// TIA Portal V20 export
FUNCTION_BLOCK "Sequence_1_JRUnloading"   // FB32865, LAD
TITLE = Sequence
// Sequence template programmend in ladder logic
// stored: IsIECCheckEnabled true, MemoryReserve 100, Namespace Unit1.Em13, SetENOAutomatically true
   VAR_INPUT
      unitStatus { ExternalAccessible := 'False'; ExternalVisible := 'False'; ExternalWritable := 'False'} : "LAF_typeUnitStatus";   // Current unit status o be used in this EM
   END_VAR
   VAR
      instSequenceLADControl { ExternalAccessible := 'False'; ExternalVisible := 'False'; ExternalWritable := 'False'} : "LAF_ControlLadSequence";
      instSequenceLADStatus { ExternalAccessible := 'False'; ExternalVisible := 'False'; ExternalWritable := 'False'} : "LAF_StatusLadSequence";
      statTonTime { ExternalAccessible := 'False'; ExternalVisible := 'False'; ExternalWritable := 'False'} : Array[0..9999] of TON_TIME;
      NoDataCheck { S7_SetPoint := 'True'} : "LER_typePartData";
      statPulse { ExternalWritable := 'False'} : Array[0..9] of Bool;
   END_VAR
   VAR_TEMP
      tempCustomerAction : Bool;   // Placeholder for possible actions
      tempDo_nothing_and_wait_for_init : Bool;   // Placeholder for doing nothing
      tempSafeStateCondition : Bool;   // Temp Condition for the equipment module to be in a safe state
   END_VAR
   VAR CONSTANT
      STEP_IDLE : DInt := 1;
      JOB_1_STEP_01 : DInt := 101;
      JOB_1_STEP_10 : DInt := 110;
      JOB_1_STEP_20 : DInt := 120;
      JOB_1_STEP_30 : DInt := 130;
      JOB_1_STEP_40 : DInt := 140;
      JOB_1_STEP_50 : DInt := 150;
      JOB_1_STEP_60 : DInt := 160;
      JOB_1_STEP_70 : DInt := 170;
      JOB_1_STEP_80 : DInt := 180;
      JOB_1_STEP_90 : DInt := 190;
      JOB_2_STEP_01 : DInt := 201;
      JOB_2_STEP_10 : DInt := 210;
      JOB_2_STEP_20 : DInt := 220;
      JOB_2_STEP_30 : DInt := 230;
      JOB_2_STEP_40 : DInt := 240;
      JOB_2_STEP_50 : DInt := 250;
      JOB_2_STEP_51 : DInt := 251;
      JOB_2_STEP_60 : DInt := 260;
      JOB_2_STEP_70 : DInt := 270;
      JOB_2_STEP_80 : DInt := 280;
      JOB_2_STEP_90 : DInt := 290;
      JOB_3_STEP_01 : DInt := 301;
      JOB_3_STEP_10 : DInt := 310;
      JOB_3_STEP_20 : DInt := 320;
      JOB_3_STEP_30 : DInt := 330;
      JOB_3_STEP_31 : DInt := 331;
      JOB_3_STEP_32 : DInt := 332;
      JOB_3_STEP_33 : DInt := 333;
      JOB_3_STEP_34 : DInt := 334;
      JOB_3_STEP_35 : DInt := 335;
      JOB_3_STEP_36 : DInt := 336;
      JOB_3_STEP_37 : DInt := 337;
      JOB_3_STEP_38 : DInt := 338;
      JOB_3_STEP_39 : DInt := 339;
      JOB_3_STEP_40 : DInt := 340;
      JOB_3_STEP_41 : DInt := 341;
      JOB_3_STEP_50 : DInt := 350;
      JOB_3_STEP_60 : DInt := 360;
      JOB_3_STEP_70 : DInt := 370;
      JOB_3_STEP_80 : DInt := 380;
      JOB_3_STEP_90 : DInt := 390;
      JOB_4_STEP_01 : DInt := 401;
      JOB_4_STEP_10 : DInt := 410;
      JOB_4_STEP_11 : DInt := 411;
      JOB_4_STEP_20 : DInt := 420;
      JOB_4_STEP_30 : DInt := 430;
      JOB_4_STEP_31 : DInt := 431;
      JOB_4_STEP_40 : DInt := 440;
      JOB_4_STEP_50 : DInt := 450;
      JOB_4_STEP_51 : DInt := 451;
      JOB_4_STEP_60 : DInt := 460;
      JOB_4_STEP_70 : DInt := 470;
      JOB_4_STEP_71 : DInt := 471;
      JOB_4_STEP_80 : DInt := 480;
      JOB_4_STEP_90 : DInt := 490;
      STEP_IMMEDIATE_STOP : DInt := 9001;   // Step executed when an immediate stop command is triggered for the sequence (i.e. when unit is in state aborting)
      TO_DO_INSERT_ACTIONS_HERE : Bool := TRUE;   // Template : Add actions
      TO_DO_INSERT_CONDITION_FOR_TRANSITION_HERE : Bool := TRUE;   // Template : Add conditions
   END_VAR
   VAR_TEMP   // added for the SCL form of the ladder/FBD networks
      _w1 : Bool;
      _w2 : Bool;
      _w3 : Bool;
      _w4 : Bool;
      _w5 : Bool;
   END_VAR
BEGIN

REGION Network 1: BLOCK INFO HEADER
   // (company) / (C) Copyright (year)
   // ---------------------------------------------------------------------------------
   // Title:                             (Title of this block)
   // Comment/Function: (that is implemented in the block)
   // Library/Family:           (that the source is dedicated to)
   // Author:                        (department / person in charge / contact)
   // Target System:          (test system with FW version)
   // Engineering:              TIA Portal (SW version)
   // Restrictions:               (OB types, etc.)
   // Requirements:           (hardware, technological package, etc.)
   // ---------------------------------------------------------------------------------
   // Change log table:
   // Version          | Date             | Signature      | Expert in charge  | Changes applied ------------------------|----------------------|-------------------------|--------------------------------|-----------------------
   // 001.000.000 | yyyy-mm-dd | 0x00000000 | (name of expert) | First released version
END_REGION

REGION Network 2: DESCRIPTION
   // This is a template block provided by the Automation Framework. It can be used to create an own project.
   // The Block Info Header is prepared to put in your own data.
   // Description of the block could be added here and the docu created by Code2Docu.
END_REGION

REGION Network 3: ********************* CONTROL *************************
END_REGION

REGION Network 4: Sequence Control ("Enter your Sequins number here")
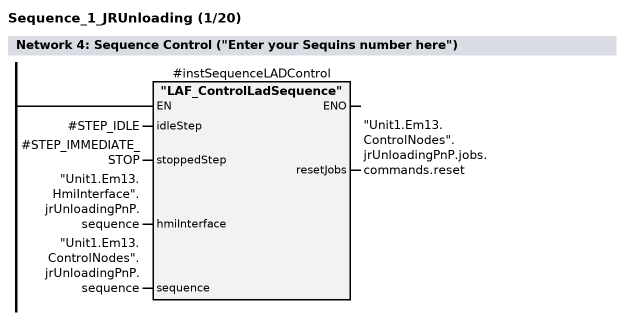
   RUNG wire#powerrail
      #instSequenceLADControl(idleStep := #STEP_IDLE, stoppedStep := #STEP_IMMEDIATE_STOP, hmiInterface := "Unit1.Em13.HmiInterface".jrUnloadingPnP.sequence, sequence := "Unit1.Em13.ControlNodes".jrUnloadingPnP.sequence, resetJobs => "Unit1.Em13.ControlNodes".jrUnloadingPnP.jobs.commands.reset)
   END_RUNG
   // the same network as SCL:
   #instSequenceLADControl(idleStep := #STEP_IDLE,   // "LAF_ControlLadSequence"
                           stoppedStep := #STEP_IMMEDIATE_STOP,
                           hmiInterface := "Unit1.Em13.HmiInterface".jrUnloadingPnP.sequence,
                           sequence := "Unit1.Em13.ControlNodes".jrUnloadingPnP.sequence,
                           resetJobs => "Unit1.Em13.ControlNodes".jrUnloadingPnP.jobs.commands.reset);
END_REGION

REGION Network 5: Step IDLE
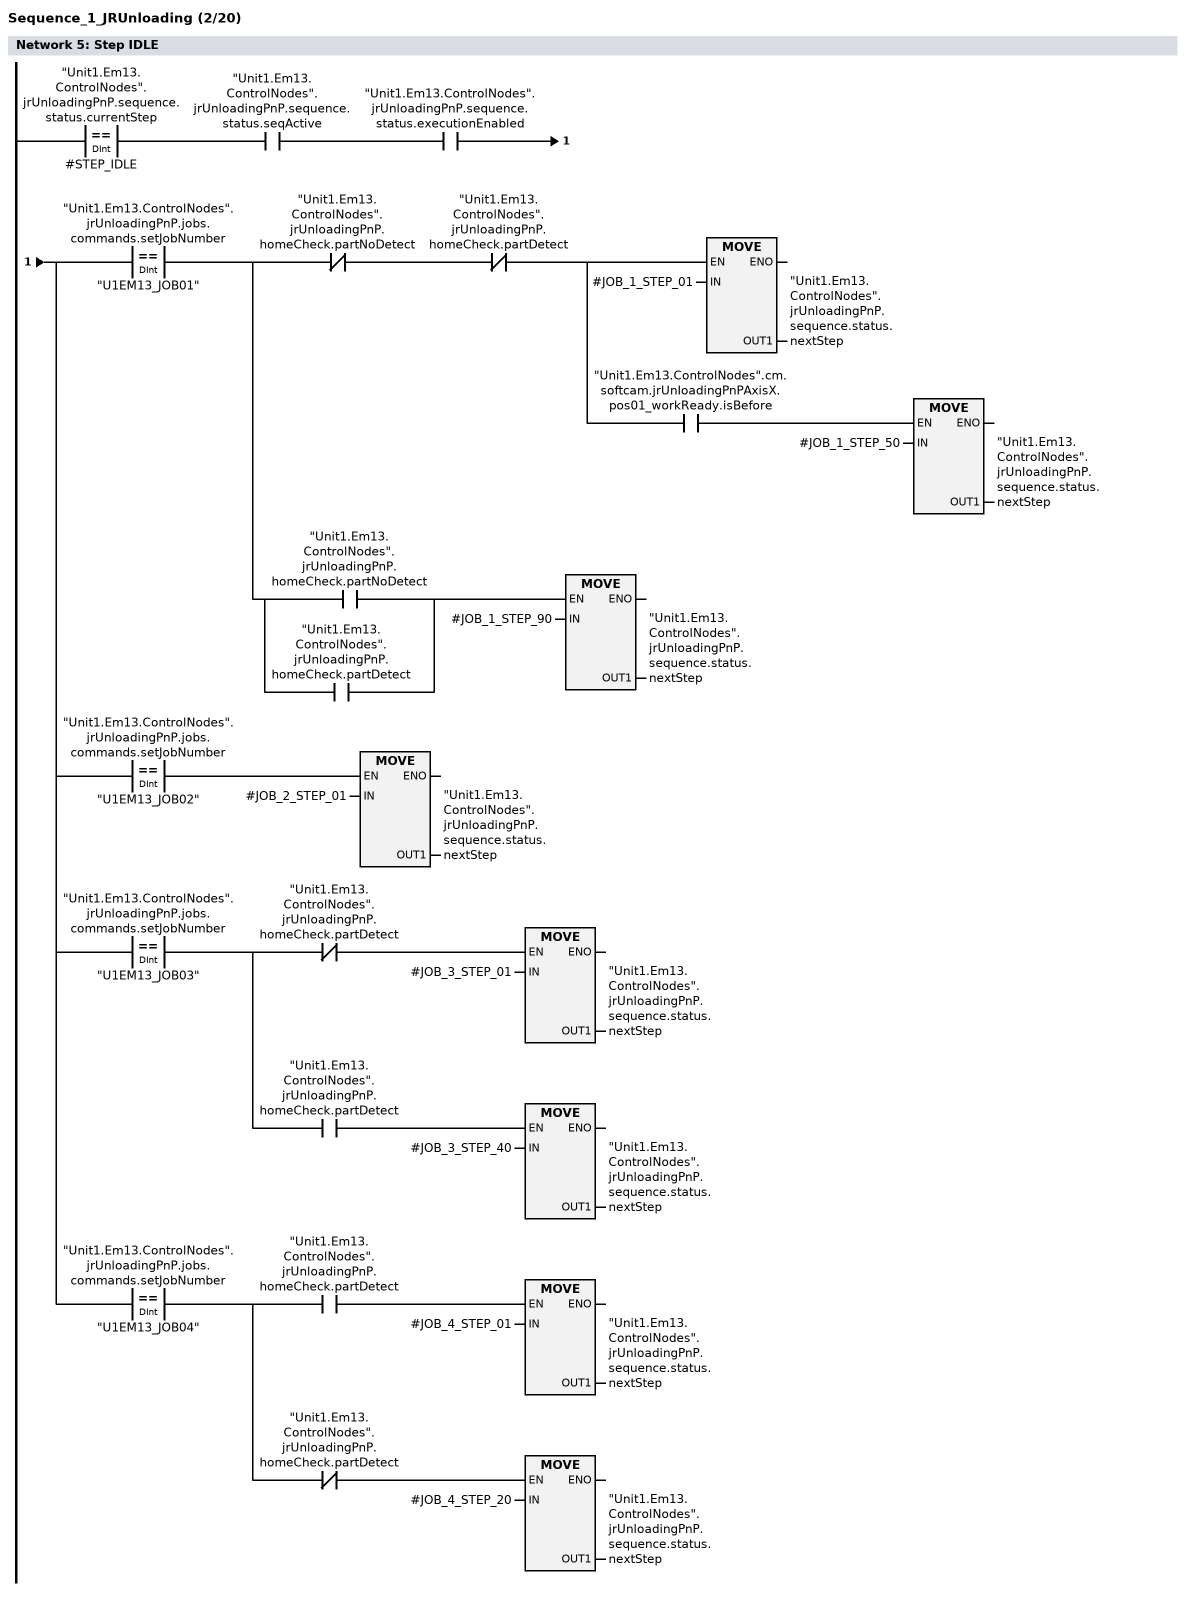
   RUNG wire#powerrail
      { S7_Templates := "SrcType := DInt" } EQ_Contact(in1 := "Unit1.Em13.ControlNodes".jrUnloadingPnP.sequence.status.currentStep, in2 := #STEP_IDLE)
      Contact( "Unit1.Em13.ControlNodes".jrUnloadingPnP.sequence.status.seqActive )
      Contact( "Unit1.Em13.ControlNodes".jrUnloadingPnP.sequence.status.executionEnabled )
      wire#w1
      { S7_Templates := "SrcType := DInt" } EQ_Contact(in1 := "Unit1.Em13.ControlNodes".jrUnloadingPnP.jobs.commands.setJobNumber, in2 := "U1EM13_JOB01")
      wire#w2
      I_Contact( "Unit1.Em13.ControlNodes".jrUnloadingPnP.homeCheck.partNoDetect )
      I_Contact( "Unit1.Em13.ControlNodes".jrUnloadingPnP.homeCheck.partDetect )
      wire#w3
      Move(in := #JOB_1_STEP_01, out1 => "Unit1.Em13.ControlNodes".jrUnloadingPnP.sequence.status.nextStep)
   END_RUNG
   RUNG wire#w3
      Contact( "Unit1.Em13.ControlNodes".cm.softcam.jrUnIoadingPnPAxisX.pos01_workReady.isBefore )
      Move(in := #JOB_1_STEP_50, out1 => "Unit1.Em13.ControlNodes".jrUnloadingPnP.sequence.status.nextStep)
   END_RUNG
   RUNG wire#w2
      Contact( "Unit1.Em13.ControlNodes".jrUnloadingPnP.homeCheck.partNoDetect )
      wire#w4
      Move(in := #JOB_1_STEP_90, out1 => "Unit1.Em13.ControlNodes".jrUnloadingPnP.sequence.status.nextStep)
   END_RUNG
   RUNG wire#w2
      Contact( "Unit1.Em13.ControlNodes".jrUnloadingPnP.homeCheck.partDetect )
   END_RUNG wire#w4
   RUNG wire#w1
      { S7_Templates := "SrcType := DInt" } EQ_Contact(in1 := "Unit1.Em13.ControlNodes".jrUnloadingPnP.jobs.commands.setJobNumber, in2 := "U1EM13_JOB02")
      Move(in := #JOB_2_STEP_01, out1 => "Unit1.Em13.ControlNodes".jrUnloadingPnP.sequence.status.nextStep)
   END_RUNG
   RUNG wire#w1
      { S7_Templates := "SrcType := DInt" } EQ_Contact(in1 := "Unit1.Em13.ControlNodes".jrUnloadingPnP.jobs.commands.setJobNumber, in2 := "U1EM13_JOB03")
      wire#w5
      I_Contact( "Unit1.Em13.ControlNodes".jrUnloadingPnP.homeCheck.partDetect )
      Move(in := #JOB_3_STEP_01, out1 => "Unit1.Em13.ControlNodes".jrUnloadingPnP.sequence.status.nextStep)
   END_RUNG
   RUNG wire#w5
      Contact( "Unit1.Em13.ControlNodes".jrUnloadingPnP.homeCheck.partDetect )
      Move(in := #JOB_3_STEP_40, out1 => "Unit1.Em13.ControlNodes".jrUnloadingPnP.sequence.status.nextStep)
   END_RUNG
   RUNG wire#w1
      { S7_Templates := "SrcType := DInt" } EQ_Contact(in1 := "Unit1.Em13.ControlNodes".jrUnloadingPnP.jobs.commands.setJobNumber, in2 := "U1EM13_JOB04")
      wire#w6
      Contact( "Unit1.Em13.ControlNodes".jrUnloadingPnP.homeCheck.partDetect )
      Move(in := #JOB_4_STEP_01, out1 => "Unit1.Em13.ControlNodes".jrUnloadingPnP.sequence.status.nextStep)
   END_RUNG
   RUNG wire#w6
      I_Contact( "Unit1.Em13.ControlNodes".jrUnloadingPnP.homeCheck.partDetect )
      Move(in := #JOB_4_STEP_20, out1 => "Unit1.Em13.ControlNodes".jrUnloadingPnP.sequence.status.nextStep)
   END_RUNG
   // the same network as SCL:
   #_w1 := ("Unit1.Em13.ControlNodes".jrUnloadingPnP.sequence.status.currentStep = #STEP_IDLE) AND "Unit1.Em13.ControlNodes".jrUnloadingPnP.sequence.status.seqActive AND "Unit1.Em13.ControlNodes".jrUnloadingPnP.sequence.status.executionEnabled;
   #_w2 := #_w1 AND ("Unit1.Em13.ControlNodes".jrUnloadingPnP.jobs.commands.setJobNumber = "U1EM13_JOB01");
   #_w3 := #_w2 AND NOT "Unit1.Em13.ControlNodes".jrUnloadingPnP.homeCheck.partNoDetect AND NOT "Unit1.Em13.ControlNodes".jrUnloadingPnP.homeCheck.partDetect;
   IF #_w3 THEN "Unit1.Em13.ControlNodes".jrUnloadingPnP.sequence.status.nextStep := #JOB_1_STEP_01; END_IF;
   IF #_w3 AND "Unit1.Em13.ControlNodes".cm.softcam.jrUnIoadingPnPAxisX.pos01_workReady.isBefore THEN
       "Unit1.Em13.ControlNodes".jrUnloadingPnP.sequence.status.nextStep := #JOB_1_STEP_50;
   END_IF;
   IF #_w2 AND ("Unit1.Em13.ControlNodes".jrUnloadingPnP.homeCheck.partNoDetect OR "Unit1.Em13.ControlNodes".jrUnloadingPnP.homeCheck.partDetect) THEN
       "Unit1.Em13.ControlNodes".jrUnloadingPnP.sequence.status.nextStep := #JOB_1_STEP_90;
   END_IF;
   IF #_w1 AND ("Unit1.Em13.ControlNodes".jrUnloadingPnP.jobs.commands.setJobNumber = "U1EM13_JOB02") THEN
       "Unit1.Em13.ControlNodes".jrUnloadingPnP.sequence.status.nextStep := #JOB_2_STEP_01;
   END_IF;
   #_w4 := #_w1 AND ("Unit1.Em13.ControlNodes".jrUnloadingPnP.jobs.commands.setJobNumber = "U1EM13_JOB03");
   IF #_w4 AND NOT "Unit1.Em13.ControlNodes".jrUnloadingPnP.homeCheck.partDetect THEN
       "Unit1.Em13.ControlNodes".jrUnloadingPnP.sequence.status.nextStep := #JOB_3_STEP_01;
   END_IF;
   IF #_w4 AND "Unit1.Em13.ControlNodes".jrUnloadingPnP.homeCheck.partDetect THEN
       "Unit1.Em13.ControlNodes".jrUnloadingPnP.sequence.status.nextStep := #JOB_3_STEP_40;
   END_IF;
   #_w5 := #_w1 AND ("Unit1.Em13.ControlNodes".jrUnloadingPnP.jobs.commands.setJobNumber = "U1EM13_JOB04");
   IF #_w5 AND "Unit1.Em13.ControlNodes".jrUnloadingPnP.homeCheck.partDetect THEN
       "Unit1.Em13.ControlNodes".jrUnloadingPnP.sequence.status.nextStep := #JOB_4_STEP_01;
   END_IF;
   IF #_w5 AND NOT "Unit1.Em13.ControlNodes".jrUnloadingPnP.homeCheck.partDetect THEN
       "Unit1.Em13.ControlNodes".jrUnloadingPnP.sequence.status.nextStep := #JOB_4_STEP_20;
   END_IF;
END_REGION

REGION Network 6: *************** JOB[1] EM HOMING ************************
END_REGION

REGION Network 7: Step[101] : JOB[1] Condition
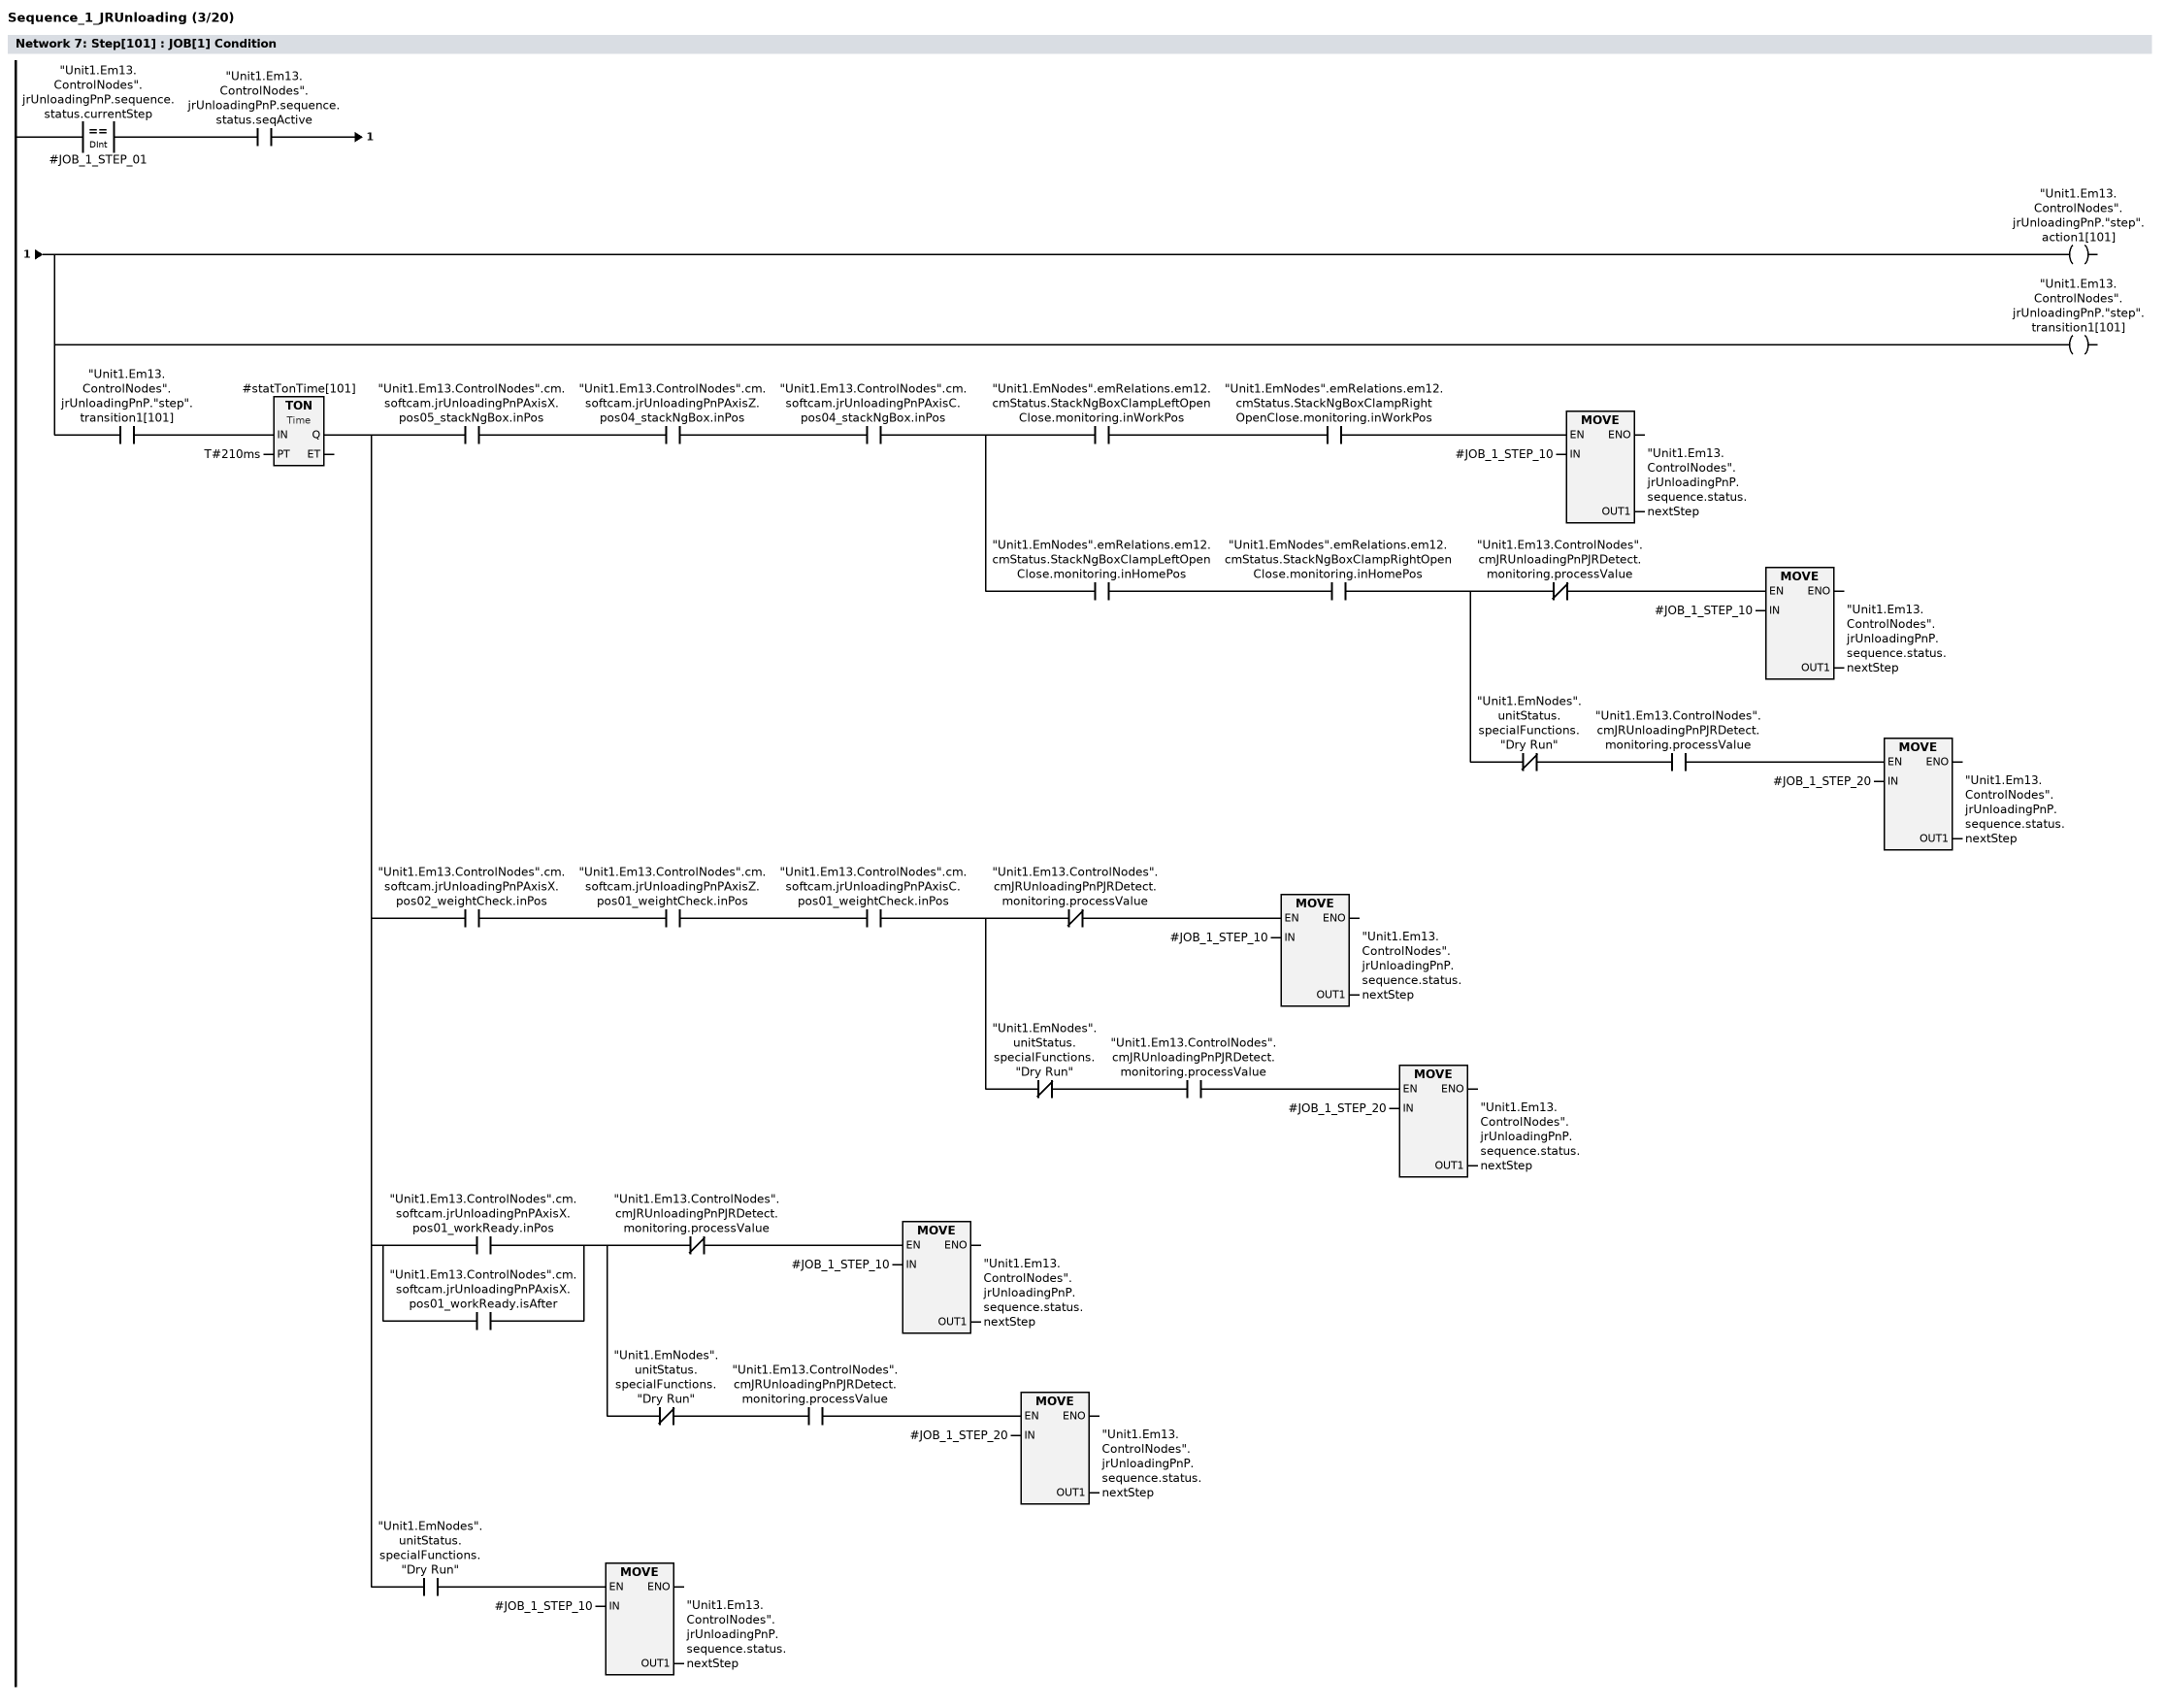
   RUNG wire#powerrail
      { S7_Templates := "SrcType := DInt" } EQ_Contact(in1 := "Unit1.Em13.ControlNodes".jrUnloadingPnP.sequence.status.currentStep, in2 := #JOB_1_STEP_01)
      Contact( "Unit1.Em13.ControlNodes".jrUnloadingPnP.sequence.status.seqActive )
      wire#w1
      Coil( "Unit1.Em13.ControlNodes".jrUnloadingPnP."step".action1[101] )
   END_RUNG
   RUNG wire#w1
      Coil( "Unit1.Em13.ControlNodes".jrUnloadingPnP."step".transition1[101] )
   END_RUNG
   RUNG wire#w1
      Contact( "Unit1.Em13.ControlNodes".jrUnloadingPnP."step".transition1[101] )
      { S7_Templates := "time_type := Time" } #statTonTime[101].TON(pt := T#210ms, et =>)
      wire#w2
      Contact( "Unit1.Em13.ControlNodes".cm.softcam.jrUnIoadingPnPAxisX.pos05_stackNgBox.inPos )
      Contact( "Unit1.Em13.ControlNodes".cm.softcam.jrUnIoadingPnPAxisZ.pos04_stackNgBox.inPos )
      Contact( "Unit1.Em13.ControlNodes".cm.softcam.jrUnIoadingPnPAxisC.pos04_stackNgBox.inPos )
      wire#w3
      Contact( "Unit1.EmNodes".emRelations.em12.cmStatus.StackNgBoxClampLeftOpenClose.monitoring.inWorkPos )
      Contact( "Unit1.EmNodes".emRelations.em12.cmStatus.StackNgBoxClampRightOpenClose.monitoring.inWorkPos )
      Move(in := #JOB_1_STEP_10, out1 => "Unit1.Em13.ControlNodes".jrUnloadingPnP.sequence.status.nextStep)
   END_RUNG
   RUNG wire#w3
      Contact( "Unit1.EmNodes".emRelations.em12.cmStatus.StackNgBoxClampLeftOpenClose.monitoring.inHomePos )
      Contact( "Unit1.EmNodes".emRelations.em12.cmStatus.StackNgBoxClampRightOpenClose.monitoring.inHomePos )
      wire#w4
      I_Contact( "Unit1.Em13.ControlNodes".cmJRUnloadingPnPJRDetect.monitoring.processValue )
      Move(in := #JOB_1_STEP_10, out1 => "Unit1.Em13.ControlNodes".jrUnloadingPnP.sequence.status.nextStep)
   END_RUNG
   RUNG wire#w4
      I_Contact( "Unit1.EmNodes".unitStatus.specialFunctions."Dry Run" )
      Contact( "Unit1.Em13.ControlNodes".cmJRUnloadingPnPJRDetect.monitoring.processValue )
      Move(in := #JOB_1_STEP_20, out1 => "Unit1.Em13.ControlNodes".jrUnloadingPnP.sequence.status.nextStep)
   END_RUNG
   RUNG wire#w2
      Contact( "Unit1.Em13.ControlNodes".cm.softcam.jrUnIoadingPnPAxisX.pos02_weightCheck.inPos )
      Contact( "Unit1.Em13.ControlNodes".cm.softcam.jrUnIoadingPnPAxisZ.pos01_weightCheck.inPos )
      Contact( "Unit1.Em13.ControlNodes".cm.softcam.jrUnIoadingPnPAxisC.pos01_weightCheck.inPos )
      wire#w5
      I_Contact( "Unit1.Em13.ControlNodes".cmJRUnloadingPnPJRDetect.monitoring.processValue )
      Move(in := #JOB_1_STEP_10, out1 => "Unit1.Em13.ControlNodes".jrUnloadingPnP.sequence.status.nextStep)
   END_RUNG
   RUNG wire#w5
      I_Contact( "Unit1.EmNodes".unitStatus.specialFunctions."Dry Run" )
      Contact( "Unit1.Em13.ControlNodes".cmJRUnloadingPnPJRDetect.monitoring.processValue )
      Move(in := #JOB_1_STEP_20, out1 => "Unit1.Em13.ControlNodes".jrUnloadingPnP.sequence.status.nextStep)
   END_RUNG
   RUNG wire#w2
      Contact( "Unit1.Em13.ControlNodes".cm.softcam.jrUnIoadingPnPAxisX.pos01_workReady.inPos )
      wire#w6
      I_Contact( "Unit1.Em13.ControlNodes".cmJRUnloadingPnPJRDetect.monitoring.processValue )
      Move(in := #JOB_1_STEP_10, out1 => "Unit1.Em13.ControlNodes".jrUnloadingPnP.sequence.status.nextStep)
   END_RUNG
   RUNG wire#w2
      Contact( "Unit1.Em13.ControlNodes".cm.softcam.jrUnIoadingPnPAxisX.pos01_workReady.isAfter )
   END_RUNG wire#w6
   RUNG wire#w6
      I_Contact( "Unit1.EmNodes".unitStatus.specialFunctions."Dry Run" )
      Contact( "Unit1.Em13.ControlNodes".cmJRUnloadingPnPJRDetect.monitoring.processValue )
      Move(in := #JOB_1_STEP_20, out1 => "Unit1.Em13.ControlNodes".jrUnloadingPnP.sequence.status.nextStep)
   END_RUNG
   RUNG wire#w2
      Contact( "Unit1.EmNodes".unitStatus.specialFunctions."Dry Run" )
      Move(in := #JOB_1_STEP_10, out1 => "Unit1.Em13.ControlNodes".jrUnloadingPnP.sequence.status.nextStep)
   END_RUNG
   // the same network as SCL:
   "Unit1.Em13.ControlNodes".jrUnloadingPnP."step".action1[101] := ("Unit1.Em13.ControlNodes".jrUnloadingPnP.sequence.status.currentStep = #JOB_1_STEP_01) AND "Unit1.Em13.ControlNodes".jrUnloadingPnP.sequence.status.seqActive;
   "Unit1.Em13.ControlNodes".jrUnloadingPnP."step".transition1[101] := ("Unit1.Em13.ControlNodes".jrUnloadingPnP.sequence.status.currentStep = #JOB_1_STEP_01) AND "Unit1.Em13.ControlNodes".jrUnloadingPnP.sequence.status.seqActive;
   #statTonTime[101].TON(IN := ("Unit1.Em13.ControlNodes".jrUnloadingPnP.sequence.status.currentStep = #JOB_1_STEP_01) AND "Unit1.Em13.ControlNodes".jrUnloadingPnP.sequence.status.seqActive AND "Unit1.Em13.ControlNodes".jrUnloadingPnP."step".transition1[101],
                         PT := T#210ms);
   #_w1 := #statTonTime[101].Q AND "Unit1.Em13.ControlNodes".cm.softcam.jrUnIoadingPnPAxisX.pos05_stackNgBox.inPos AND "Unit1.Em13.ControlNodes".cm.softcam.jrUnIoadingPnPAxisZ.pos04_stackNgBox.inPos AND "Unit1.Em13.ControlNodes".cm.softcam.jrUnIoadingPnPAxisC.pos04_stackNgBox.inPos;
   IF #_w1 AND "Unit1.EmNodes".emRelations.em12.cmStatus.StackNgBoxClampLeftOpenClose.monitoring.inWorkPos AND "Unit1.EmNodes".emRelations.em12.cmStatus.StackNgBoxClampRightOpenClose.monitoring.inWorkPos THEN
       "Unit1.Em13.ControlNodes".jrUnloadingPnP.sequence.status.nextStep := #JOB_1_STEP_10;
   END_IF;
   #_w2 := #_w1 AND "Unit1.EmNodes".emRelations.em12.cmStatus.StackNgBoxClampLeftOpenClose.monitoring.inHomePos AND "Unit1.EmNodes".emRelations.em12.cmStatus.StackNgBoxClampRightOpenClose.monitoring.inHomePos;
   IF #_w2 AND NOT "Unit1.Em13.ControlNodes".cmJRUnloadingPnPJRDetect.monitoring.processValue THEN
       "Unit1.Em13.ControlNodes".jrUnloadingPnP.sequence.status.nextStep := #JOB_1_STEP_10;
   END_IF;
   IF #_w2 AND NOT "Unit1.EmNodes".unitStatus.specialFunctions."Dry Run" AND "Unit1.Em13.ControlNodes".cmJRUnloadingPnPJRDetect.monitoring.processValue THEN
       "Unit1.Em13.ControlNodes".jrUnloadingPnP.sequence.status.nextStep := #JOB_1_STEP_20;
   END_IF;
   #_w3 := #statTonTime[101].Q AND "Unit1.Em13.ControlNodes".cm.softcam.jrUnIoadingPnPAxisX.pos02_weightCheck.inPos AND "Unit1.Em13.ControlNodes".cm.softcam.jrUnIoadingPnPAxisZ.pos01_weightCheck.inPos AND "Unit1.Em13.ControlNodes".cm.softcam.jrUnIoadingPnPAxisC.pos01_weightCheck.inPos;
   IF #_w3 AND NOT "Unit1.Em13.ControlNodes".cmJRUnloadingPnPJRDetect.monitoring.processValue THEN
       "Unit1.Em13.ControlNodes".jrUnloadingPnP.sequence.status.nextStep := #JOB_1_STEP_10;
   END_IF;
   IF #_w3 AND NOT "Unit1.EmNodes".unitStatus.specialFunctions."Dry Run" AND "Unit1.Em13.ControlNodes".cmJRUnloadingPnPJRDetect.monitoring.processValue THEN
       "Unit1.Em13.ControlNodes".jrUnloadingPnP.sequence.status.nextStep := #JOB_1_STEP_20;
   END_IF;
   #_w4 := #statTonTime[101].Q AND ("Unit1.Em13.ControlNodes".cm.softcam.jrUnIoadingPnPAxisX.pos01_workReady.inPos OR "Unit1.Em13.ControlNodes".cm.softcam.jrUnIoadingPnPAxisX.pos01_workReady.isAfter);
   IF #_w4 AND NOT "Unit1.Em13.ControlNodes".cmJRUnloadingPnPJRDetect.monitoring.processValue THEN
       "Unit1.Em13.ControlNodes".jrUnloadingPnP.sequence.status.nextStep := #JOB_1_STEP_10;
   END_IF;
   IF #_w4 AND NOT "Unit1.EmNodes".unitStatus.specialFunctions."Dry Run" AND "Unit1.Em13.ControlNodes".cmJRUnloadingPnPJRDetect.monitoring.processValue THEN
       "Unit1.Em13.ControlNodes".jrUnloadingPnP.sequence.status.nextStep := #JOB_1_STEP_20;
   END_IF;
   IF #statTonTime[101].Q AND "Unit1.EmNodes".unitStatus.specialFunctions."Dry Run" THEN
       "Unit1.Em13.ControlNodes".jrUnloadingPnP.sequence.status.nextStep := #JOB_1_STEP_10;
   END_IF;
END_REGION

REGION Network 8: Step[110] : Clamp Open
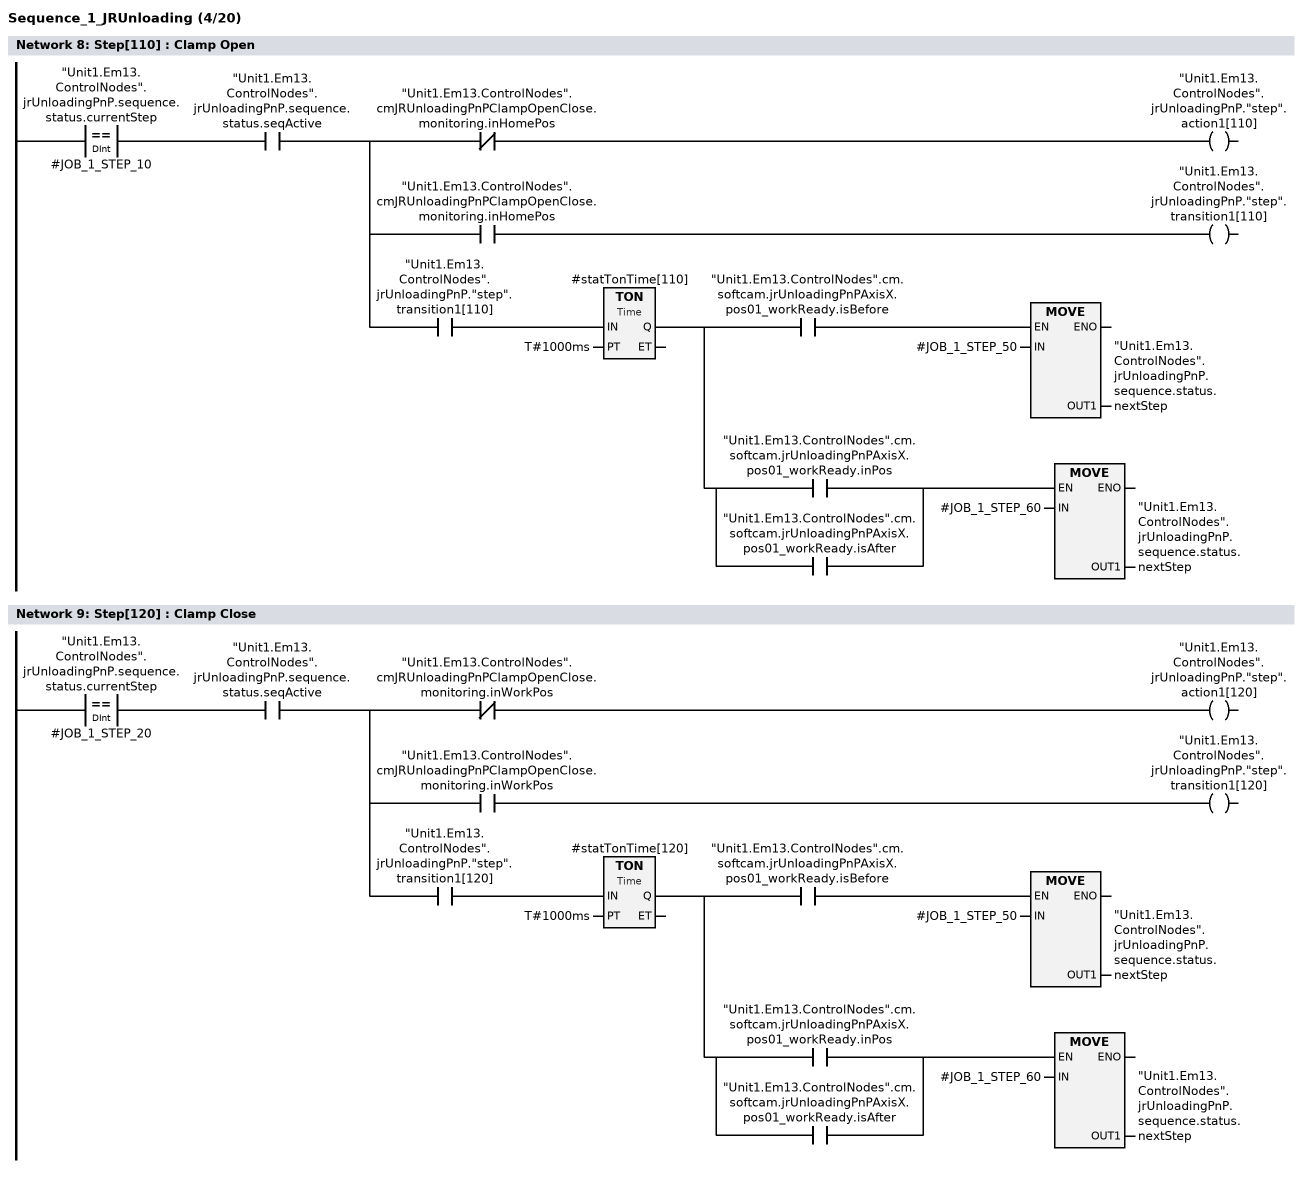
   RUNG wire#powerrail
      { S7_Templates := "SrcType := DInt" } EQ_Contact(in1 := "Unit1.Em13.ControlNodes".jrUnloadingPnP.sequence.status.currentStep, in2 := #JOB_1_STEP_10)
      Contact( "Unit1.Em13.ControlNodes".jrUnloadingPnP.sequence.status.seqActive )
      wire#w1
      I_Contact( "Unit1.Em13.ControlNodes".cmJRUnloadingPnPClampOpenClose.monitoring.inHomePos )
      Coil( "Unit1.Em13.ControlNodes".jrUnloadingPnP."step".action1[110] )
   END_RUNG
   RUNG wire#w1
      Contact( "Unit1.Em13.ControlNodes".cmJRUnloadingPnPClampOpenClose.monitoring.inHomePos )
      Coil( "Unit1.Em13.ControlNodes".jrUnloadingPnP."step".transition1[110] )
   END_RUNG
   RUNG wire#w1
      Contact( "Unit1.Em13.ControlNodes".jrUnloadingPnP."step".transition1[110] )
      { S7_Templates := "time_type := Time" } #statTonTime[110].TON(pt := T#1000ms, et =>)
      wire#w2
      Contact( "Unit1.Em13.ControlNodes".cm.softcam.jrUnIoadingPnPAxisX.pos01_workReady.isBefore )
      Move(in := #JOB_1_STEP_50, out1 => "Unit1.Em13.ControlNodes".jrUnloadingPnP.sequence.status.nextStep)
   END_RUNG
   RUNG wire#w2
      Contact( "Unit1.Em13.ControlNodes".cm.softcam.jrUnIoadingPnPAxisX.pos01_workReady.inPos )
      wire#w3
      Move(in := #JOB_1_STEP_60, out1 => "Unit1.Em13.ControlNodes".jrUnloadingPnP.sequence.status.nextStep)
   END_RUNG
   RUNG wire#w2
      Contact( "Unit1.Em13.ControlNodes".cm.softcam.jrUnIoadingPnPAxisX.pos01_workReady.isAfter )
   END_RUNG wire#w3
   // the same network as SCL:
   #_w1 := ("Unit1.Em13.ControlNodes".jrUnloadingPnP.sequence.status.currentStep = #JOB_1_STEP_10) AND "Unit1.Em13.ControlNodes".jrUnloadingPnP.sequence.status.seqActive;
   "Unit1.Em13.ControlNodes".jrUnloadingPnP."step".action1[110] := #_w1 AND NOT "Unit1.Em13.ControlNodes".cmJRUnloadingPnPClampOpenClose.monitoring.inHomePos;
   "Unit1.Em13.ControlNodes".jrUnloadingPnP."step".transition1[110] := #_w1 AND "Unit1.Em13.ControlNodes".cmJRUnloadingPnPClampOpenClose.monitoring.inHomePos;
   #statTonTime[110].TON(IN := #_w1 AND "Unit1.Em13.ControlNodes".jrUnloadingPnP."step".transition1[110],
                         PT := T#1000ms);
   IF #statTonTime[110].Q AND "Unit1.Em13.ControlNodes".cm.softcam.jrUnIoadingPnPAxisX.pos01_workReady.isBefore THEN
       "Unit1.Em13.ControlNodes".jrUnloadingPnP.sequence.status.nextStep := #JOB_1_STEP_50;
   END_IF;
   IF #statTonTime[110].Q AND ("Unit1.Em13.ControlNodes".cm.softcam.jrUnIoadingPnPAxisX.pos01_workReady.inPos OR "Unit1.Em13.ControlNodes".cm.softcam.jrUnIoadingPnPAxisX.pos01_workReady.isAfter) THEN
       "Unit1.Em13.ControlNodes".jrUnloadingPnP.sequence.status.nextStep := #JOB_1_STEP_60;
   END_IF;
END_REGION

REGION Network 9: Step[120] : Clamp Close
   RUNG wire#powerrail
      { S7_Templates := "SrcType := DInt" } EQ_Contact(in1 := "Unit1.Em13.ControlNodes".jrUnloadingPnP.sequence.status.currentStep, in2 := #JOB_1_STEP_20)
      Contact( "Unit1.Em13.ControlNodes".jrUnloadingPnP.sequence.status.seqActive )
      wire#w1
      I_Contact( "Unit1.Em13.ControlNodes".cmJRUnloadingPnPClampOpenClose.monitoring.inWorkPos )
      Coil( "Unit1.Em13.ControlNodes".jrUnloadingPnP."step".action1[120] )
   END_RUNG
   RUNG wire#w1
      Contact( "Unit1.Em13.ControlNodes".cmJRUnloadingPnPClampOpenClose.monitoring.inWorkPos )
      Coil( "Unit1.Em13.ControlNodes".jrUnloadingPnP."step".transition1[120] )
   END_RUNG
   RUNG wire#w1
      Contact( "Unit1.Em13.ControlNodes".jrUnloadingPnP."step".transition1[120] )
      { S7_Templates := "time_type := Time" } #statTonTime[120].TON(pt := T#1000ms, et =>)
      wire#w2
      Contact( "Unit1.Em13.ControlNodes".cm.softcam.jrUnIoadingPnPAxisX.pos01_workReady.isBefore )
      Move(in := #JOB_1_STEP_50, out1 => "Unit1.Em13.ControlNodes".jrUnloadingPnP.sequence.status.nextStep)
   END_RUNG
   RUNG wire#w2
      Contact( "Unit1.Em13.ControlNodes".cm.softcam.jrUnIoadingPnPAxisX.pos01_workReady.inPos )
      wire#w3
      Move(in := #JOB_1_STEP_60, out1 => "Unit1.Em13.ControlNodes".jrUnloadingPnP.sequence.status.nextStep)
   END_RUNG
   RUNG wire#w2
      Contact( "Unit1.Em13.ControlNodes".cm.softcam.jrUnIoadingPnPAxisX.pos01_workReady.isAfter )
   END_RUNG wire#w3
   // the same network as SCL:
   #_w1 := ("Unit1.Em13.ControlNodes".jrUnloadingPnP.sequence.status.currentStep = #JOB_1_STEP_20) AND "Unit1.Em13.ControlNodes".jrUnloadingPnP.sequence.status.seqActive;
   "Unit1.Em13.ControlNodes".jrUnloadingPnP."step".action1[120] := #_w1 AND NOT "Unit1.Em13.ControlNodes".cmJRUnloadingPnPClampOpenClose.monitoring.inWorkPos;
   "Unit1.Em13.ControlNodes".jrUnloadingPnP."step".transition1[120] := #_w1 AND "Unit1.Em13.ControlNodes".cmJRUnloadingPnPClampOpenClose.monitoring.inWorkPos;
   #statTonTime[120].TON(IN := #_w1 AND "Unit1.Em13.ControlNodes".jrUnloadingPnP."step".transition1[120],
                         PT := T#1000ms);
   IF #statTonTime[120].Q AND "Unit1.Em13.ControlNodes".cm.softcam.jrUnIoadingPnPAxisX.pos01_workReady.isBefore THEN
       "Unit1.Em13.ControlNodes".jrUnloadingPnP.sequence.status.nextStep := #JOB_1_STEP_50;
   END_IF;
   IF #statTonTime[120].Q AND ("Unit1.Em13.ControlNodes".cm.softcam.jrUnIoadingPnPAxisX.pos01_workReady.inPos OR "Unit1.Em13.ControlNodes".cm.softcam.jrUnIoadingPnPAxisX.pos01_workReady.isAfter) THEN
       "Unit1.Em13.ControlNodes".jrUnloadingPnP.sequence.status.nextStep := #JOB_1_STEP_60;
   END_IF;
END_REGION

REGION Network 10: Step[150] : JR Unload P&P X-axis Work Ready Position
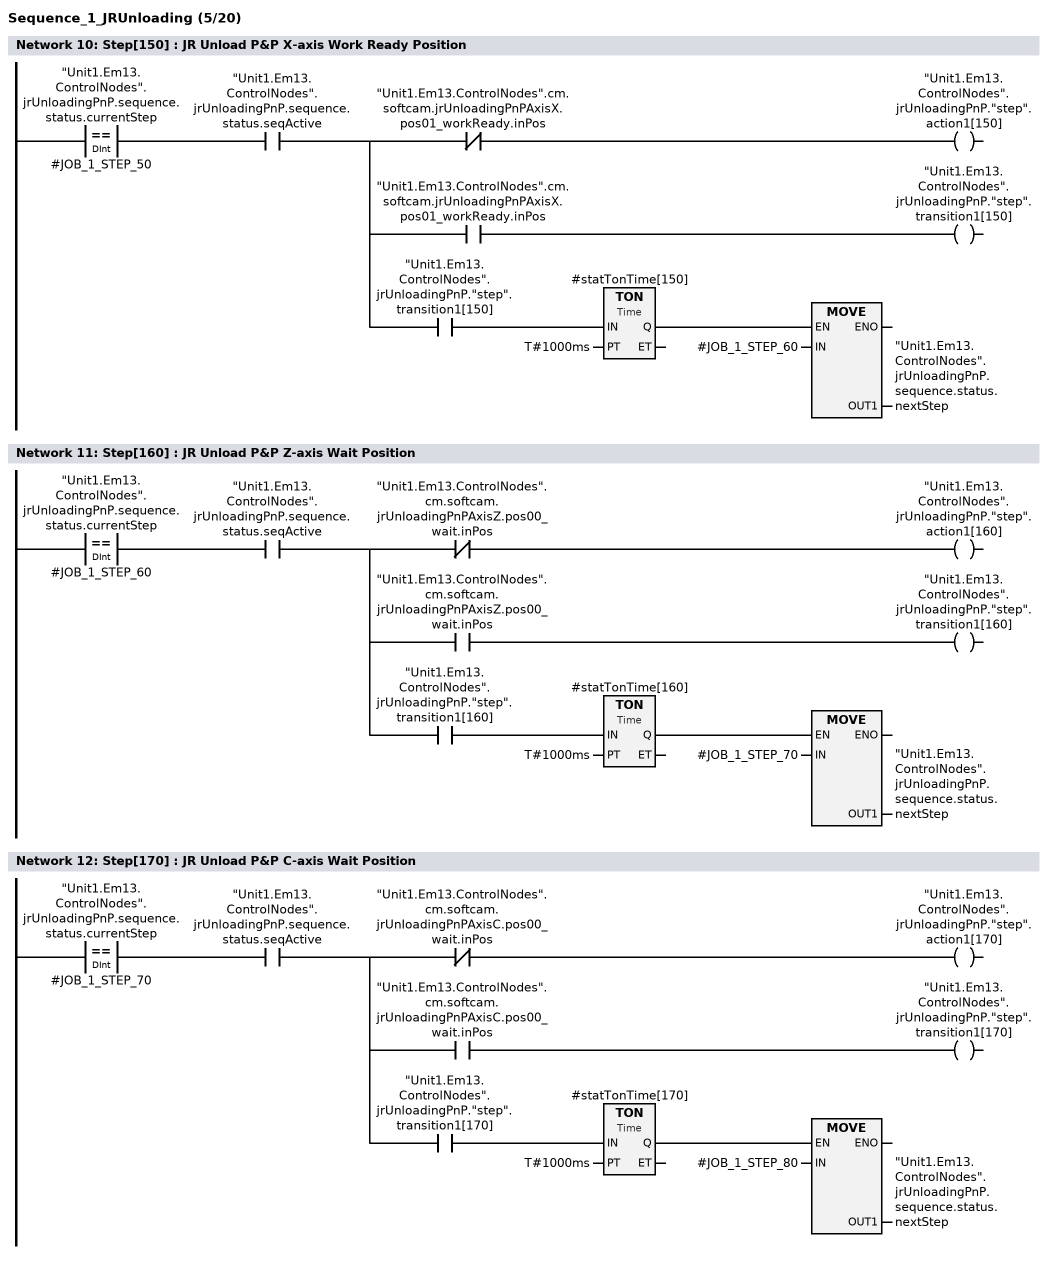
   RUNG wire#powerrail
      { S7_Templates := "SrcType := DInt" } EQ_Contact(in1 := "Unit1.Em13.ControlNodes".jrUnloadingPnP.sequence.status.currentStep, in2 := #JOB_1_STEP_50)
      Contact( "Unit1.Em13.ControlNodes".jrUnloadingPnP.sequence.status.seqActive )
      wire#w1
      I_Contact( "Unit1.Em13.ControlNodes".cm.softcam.jrUnIoadingPnPAxisX.pos01_workReady.inPos )
      Coil( "Unit1.Em13.ControlNodes".jrUnloadingPnP."step".action1[150] )
   END_RUNG
   RUNG wire#w1
      Contact( "Unit1.Em13.ControlNodes".cm.softcam.jrUnIoadingPnPAxisX.pos01_workReady.inPos )
      Coil( "Unit1.Em13.ControlNodes".jrUnloadingPnP."step".transition1[150] )
   END_RUNG
   RUNG wire#w1
      Contact( "Unit1.Em13.ControlNodes".jrUnloadingPnP."step".transition1[150] )
      { S7_Templates := "time_type := Time" } #statTonTime[150].TON(pt := T#1000ms, et =>)
      Move(in := #JOB_1_STEP_60, out1 => "Unit1.Em13.ControlNodes".jrUnloadingPnP.sequence.status.nextStep)
   END_RUNG
   // the same network as SCL:
   #_w1 := ("Unit1.Em13.ControlNodes".jrUnloadingPnP.sequence.status.currentStep = #JOB_1_STEP_50) AND "Unit1.Em13.ControlNodes".jrUnloadingPnP.sequence.status.seqActive;
   "Unit1.Em13.ControlNodes".jrUnloadingPnP."step".action1[150] := #_w1 AND NOT "Unit1.Em13.ControlNodes".cm.softcam.jrUnIoadingPnPAxisX.pos01_workReady.inPos;
   "Unit1.Em13.ControlNodes".jrUnloadingPnP."step".transition1[150] := #_w1 AND "Unit1.Em13.ControlNodes".cm.softcam.jrUnIoadingPnPAxisX.pos01_workReady.inPos;
   #statTonTime[150].TON(IN := #_w1 AND "Unit1.Em13.ControlNodes".jrUnloadingPnP."step".transition1[150],
                         PT := T#1000ms);
   IF #statTonTime[150].Q THEN
       "Unit1.Em13.ControlNodes".jrUnloadingPnP.sequence.status.nextStep := #JOB_1_STEP_60;
   END_IF;
END_REGION

REGION Network 11: Step[160] : JR Unload P&P Z-axis Wait Position
   RUNG wire#powerrail
      { S7_Templates := "SrcType := DInt" } EQ_Contact(in1 := "Unit1.Em13.ControlNodes".jrUnloadingPnP.sequence.status.currentStep, in2 := #JOB_1_STEP_60)
      Contact( "Unit1.Em13.ControlNodes".jrUnloadingPnP.sequence.status.seqActive )
      wire#w1
      I_Contact( "Unit1.Em13.ControlNodes".cm.softcam.jrUnIoadingPnPAxisZ.pos00_wait.inPos )
      Coil( "Unit1.Em13.ControlNodes".jrUnloadingPnP."step".action1[160] )
   END_RUNG
   RUNG wire#w1
      Contact( "Unit1.Em13.ControlNodes".cm.softcam.jrUnIoadingPnPAxisZ.pos00_wait.inPos )
      Coil( "Unit1.Em13.ControlNodes".jrUnloadingPnP."step".transition1[160] )
   END_RUNG
   RUNG wire#w1
      Contact( "Unit1.Em13.ControlNodes".jrUnloadingPnP."step".transition1[160] )
      { S7_Templates := "time_type := Time" } #statTonTime[160].TON(pt := T#1000ms, et =>)
      Move(in := #JOB_1_STEP_70, out1 => "Unit1.Em13.ControlNodes".jrUnloadingPnP.sequence.status.nextStep)
   END_RUNG
   // the same network as SCL:
   #_w1 := ("Unit1.Em13.ControlNodes".jrUnloadingPnP.sequence.status.currentStep = #JOB_1_STEP_60) AND "Unit1.Em13.ControlNodes".jrUnloadingPnP.sequence.status.seqActive;
   "Unit1.Em13.ControlNodes".jrUnloadingPnP."step".action1[160] := #_w1 AND NOT "Unit1.Em13.ControlNodes".cm.softcam.jrUnIoadingPnPAxisZ.pos00_wait.inPos;
   "Unit1.Em13.ControlNodes".jrUnloadingPnP."step".transition1[160] := #_w1 AND "Unit1.Em13.ControlNodes".cm.softcam.jrUnIoadingPnPAxisZ.pos00_wait.inPos;
   #statTonTime[160].TON(IN := #_w1 AND "Unit1.Em13.ControlNodes".jrUnloadingPnP."step".transition1[160],
                         PT := T#1000ms);
   IF #statTonTime[160].Q THEN
       "Unit1.Em13.ControlNodes".jrUnloadingPnP.sequence.status.nextStep := #JOB_1_STEP_70;
   END_IF;
END_REGION

REGION Network 12: Step[170] : JR Unload P&P C-axis Wait Position
   RUNG wire#powerrail
      { S7_Templates := "SrcType := DInt" } EQ_Contact(in1 := "Unit1.Em13.ControlNodes".jrUnloadingPnP.sequence.status.currentStep, in2 := #JOB_1_STEP_70)
      Contact( "Unit1.Em13.ControlNodes".jrUnloadingPnP.sequence.status.seqActive )
      wire#w1
      I_Contact( "Unit1.Em13.ControlNodes".cm.softcam.jrUnIoadingPnPAxisC.pos00_wait.inPos )
      Coil( "Unit1.Em13.ControlNodes".jrUnloadingPnP."step".action1[170] )
   END_RUNG
   RUNG wire#w1
      Contact( "Unit1.Em13.ControlNodes".cm.softcam.jrUnIoadingPnPAxisC.pos00_wait.inPos )
      Coil( "Unit1.Em13.ControlNodes".jrUnloadingPnP."step".transition1[170] )
   END_RUNG
   RUNG wire#w1
      Contact( "Unit1.Em13.ControlNodes".jrUnloadingPnP."step".transition1[170] )
      { S7_Templates := "time_type := Time" } #statTonTime[170].TON(pt := T#1000ms, et =>)
      Move(in := #JOB_1_STEP_80, out1 => "Unit1.Em13.ControlNodes".jrUnloadingPnP.sequence.status.nextStep)
   END_RUNG
   // the same network as SCL:
   #_w1 := ("Unit1.Em13.ControlNodes".jrUnloadingPnP.sequence.status.currentStep = #JOB_1_STEP_70) AND "Unit1.Em13.ControlNodes".jrUnloadingPnP.sequence.status.seqActive;
   "Unit1.Em13.ControlNodes".jrUnloadingPnP."step".action1[170] := #_w1 AND NOT "Unit1.Em13.ControlNodes".cm.softcam.jrUnIoadingPnPAxisC.pos00_wait.inPos;
   "Unit1.Em13.ControlNodes".jrUnloadingPnP."step".transition1[170] := #_w1 AND "Unit1.Em13.ControlNodes".cm.softcam.jrUnIoadingPnPAxisC.pos00_wait.inPos;
   #statTonTime[170].TON(IN := #_w1 AND "Unit1.Em13.ControlNodes".jrUnloadingPnP."step".transition1[170],
                         PT := T#1000ms);
   IF #statTonTime[170].Q THEN
       "Unit1.Em13.ControlNodes".jrUnloadingPnP.sequence.status.nextStep := #JOB_1_STEP_80;
   END_IF;
END_REGION

REGION Network 13: Step[180] : JR Unload P&P X-axis Wait Position
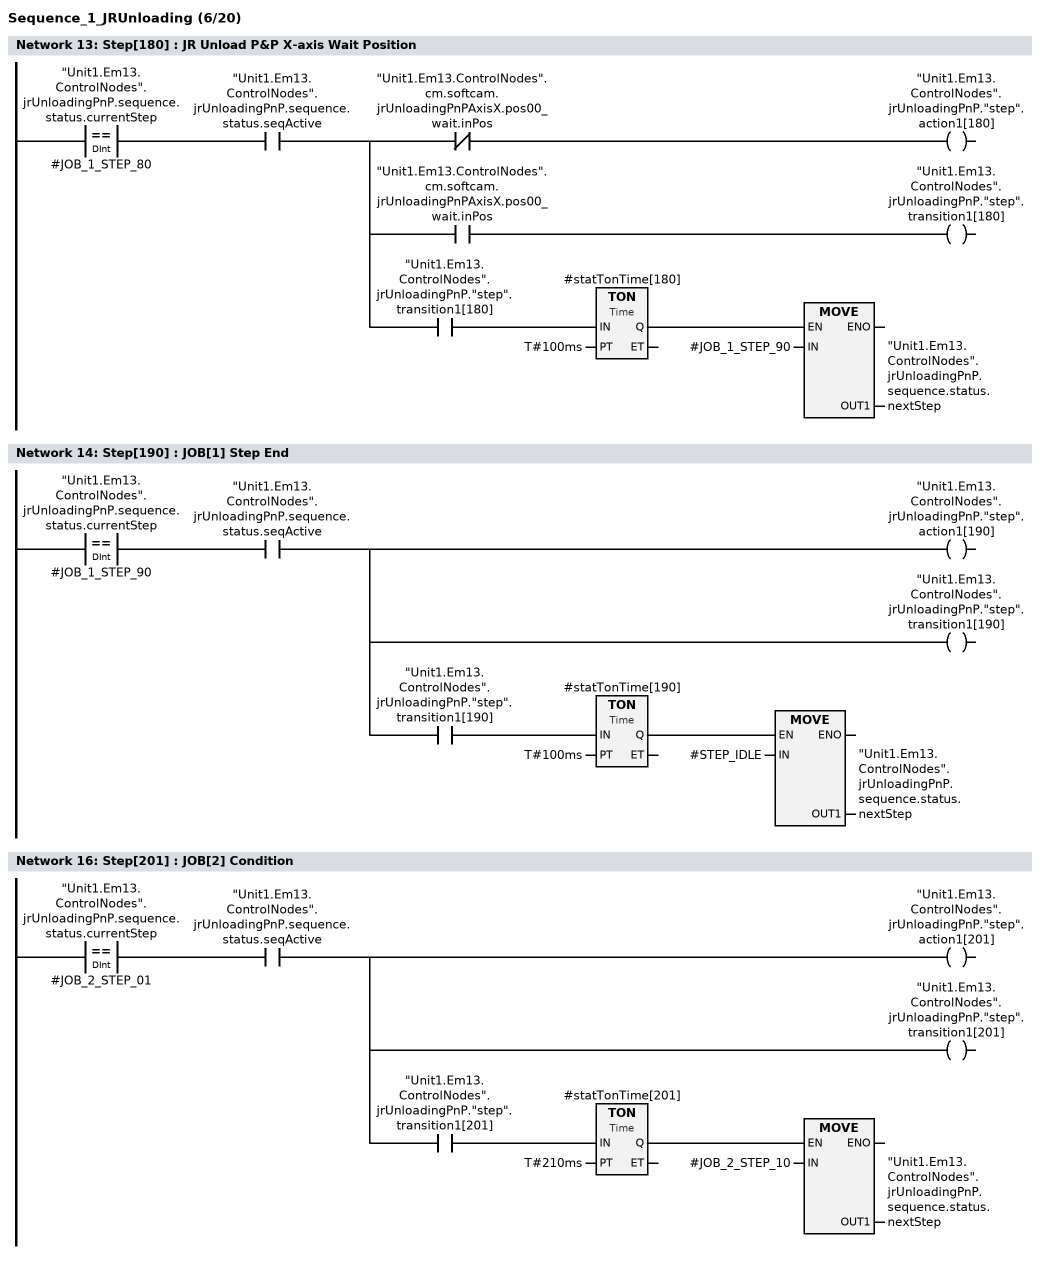
   RUNG wire#powerrail
      { S7_Templates := "SrcType := DInt" } EQ_Contact(in1 := "Unit1.Em13.ControlNodes".jrUnloadingPnP.sequence.status.currentStep, in2 := #JOB_1_STEP_80)
      Contact( "Unit1.Em13.ControlNodes".jrUnloadingPnP.sequence.status.seqActive )
      wire#w1
      I_Contact( "Unit1.Em13.ControlNodes".cm.softcam.jrUnIoadingPnPAxisX.pos00_wait.inPos )
      Coil( "Unit1.Em13.ControlNodes".jrUnloadingPnP."step".action1[180] )
   END_RUNG
   RUNG wire#w1
      Contact( "Unit1.Em13.ControlNodes".cm.softcam.jrUnIoadingPnPAxisX.pos00_wait.inPos )
      Coil( "Unit1.Em13.ControlNodes".jrUnloadingPnP."step".transition1[180] )
   END_RUNG
   RUNG wire#w1
      Contact( "Unit1.Em13.ControlNodes".jrUnloadingPnP."step".transition1[180] )
      { S7_Templates := "time_type := Time" } #statTonTime[180].TON(pt := T#100ms, et =>)
      Move(in := #JOB_1_STEP_90, out1 => "Unit1.Em13.ControlNodes".jrUnloadingPnP.sequence.status.nextStep)
   END_RUNG
   // the same network as SCL:
   #_w1 := ("Unit1.Em13.ControlNodes".jrUnloadingPnP.sequence.status.currentStep = #JOB_1_STEP_80) AND "Unit1.Em13.ControlNodes".jrUnloadingPnP.sequence.status.seqActive;
   "Unit1.Em13.ControlNodes".jrUnloadingPnP."step".action1[180] := #_w1 AND NOT "Unit1.Em13.ControlNodes".cm.softcam.jrUnIoadingPnPAxisX.pos00_wait.inPos;
   "Unit1.Em13.ControlNodes".jrUnloadingPnP."step".transition1[180] := #_w1 AND "Unit1.Em13.ControlNodes".cm.softcam.jrUnIoadingPnPAxisX.pos00_wait.inPos;
   #statTonTime[180].TON(IN := #_w1 AND "Unit1.Em13.ControlNodes".jrUnloadingPnP."step".transition1[180],
                         PT := T#100ms);
   IF #statTonTime[180].Q THEN
       "Unit1.Em13.ControlNodes".jrUnloadingPnP.sequence.status.nextStep := #JOB_1_STEP_90;
   END_IF;
END_REGION

REGION Network 14: Step[190] : JOB[1] Step End
   RUNG wire#powerrail
      { S7_Templates := "SrcType := DInt" } EQ_Contact(in1 := "Unit1.Em13.ControlNodes".jrUnloadingPnP.sequence.status.currentStep, in2 := #JOB_1_STEP_90)
      Contact( "Unit1.Em13.ControlNodes".jrUnloadingPnP.sequence.status.seqActive )
      wire#w1
      Coil( "Unit1.Em13.ControlNodes".jrUnloadingPnP."step".action1[190] )
   END_RUNG
   RUNG wire#w1
      Coil( "Unit1.Em13.ControlNodes".jrUnloadingPnP."step".transition1[190] )
   END_RUNG
   RUNG wire#w1
      Contact( "Unit1.Em13.ControlNodes".jrUnloadingPnP."step".transition1[190] )
      { S7_Templates := "time_type := Time" } #statTonTime[190].TON(pt := T#100ms, et =>)
      Move(in := #STEP_IDLE, out1 => "Unit1.Em13.ControlNodes".jrUnloadingPnP.sequence.status.nextStep)
   END_RUNG
   // the same network as SCL:
   "Unit1.Em13.ControlNodes".jrUnloadingPnP."step".action1[190] := ("Unit1.Em13.ControlNodes".jrUnloadingPnP.sequence.status.currentStep = #JOB_1_STEP_90) AND "Unit1.Em13.ControlNodes".jrUnloadingPnP.sequence.status.seqActive;
   "Unit1.Em13.ControlNodes".jrUnloadingPnP."step".transition1[190] := ("Unit1.Em13.ControlNodes".jrUnloadingPnP.sequence.status.currentStep = #JOB_1_STEP_90) AND "Unit1.Em13.ControlNodes".jrUnloadingPnP.sequence.status.seqActive;
   #statTonTime[190].TON(IN := ("Unit1.Em13.ControlNodes".jrUnloadingPnP.sequence.status.currentStep = #JOB_1_STEP_90) AND "Unit1.Em13.ControlNodes".jrUnloadingPnP.sequence.status.seqActive AND "Unit1.Em13.ControlNodes".jrUnloadingPnP."step".transition1[190],
                         PT := T#100ms);
   IF #statTonTime[190].Q THEN
       "Unit1.Em13.ControlNodes".jrUnloadingPnP.sequence.status.nextStep := #STEP_IDLE;
   END_IF;
END_REGION

REGION Network 15: *************** JOB[2] JR GET=AUTO **********************
END_REGION

REGION Network 16: Step[201] : JOB[2] Condition
   RUNG wire#powerrail
      { S7_Templates := "SrcType := DInt" } EQ_Contact(in1 := "Unit1.Em13.ControlNodes".jrUnloadingPnP.sequence.status.currentStep, in2 := #JOB_2_STEP_01)
      Contact( "Unit1.Em13.ControlNodes".jrUnloadingPnP.sequence.status.seqActive )
      wire#w1
      Coil( "Unit1.Em13.ControlNodes".jrUnloadingPnP."step".action1[201] )
   END_RUNG
   RUNG wire#w1
      Coil( "Unit1.Em13.ControlNodes".jrUnloadingPnP."step".transition1[201] )
   END_RUNG
   RUNG wire#w1
      Contact( "Unit1.Em13.ControlNodes".jrUnloadingPnP."step".transition1[201] )
      { S7_Templates := "time_type := Time" } #statTonTime[201].TON(pt := T#210ms, et =>)
      Move(in := #JOB_2_STEP_10, out1 => "Unit1.Em13.ControlNodes".jrUnloadingPnP.sequence.status.nextStep)
   END_RUNG
   // the same network as SCL:
   "Unit1.Em13.ControlNodes".jrUnloadingPnP."step".action1[201] := ("Unit1.Em13.ControlNodes".jrUnloadingPnP.sequence.status.currentStep = #JOB_2_STEP_01) AND "Unit1.Em13.ControlNodes".jrUnloadingPnP.sequence.status.seqActive;
   "Unit1.Em13.ControlNodes".jrUnloadingPnP."step".transition1[201] := ("Unit1.Em13.ControlNodes".jrUnloadingPnP.sequence.status.currentStep = #JOB_2_STEP_01) AND "Unit1.Em13.ControlNodes".jrUnloadingPnP.sequence.status.seqActive;
   #statTonTime[201].TON(IN := ("Unit1.Em13.ControlNodes".jrUnloadingPnP.sequence.status.currentStep = #JOB_2_STEP_01) AND "Unit1.Em13.ControlNodes".jrUnloadingPnP.sequence.status.seqActive AND "Unit1.Em13.ControlNodes".jrUnloadingPnP."step".transition1[201],
                         PT := T#210ms);
   IF #statTonTime[201].Q THEN
       "Unit1.Em13.ControlNodes".jrUnloadingPnP.sequence.status.nextStep := #JOB_2_STEP_10;
   END_IF;
END_REGION

REGION Network 17: Step[210] : JR Unload P&P X-axis Work Ready Position
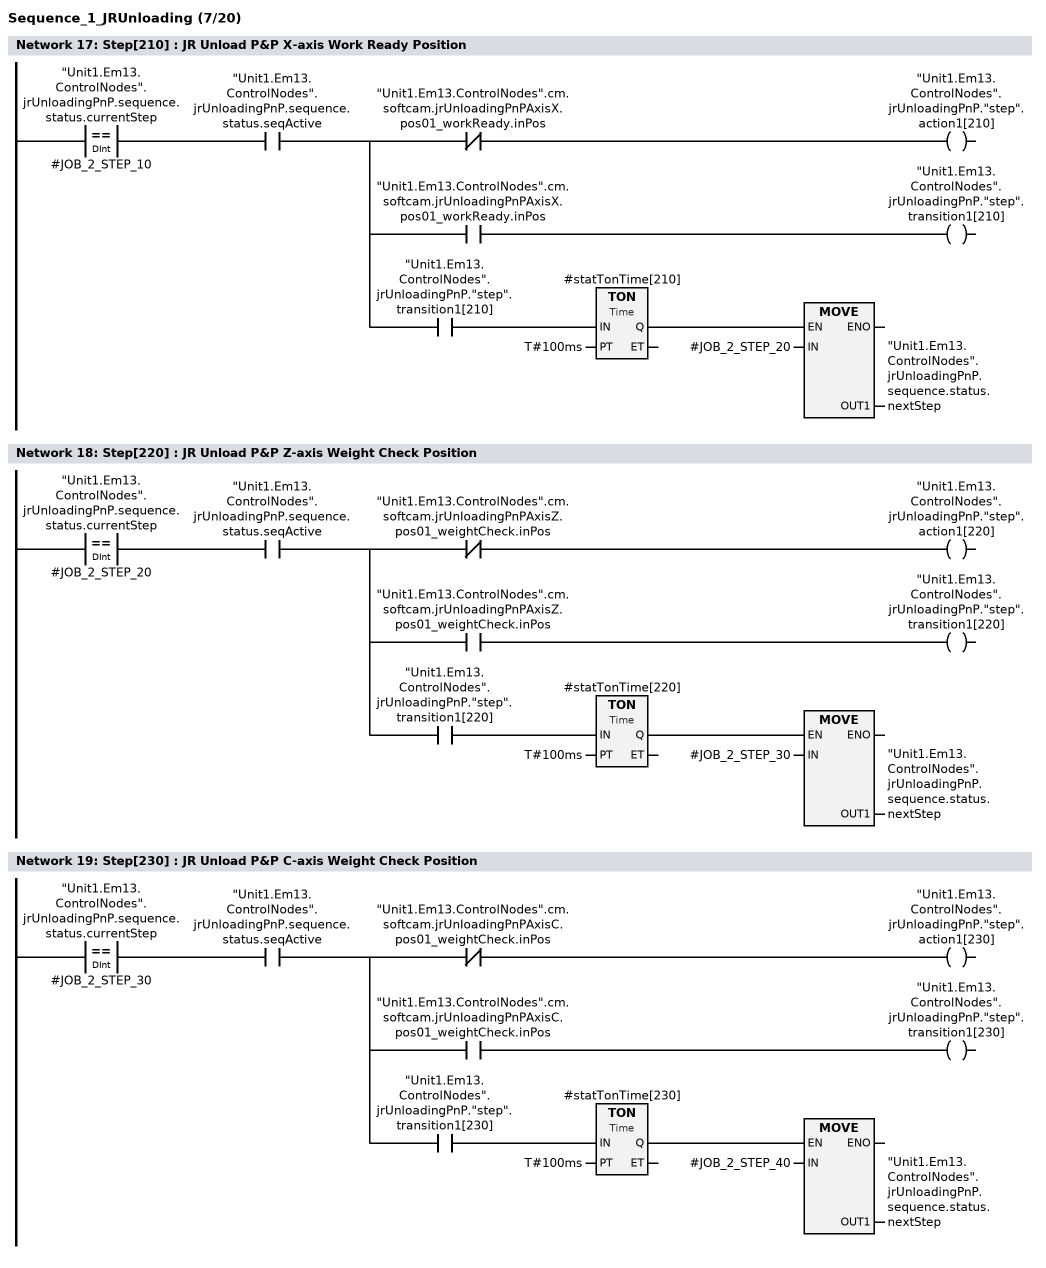
   RUNG wire#powerrail
      { S7_Templates := "SrcType := DInt" } EQ_Contact(in1 := "Unit1.Em13.ControlNodes".jrUnloadingPnP.sequence.status.currentStep, in2 := #JOB_2_STEP_10)
      Contact( "Unit1.Em13.ControlNodes".jrUnloadingPnP.sequence.status.seqActive )
      wire#w1
      I_Contact( "Unit1.Em13.ControlNodes".cm.softcam.jrUnIoadingPnPAxisX.pos01_workReady.inPos )
      Coil( "Unit1.Em13.ControlNodes".jrUnloadingPnP."step".action1[210] )
   END_RUNG
   RUNG wire#w1
      Contact( "Unit1.Em13.ControlNodes".cm.softcam.jrUnIoadingPnPAxisX.pos01_workReady.inPos )
      Coil( "Unit1.Em13.ControlNodes".jrUnloadingPnP."step".transition1[210] )
   END_RUNG
   RUNG wire#w1
      Contact( "Unit1.Em13.ControlNodes".jrUnloadingPnP."step".transition1[210] )
      { S7_Templates := "time_type := Time" } #statTonTime[210].TON(pt := T#100ms, et =>)
      Move(in := #JOB_2_STEP_20, out1 => "Unit1.Em13.ControlNodes".jrUnloadingPnP.sequence.status.nextStep)
   END_RUNG
   // the same network as SCL:
   #_w1 := ("Unit1.Em13.ControlNodes".jrUnloadingPnP.sequence.status.currentStep = #JOB_2_STEP_10) AND "Unit1.Em13.ControlNodes".jrUnloadingPnP.sequence.status.seqActive;
   "Unit1.Em13.ControlNodes".jrUnloadingPnP."step".action1[210] := #_w1 AND NOT "Unit1.Em13.ControlNodes".cm.softcam.jrUnIoadingPnPAxisX.pos01_workReady.inPos;
   "Unit1.Em13.ControlNodes".jrUnloadingPnP."step".transition1[210] := #_w1 AND "Unit1.Em13.ControlNodes".cm.softcam.jrUnIoadingPnPAxisX.pos01_workReady.inPos;
   #statTonTime[210].TON(IN := #_w1 AND "Unit1.Em13.ControlNodes".jrUnloadingPnP."step".transition1[210],
                         PT := T#100ms);
   IF #statTonTime[210].Q THEN
       "Unit1.Em13.ControlNodes".jrUnloadingPnP.sequence.status.nextStep := #JOB_2_STEP_20;
   END_IF;
END_REGION

REGION Network 18: Step[220] : JR Unload P&P Z-axis Weight Check Position
   RUNG wire#powerrail
      { S7_Templates := "SrcType := DInt" } EQ_Contact(in1 := "Unit1.Em13.ControlNodes".jrUnloadingPnP.sequence.status.currentStep, in2 := #JOB_2_STEP_20)
      Contact( "Unit1.Em13.ControlNodes".jrUnloadingPnP.sequence.status.seqActive )
      wire#w1
      I_Contact( "Unit1.Em13.ControlNodes".cm.softcam.jrUnIoadingPnPAxisZ.pos01_weightCheck.inPos )
      Coil( "Unit1.Em13.ControlNodes".jrUnloadingPnP."step".action1[220] )
   END_RUNG
   RUNG wire#w1
      Contact( "Unit1.Em13.ControlNodes".cm.softcam.jrUnIoadingPnPAxisZ.pos01_weightCheck.inPos )
      Coil( "Unit1.Em13.ControlNodes".jrUnloadingPnP."step".transition1[220] )
   END_RUNG
   RUNG wire#w1
      Contact( "Unit1.Em13.ControlNodes".jrUnloadingPnP."step".transition1[220] )
      { S7_Templates := "time_type := Time" } #statTonTime[220].TON(pt := T#100ms, et =>)
      Move(in := #JOB_2_STEP_30, out1 => "Unit1.Em13.ControlNodes".jrUnloadingPnP.sequence.status.nextStep)
   END_RUNG
   // the same network as SCL:
   #_w1 := ("Unit1.Em13.ControlNodes".jrUnloadingPnP.sequence.status.currentStep = #JOB_2_STEP_20) AND "Unit1.Em13.ControlNodes".jrUnloadingPnP.sequence.status.seqActive;
   "Unit1.Em13.ControlNodes".jrUnloadingPnP."step".action1[220] := #_w1 AND NOT "Unit1.Em13.ControlNodes".cm.softcam.jrUnIoadingPnPAxisZ.pos01_weightCheck.inPos;
   "Unit1.Em13.ControlNodes".jrUnloadingPnP."step".transition1[220] := #_w1 AND "Unit1.Em13.ControlNodes".cm.softcam.jrUnIoadingPnPAxisZ.pos01_weightCheck.inPos;
   #statTonTime[220].TON(IN := #_w1 AND "Unit1.Em13.ControlNodes".jrUnloadingPnP."step".transition1[220],
                         PT := T#100ms);
   IF #statTonTime[220].Q THEN
       "Unit1.Em13.ControlNodes".jrUnloadingPnP.sequence.status.nextStep := #JOB_2_STEP_30;
   END_IF;
END_REGION

REGION Network 19: Step[230] : JR Unload P&P C-axis Weight Check Position
   RUNG wire#powerrail
      { S7_Templates := "SrcType := DInt" } EQ_Contact(in1 := "Unit1.Em13.ControlNodes".jrUnloadingPnP.sequence.status.currentStep, in2 := #JOB_2_STEP_30)
      Contact( "Unit1.Em13.ControlNodes".jrUnloadingPnP.sequence.status.seqActive )
      wire#w1
      I_Contact( "Unit1.Em13.ControlNodes".cm.softcam.jrUnIoadingPnPAxisC.pos01_weightCheck.inPos )
      Coil( "Unit1.Em13.ControlNodes".jrUnloadingPnP."step".action1[230] )
   END_RUNG
   RUNG wire#w1
      Contact( "Unit1.Em13.ControlNodes".cm.softcam.jrUnIoadingPnPAxisC.pos01_weightCheck.inPos )
      Coil( "Unit1.Em13.ControlNodes".jrUnloadingPnP."step".transition1[230] )
   END_RUNG
   RUNG wire#w1
      Contact( "Unit1.Em13.ControlNodes".jrUnloadingPnP."step".transition1[230] )
      { S7_Templates := "time_type := Time" } #statTonTime[230].TON(pt := T#100ms, et =>)
      Move(in := #JOB_2_STEP_40, out1 => "Unit1.Em13.ControlNodes".jrUnloadingPnP.sequence.status.nextStep)
   END_RUNG
   // the same network as SCL:
   #_w1 := ("Unit1.Em13.ControlNodes".jrUnloadingPnP.sequence.status.currentStep = #JOB_2_STEP_30) AND "Unit1.Em13.ControlNodes".jrUnloadingPnP.sequence.status.seqActive;
   "Unit1.Em13.ControlNodes".jrUnloadingPnP."step".action1[230] := #_w1 AND NOT "Unit1.Em13.ControlNodes".cm.softcam.jrUnIoadingPnPAxisC.pos01_weightCheck.inPos;
   "Unit1.Em13.ControlNodes".jrUnloadingPnP."step".transition1[230] := #_w1 AND "Unit1.Em13.ControlNodes".cm.softcam.jrUnIoadingPnPAxisC.pos01_weightCheck.inPos;
   #statTonTime[230].TON(IN := #_w1 AND "Unit1.Em13.ControlNodes".jrUnloadingPnP."step".transition1[230],
                         PT := T#100ms);
   IF #statTonTime[230].Q THEN
       "Unit1.Em13.ControlNodes".jrUnloadingPnP.sequence.status.nextStep := #JOB_2_STEP_40;
   END_IF;
END_REGION

REGION Network 20: Step[240] : JR Unload P&P X-axis Weight Check Position
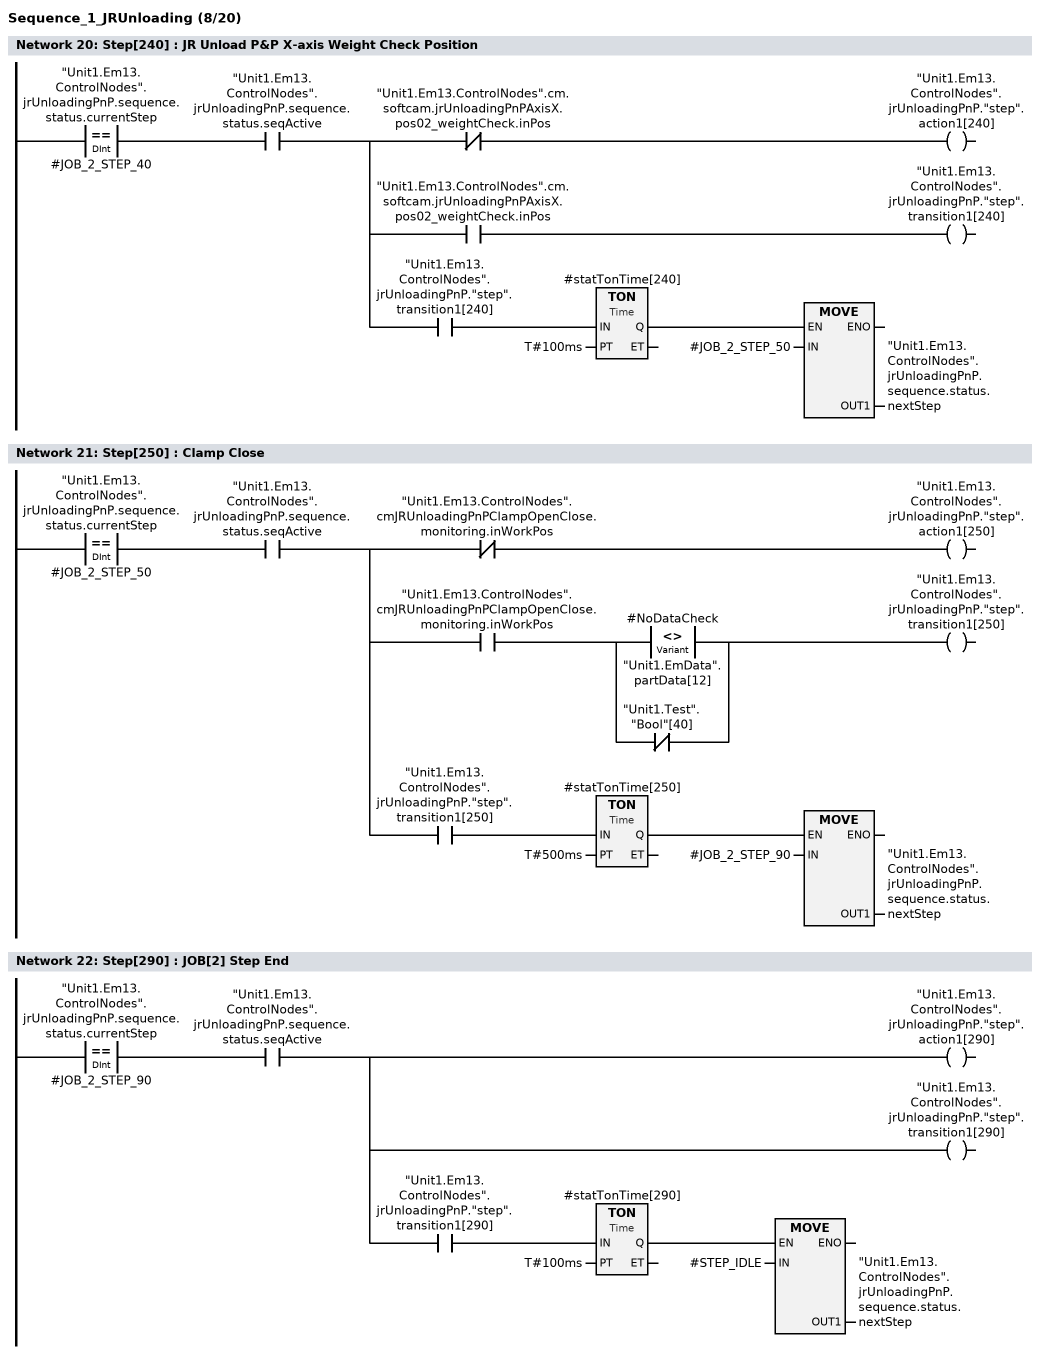
   RUNG wire#powerrail
      { S7_Templates := "SrcType := DInt" } EQ_Contact(in1 := "Unit1.Em13.ControlNodes".jrUnloadingPnP.sequence.status.currentStep, in2 := #JOB_2_STEP_40)
      Contact( "Unit1.Em13.ControlNodes".jrUnloadingPnP.sequence.status.seqActive )
      wire#w1
      I_Contact( "Unit1.Em13.ControlNodes".cm.softcam.jrUnIoadingPnPAxisX.pos02_weightCheck.inPos )
      Coil( "Unit1.Em13.ControlNodes".jrUnloadingPnP."step".action1[240] )
   END_RUNG
   RUNG wire#w1
      Contact( "Unit1.Em13.ControlNodes".cm.softcam.jrUnIoadingPnPAxisX.pos02_weightCheck.inPos )
      Coil( "Unit1.Em13.ControlNodes".jrUnloadingPnP."step".transition1[240] )
   END_RUNG
   RUNG wire#w1
      Contact( "Unit1.Em13.ControlNodes".jrUnloadingPnP."step".transition1[240] )
      { S7_Templates := "time_type := Time" } #statTonTime[240].TON(pt := T#100ms, et =>)
      Move(in := #JOB_2_STEP_50, out1 => "Unit1.Em13.ControlNodes".jrUnloadingPnP.sequence.status.nextStep)
   END_RUNG
   // the same network as SCL:
   #_w1 := ("Unit1.Em13.ControlNodes".jrUnloadingPnP.sequence.status.currentStep = #JOB_2_STEP_40) AND "Unit1.Em13.ControlNodes".jrUnloadingPnP.sequence.status.seqActive;
   "Unit1.Em13.ControlNodes".jrUnloadingPnP."step".action1[240] := #_w1 AND NOT "Unit1.Em13.ControlNodes".cm.softcam.jrUnIoadingPnPAxisX.pos02_weightCheck.inPos;
   "Unit1.Em13.ControlNodes".jrUnloadingPnP."step".transition1[240] := #_w1 AND "Unit1.Em13.ControlNodes".cm.softcam.jrUnIoadingPnPAxisX.pos02_weightCheck.inPos;
   #statTonTime[240].TON(IN := #_w1 AND "Unit1.Em13.ControlNodes".jrUnloadingPnP."step".transition1[240],
                         PT := T#100ms);
   IF #statTonTime[240].Q THEN
       "Unit1.Em13.ControlNodes".jrUnloadingPnP.sequence.status.nextStep := #JOB_2_STEP_50;
   END_IF;
END_REGION

REGION Network 21: Step[250] : Clamp Close
   RUNG wire#powerrail
      { S7_Templates := "SrcType := DInt" } EQ_Contact(in1 := "Unit1.Em13.ControlNodes".jrUnloadingPnP.sequence.status.currentStep, in2 := #JOB_2_STEP_50)
      Contact( "Unit1.Em13.ControlNodes".jrUnloadingPnP.sequence.status.seqActive )
      wire#w1
      I_Contact( "Unit1.Em13.ControlNodes".cmJRUnloadingPnPClampOpenClose.monitoring.inWorkPos )
      Coil( "Unit1.Em13.ControlNodes".jrUnloadingPnP."step".action1[250] )
   END_RUNG
   RUNG wire#w1
      Contact( "Unit1.Em13.ControlNodes".cmJRUnloadingPnPClampOpenClose.monitoring.inWorkPos )
      wire#w2
      { S7_Templates := "SrcType := Variant" } NE_Contact(in1 := #NoDataCheck, in2 := "Unit1.EmData".partData[12])
      wire#w3
      Coil( "Unit1.Em13.ControlNodes".jrUnloadingPnP."step".transition1[250] )
   END_RUNG
   RUNG wire#w2
      I_Contact( "Unit1.Test"."Bool"[40] )
   END_RUNG wire#w3
   RUNG wire#w1
      Contact( "Unit1.Em13.ControlNodes".jrUnloadingPnP."step".transition1[250] )
      { S7_Templates := "time_type := Time" } #statTonTime[250].TON(pt := T#500ms, et =>)
      Move(in := #JOB_2_STEP_90, out1 => "Unit1.Em13.ControlNodes".jrUnloadingPnP.sequence.status.nextStep)
   END_RUNG
   // the same network as SCL:
   #_w1 := ("Unit1.Em13.ControlNodes".jrUnloadingPnP.sequence.status.currentStep = #JOB_2_STEP_50) AND "Unit1.Em13.ControlNodes".jrUnloadingPnP.sequence.status.seqActive;
   "Unit1.Em13.ControlNodes".jrUnloadingPnP."step".action1[250] := #_w1 AND NOT "Unit1.Em13.ControlNodes".cmJRUnloadingPnPClampOpenClose.monitoring.inWorkPos;
   "Unit1.Em13.ControlNodes".jrUnloadingPnP."step".transition1[250] := #_w1 AND "Unit1.Em13.ControlNodes".cmJRUnloadingPnPClampOpenClose.monitoring.inWorkPos AND ((#NoDataCheck <> "Unit1.EmData".partData[12]) OR NOT "Unit1.Test"."Bool"[40]);
   #statTonTime[250].TON(IN := #_w1 AND "Unit1.Em13.ControlNodes".jrUnloadingPnP."step".transition1[250],
                         PT := T#500ms);
   IF #statTonTime[250].Q THEN
       "Unit1.Em13.ControlNodes".jrUnloadingPnP.sequence.status.nextStep := #JOB_2_STEP_90;
   END_IF;
END_REGION

REGION Network 22: Step[290] : JOB[2] Step End
   RUNG wire#powerrail
      { S7_Templates := "SrcType := DInt" } EQ_Contact(in1 := "Unit1.Em13.ControlNodes".jrUnloadingPnP.sequence.status.currentStep, in2 := #JOB_2_STEP_90)
      Contact( "Unit1.Em13.ControlNodes".jrUnloadingPnP.sequence.status.seqActive )
      wire#w1
      Coil( "Unit1.Em13.ControlNodes".jrUnloadingPnP."step".action1[290] )
   END_RUNG
   RUNG wire#w1
      Coil( "Unit1.Em13.ControlNodes".jrUnloadingPnP."step".transition1[290] )
   END_RUNG
   RUNG wire#w1
      Contact( "Unit1.Em13.ControlNodes".jrUnloadingPnP."step".transition1[290] )
      { S7_Templates := "time_type := Time" } #statTonTime[290].TON(pt := T#100ms, et =>)
      Move(in := #STEP_IDLE, out1 => "Unit1.Em13.ControlNodes".jrUnloadingPnP.sequence.status.nextStep)
   END_RUNG
   // the same network as SCL:
   "Unit1.Em13.ControlNodes".jrUnloadingPnP."step".action1[290] := ("Unit1.Em13.ControlNodes".jrUnloadingPnP.sequence.status.currentStep = #JOB_2_STEP_90) AND "Unit1.Em13.ControlNodes".jrUnloadingPnP.sequence.status.seqActive;
   "Unit1.Em13.ControlNodes".jrUnloadingPnP."step".transition1[290] := ("Unit1.Em13.ControlNodes".jrUnloadingPnP.sequence.status.currentStep = #JOB_2_STEP_90) AND "Unit1.Em13.ControlNodes".jrUnloadingPnP.sequence.status.seqActive;
   #statTonTime[290].TON(IN := ("Unit1.Em13.ControlNodes".jrUnloadingPnP.sequence.status.currentStep = #JOB_2_STEP_90) AND "Unit1.Em13.ControlNodes".jrUnloadingPnP.sequence.status.seqActive AND "Unit1.Em13.ControlNodes".jrUnloadingPnP."step".transition1[290],
                         PT := T#100ms);
   IF #statTonTime[290].Q THEN
       "Unit1.Em13.ControlNodes".jrUnloadingPnP.sequence.status.nextStep := #STEP_IDLE;
   END_IF;
END_REGION

REGION Network 23: ************* JOB[3] CONVEYOR A JR PUT=AUTO ***************
END_REGION

REGION Network 24: Step[301] : JOB[3] Condition
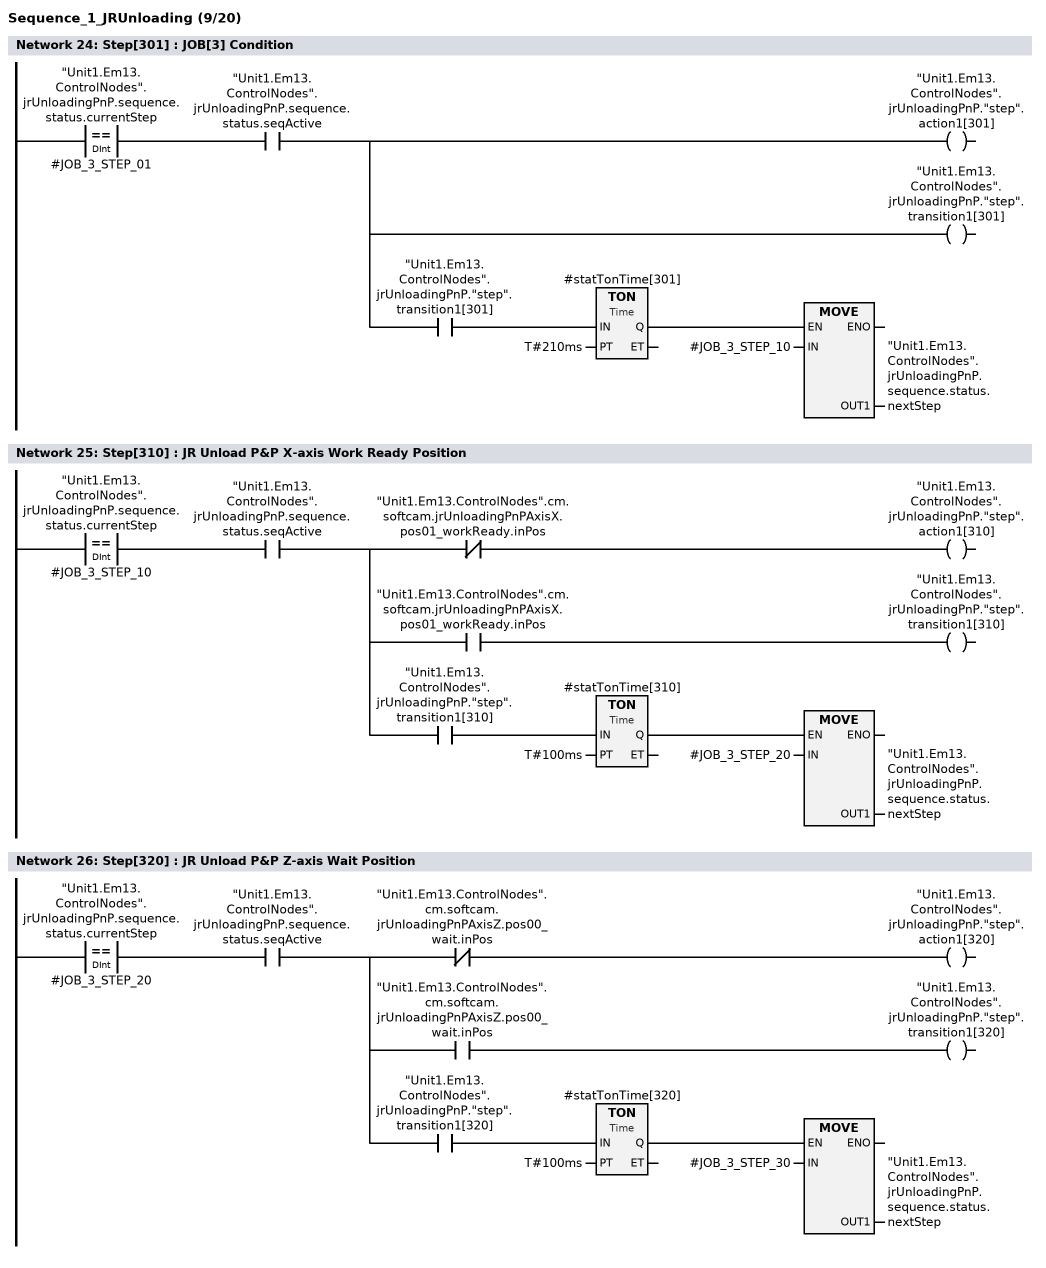
   RUNG wire#powerrail
      { S7_Templates := "SrcType := DInt" } EQ_Contact(in1 := "Unit1.Em13.ControlNodes".jrUnloadingPnP.sequence.status.currentStep, in2 := #JOB_3_STEP_01)
      Contact( "Unit1.Em13.ControlNodes".jrUnloadingPnP.sequence.status.seqActive )
      wire#w1
      Coil( "Unit1.Em13.ControlNodes".jrUnloadingPnP."step".action1[301] )
   END_RUNG
   RUNG wire#w1
      Coil( "Unit1.Em13.ControlNodes".jrUnloadingPnP."step".transition1[301] )
   END_RUNG
   RUNG wire#w1
      Contact( "Unit1.Em13.ControlNodes".jrUnloadingPnP."step".transition1[301] )
      { S7_Templates := "time_type := Time" } #statTonTime[301].TON(pt := T#210ms, et =>)
      Move(in := #JOB_3_STEP_10, out1 => "Unit1.Em13.ControlNodes".jrUnloadingPnP.sequence.status.nextStep)
   END_RUNG
   // the same network as SCL:
   "Unit1.Em13.ControlNodes".jrUnloadingPnP."step".action1[301] := ("Unit1.Em13.ControlNodes".jrUnloadingPnP.sequence.status.currentStep = #JOB_3_STEP_01) AND "Unit1.Em13.ControlNodes".jrUnloadingPnP.sequence.status.seqActive;
   "Unit1.Em13.ControlNodes".jrUnloadingPnP."step".transition1[301] := ("Unit1.Em13.ControlNodes".jrUnloadingPnP.sequence.status.currentStep = #JOB_3_STEP_01) AND "Unit1.Em13.ControlNodes".jrUnloadingPnP.sequence.status.seqActive;
   #statTonTime[301].TON(IN := ("Unit1.Em13.ControlNodes".jrUnloadingPnP.sequence.status.currentStep = #JOB_3_STEP_01) AND "Unit1.Em13.ControlNodes".jrUnloadingPnP.sequence.status.seqActive AND "Unit1.Em13.ControlNodes".jrUnloadingPnP."step".transition1[301],
                         PT := T#210ms);
   IF #statTonTime[301].Q THEN
       "Unit1.Em13.ControlNodes".jrUnloadingPnP.sequence.status.nextStep := #JOB_3_STEP_10;
   END_IF;
END_REGION

REGION Network 25: Step[310] : JR Unload P&P X-axis Work Ready Position
   RUNG wire#powerrail
      { S7_Templates := "SrcType := DInt" } EQ_Contact(in1 := "Unit1.Em13.ControlNodes".jrUnloadingPnP.sequence.status.currentStep, in2 := #JOB_3_STEP_10)
      Contact( "Unit1.Em13.ControlNodes".jrUnloadingPnP.sequence.status.seqActive )
      wire#w1
      I_Contact( "Unit1.Em13.ControlNodes".cm.softcam.jrUnIoadingPnPAxisX.pos01_workReady.inPos )
      Coil( "Unit1.Em13.ControlNodes".jrUnloadingPnP."step".action1[310] )
   END_RUNG
   RUNG wire#w1
      Contact( "Unit1.Em13.ControlNodes".cm.softcam.jrUnIoadingPnPAxisX.pos01_workReady.inPos )
      Coil( "Unit1.Em13.ControlNodes".jrUnloadingPnP."step".transition1[310] )
   END_RUNG
   RUNG wire#w1
      Contact( "Unit1.Em13.ControlNodes".jrUnloadingPnP."step".transition1[310] )
      { S7_Templates := "time_type := Time" } #statTonTime[310].TON(pt := T#100ms, et =>)
      Move(in := #JOB_3_STEP_20, out1 => "Unit1.Em13.ControlNodes".jrUnloadingPnP.sequence.status.nextStep)
   END_RUNG
   // the same network as SCL:
   #_w1 := ("Unit1.Em13.ControlNodes".jrUnloadingPnP.sequence.status.currentStep = #JOB_3_STEP_10) AND "Unit1.Em13.ControlNodes".jrUnloadingPnP.sequence.status.seqActive;
   "Unit1.Em13.ControlNodes".jrUnloadingPnP."step".action1[310] := #_w1 AND NOT "Unit1.Em13.ControlNodes".cm.softcam.jrUnIoadingPnPAxisX.pos01_workReady.inPos;
   "Unit1.Em13.ControlNodes".jrUnloadingPnP."step".transition1[310] := #_w1 AND "Unit1.Em13.ControlNodes".cm.softcam.jrUnIoadingPnPAxisX.pos01_workReady.inPos;
   #statTonTime[310].TON(IN := #_w1 AND "Unit1.Em13.ControlNodes".jrUnloadingPnP."step".transition1[310],
                         PT := T#100ms);
   IF #statTonTime[310].Q THEN
       "Unit1.Em13.ControlNodes".jrUnloadingPnP.sequence.status.nextStep := #JOB_3_STEP_20;
   END_IF;
END_REGION

REGION Network 26: Step[320] : JR Unload P&P Z-axis Wait Position
   RUNG wire#powerrail
      { S7_Templates := "SrcType := DInt" } EQ_Contact(in1 := "Unit1.Em13.ControlNodes".jrUnloadingPnP.sequence.status.currentStep, in2 := #JOB_3_STEP_20)
      Contact( "Unit1.Em13.ControlNodes".jrUnloadingPnP.sequence.status.seqActive )
      wire#w1
      I_Contact( "Unit1.Em13.ControlNodes".cm.softcam.jrUnIoadingPnPAxisZ.pos00_wait.inPos )
      Coil( "Unit1.Em13.ControlNodes".jrUnloadingPnP."step".action1[320] )
   END_RUNG
   RUNG wire#w1
      Contact( "Unit1.Em13.ControlNodes".cm.softcam.jrUnIoadingPnPAxisZ.pos00_wait.inPos )
      Coil( "Unit1.Em13.ControlNodes".jrUnloadingPnP."step".transition1[320] )
   END_RUNG
   RUNG wire#w1
      Contact( "Unit1.Em13.ControlNodes".jrUnloadingPnP."step".transition1[320] )
      { S7_Templates := "time_type := Time" } #statTonTime[320].TON(pt := T#100ms, et =>)
      Move(in := #JOB_3_STEP_30, out1 => "Unit1.Em13.ControlNodes".jrUnloadingPnP.sequence.status.nextStep)
   END_RUNG
   // the same network as SCL:
   #_w1 := ("Unit1.Em13.ControlNodes".jrUnloadingPnP.sequence.status.currentStep = #JOB_3_STEP_20) AND "Unit1.Em13.ControlNodes".jrUnloadingPnP.sequence.status.seqActive;
   "Unit1.Em13.ControlNodes".jrUnloadingPnP."step".action1[320] := #_w1 AND NOT "Unit1.Em13.ControlNodes".cm.softcam.jrUnIoadingPnPAxisZ.pos00_wait.inPos;
   "Unit1.Em13.ControlNodes".jrUnloadingPnP."step".transition1[320] := #_w1 AND "Unit1.Em13.ControlNodes".cm.softcam.jrUnIoadingPnPAxisZ.pos00_wait.inPos;
   #statTonTime[320].TON(IN := #_w1 AND "Unit1.Em13.ControlNodes".jrUnloadingPnP."step".transition1[320],
                         PT := T#100ms);
   IF #statTonTime[320].Q THEN
       "Unit1.Em13.ControlNodes".jrUnloadingPnP.sequence.status.nextStep := #JOB_3_STEP_30;
   END_IF;
END_REGION

REGION Network 27: Step[330] : JR Unload P&P X-axis Wait Position
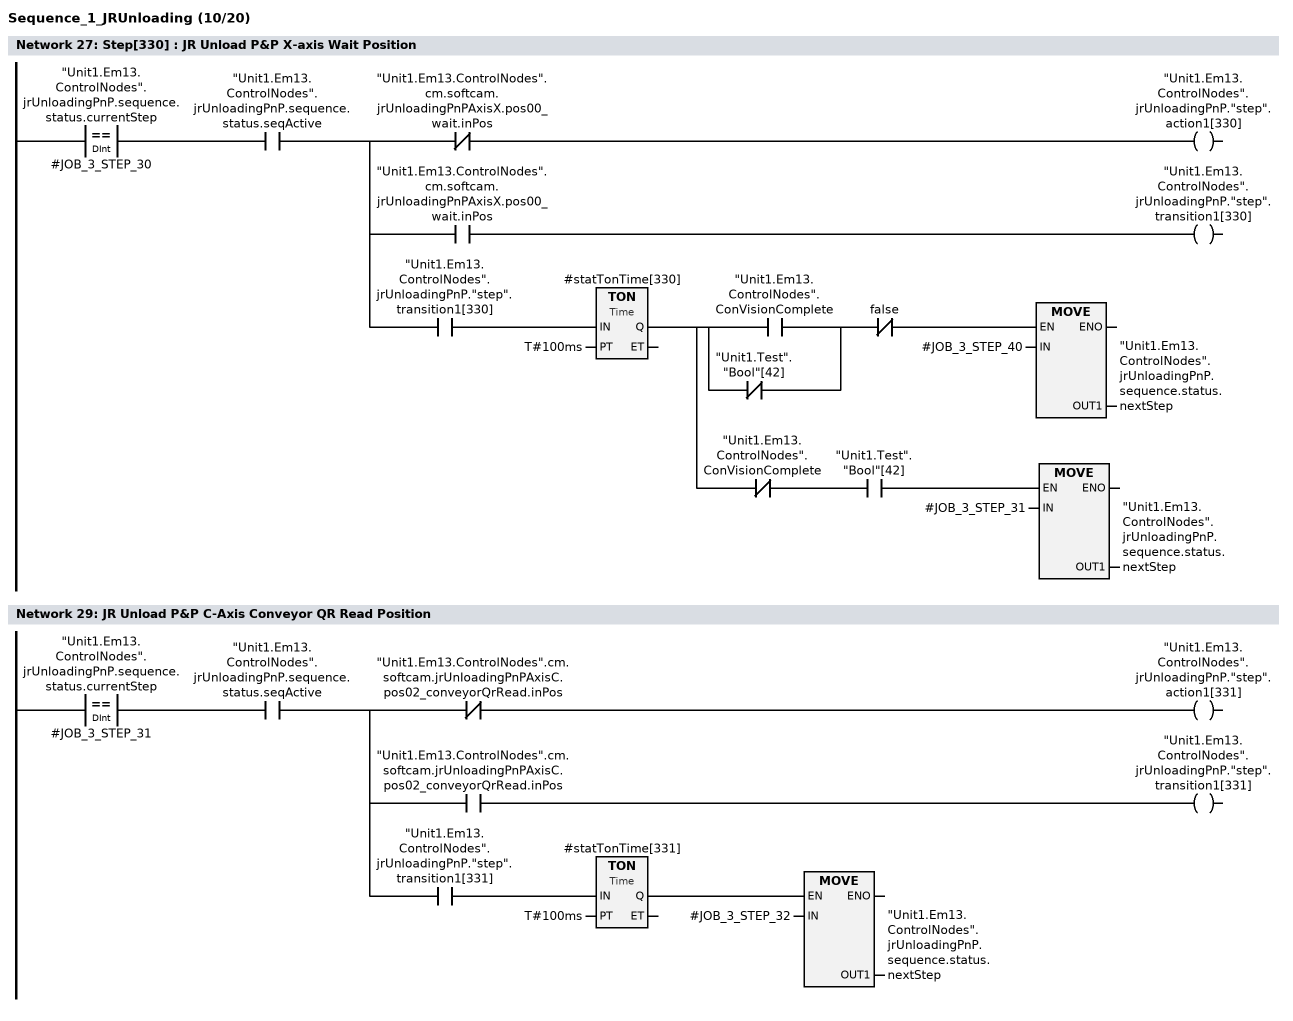
   RUNG wire#powerrail
      { S7_Templates := "SrcType := DInt" } EQ_Contact(in1 := "Unit1.Em13.ControlNodes".jrUnloadingPnP.sequence.status.currentStep, in2 := #JOB_3_STEP_30)
      Contact( "Unit1.Em13.ControlNodes".jrUnloadingPnP.sequence.status.seqActive )
      wire#w1
      I_Contact( "Unit1.Em13.ControlNodes".cm.softcam.jrUnIoadingPnPAxisX.pos00_wait.inPos )
      Coil( "Unit1.Em13.ControlNodes".jrUnloadingPnP."step".action1[330] )
   END_RUNG
   RUNG wire#w1
      Contact( "Unit1.Em13.ControlNodes".cm.softcam.jrUnIoadingPnPAxisX.pos00_wait.inPos )
      Coil( "Unit1.Em13.ControlNodes".jrUnloadingPnP."step".transition1[330] )
   END_RUNG
   RUNG wire#w1
      Contact( "Unit1.Em13.ControlNodes".jrUnloadingPnP."step".transition1[330] )
      { S7_Templates := "time_type := Time" } #statTonTime[330].TON(pt := T#100ms, et =>)
      wire#w2
      Contact( "Unit1.Em13.ControlNodes".ConVisionComplete )
      wire#w3
      I_Contact( false )
      Move(in := #JOB_3_STEP_40, out1 => "Unit1.Em13.ControlNodes".jrUnloadingPnP.sequence.status.nextStep)
   END_RUNG
   RUNG wire#w2
      I_Contact( "Unit1.Test"."Bool"[42] )
   END_RUNG wire#w3
   RUNG wire#w2
      I_Contact( "Unit1.Em13.ControlNodes".ConVisionComplete )
      Contact( "Unit1.Test"."Bool"[42] )
      Move(in := #JOB_3_STEP_31, out1 => "Unit1.Em13.ControlNodes".jrUnloadingPnP.sequence.status.nextStep)
   END_RUNG
   // the same network as SCL:
   #_w1 := ("Unit1.Em13.ControlNodes".jrUnloadingPnP.sequence.status.currentStep = #JOB_3_STEP_30) AND "Unit1.Em13.ControlNodes".jrUnloadingPnP.sequence.status.seqActive;
   "Unit1.Em13.ControlNodes".jrUnloadingPnP."step".action1[330] := #_w1 AND NOT "Unit1.Em13.ControlNodes".cm.softcam.jrUnIoadingPnPAxisX.pos00_wait.inPos;
   "Unit1.Em13.ControlNodes".jrUnloadingPnP."step".transition1[330] := #_w1 AND "Unit1.Em13.ControlNodes".cm.softcam.jrUnIoadingPnPAxisX.pos00_wait.inPos;
   #statTonTime[330].TON(IN := #_w1 AND "Unit1.Em13.ControlNodes".jrUnloadingPnP."step".transition1[330],
                         PT := T#100ms);
   IF #statTonTime[330].Q AND ("Unit1.Em13.ControlNodes".ConVisionComplete OR NOT "Unit1.Test"."Bool"[42]) AND NOT false THEN
       "Unit1.Em13.ControlNodes".jrUnloadingPnP.sequence.status.nextStep := #JOB_3_STEP_40;
   END_IF;
   IF #statTonTime[330].Q AND NOT "Unit1.Em13.ControlNodes".ConVisionComplete AND "Unit1.Test"."Bool"[42] THEN
       "Unit1.Em13.ControlNodes".jrUnloadingPnP.sequence.status.nextStep := #JOB_3_STEP_31;
   END_IF;
END_REGION

REGION Network 28: ==================== Template ====================
END_REGION

REGION Network 29: JR Unload P&P C-Axis Conveyor QR Read Position
   RUNG wire#powerrail
      { S7_Templates := "SrcType := DInt" } EQ_Contact(in1 := "Unit1.Em13.ControlNodes".jrUnloadingPnP.sequence.status.currentStep, in2 := #JOB_3_STEP_31)
      Contact( "Unit1.Em13.ControlNodes".jrUnloadingPnP.sequence.status.seqActive )
      wire#w1
      I_Contact( "Unit1.Em13.ControlNodes".cm.softcam.jrUnIoadingPnPAxisC.pos02_conveyorQrRead.inPos )
      Coil( "Unit1.Em13.ControlNodes".jrUnloadingPnP."step".action1[331] )
   END_RUNG
   RUNG wire#w1
      Contact( "Unit1.Em13.ControlNodes".cm.softcam.jrUnIoadingPnPAxisC.pos02_conveyorQrRead.inPos )
      Coil( "Unit1.Em13.ControlNodes".jrUnloadingPnP."step".transition1[331] )
   END_RUNG
   RUNG wire#w1
      Contact( "Unit1.Em13.ControlNodes".jrUnloadingPnP."step".transition1[331] )
      { S7_Templates := "time_type := Time" } #statTonTime[331].TON(pt := T#100ms, et =>)
      Move(in := #JOB_3_STEP_32, out1 => "Unit1.Em13.ControlNodes".jrUnloadingPnP.sequence.status.nextStep)
   END_RUNG
   // the same network as SCL:
   #_w1 := ("Unit1.Em13.ControlNodes".jrUnloadingPnP.sequence.status.currentStep = #JOB_3_STEP_31) AND "Unit1.Em13.ControlNodes".jrUnloadingPnP.sequence.status.seqActive;
   "Unit1.Em13.ControlNodes".jrUnloadingPnP."step".action1[331] := #_w1 AND NOT "Unit1.Em13.ControlNodes".cm.softcam.jrUnIoadingPnPAxisC.pos02_conveyorQrRead.inPos;
   "Unit1.Em13.ControlNodes".jrUnloadingPnP."step".transition1[331] := #_w1 AND "Unit1.Em13.ControlNodes".cm.softcam.jrUnIoadingPnPAxisC.pos02_conveyorQrRead.inPos;
   #statTonTime[331].TON(IN := #_w1 AND "Unit1.Em13.ControlNodes".jrUnloadingPnP."step".transition1[331],
                         PT := T#100ms);
   IF #statTonTime[331].Q THEN
       "Unit1.Em13.ControlNodes".jrUnloadingPnP.sequence.status.nextStep := #JOB_3_STEP_32;
   END_IF;
END_REGION

REGION Network 30: JR Unload P&P Z or X-Axis Conveyor QR Read Position
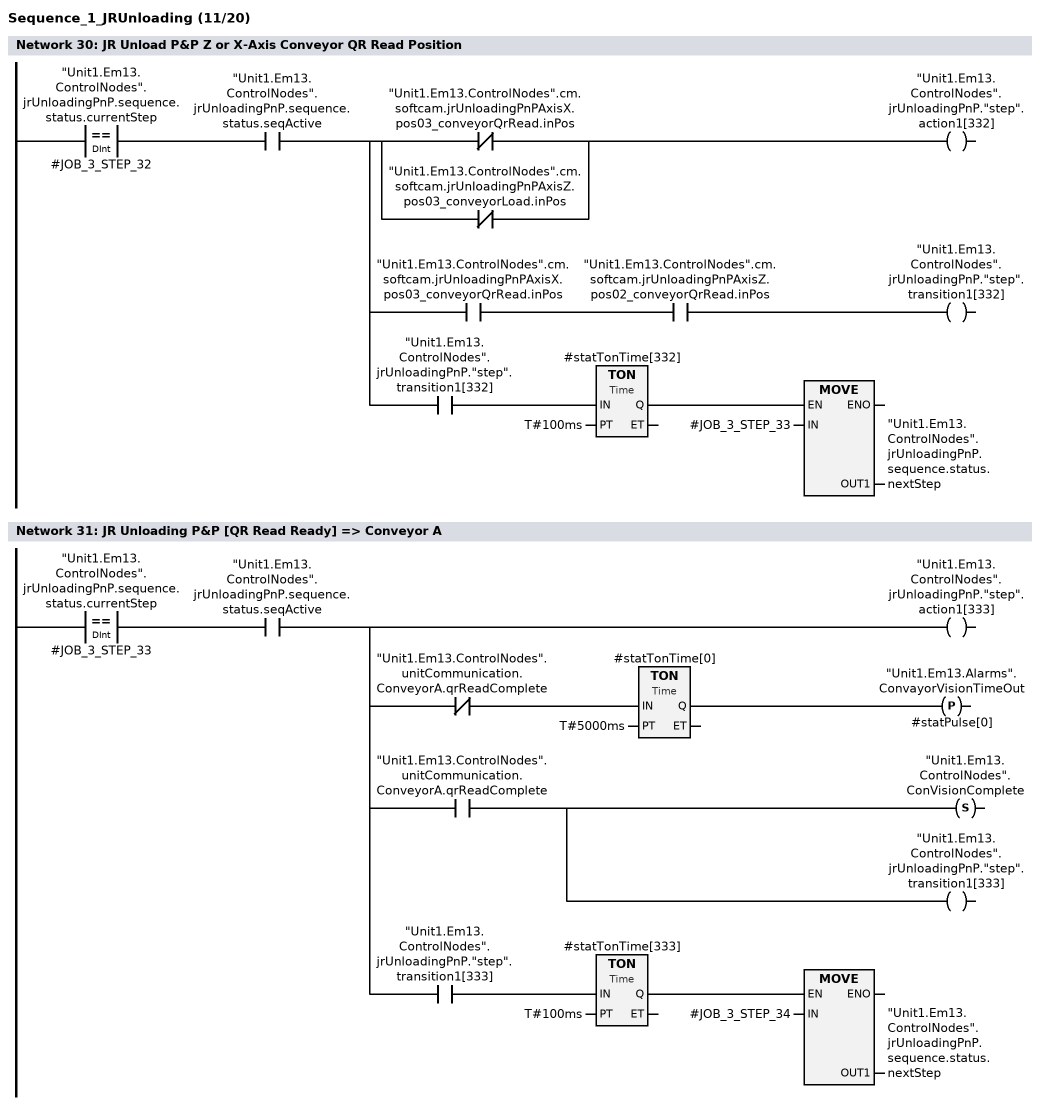
   RUNG wire#powerrail
      { S7_Templates := "SrcType := DInt" } EQ_Contact(in1 := "Unit1.Em13.ControlNodes".jrUnloadingPnP.sequence.status.currentStep, in2 := #JOB_3_STEP_32)
      Contact( "Unit1.Em13.ControlNodes".jrUnloadingPnP.sequence.status.seqActive )
      wire#w1
      I_Contact( "Unit1.Em13.ControlNodes".cm.softcam.jrUnIoadingPnPAxisX.pos03_conveyorQrRead.inPos )
      wire#w2
      Coil( "Unit1.Em13.ControlNodes".jrUnloadingPnP."step".action1[332] )
   END_RUNG
   RUNG wire#w1
      I_Contact( "Unit1.Em13.ControlNodes".cm.softcam.jrUnIoadingPnPAxisZ.pos03_conveyorLoad.inPos )
   END_RUNG wire#w2
   RUNG wire#w1
      Contact( "Unit1.Em13.ControlNodes".cm.softcam.jrUnIoadingPnPAxisX.pos03_conveyorQrRead.inPos )
      Contact( "Unit1.Em13.ControlNodes".cm.softcam.jrUnIoadingPnPAxisZ.pos02_conveyorQrRead.inPos )
      Coil( "Unit1.Em13.ControlNodes".jrUnloadingPnP."step".transition1[332] )
   END_RUNG
   RUNG wire#w1
      Contact( "Unit1.Em13.ControlNodes".jrUnloadingPnP."step".transition1[332] )
      { S7_Templates := "time_type := Time" } #statTonTime[332].TON(pt := T#100ms, et =>)
      Move(in := #JOB_3_STEP_33, out1 => "Unit1.Em13.ControlNodes".jrUnloadingPnP.sequence.status.nextStep)
   END_RUNG
   // the same network as SCL:
   #_w1 := ("Unit1.Em13.ControlNodes".jrUnloadingPnP.sequence.status.currentStep = #JOB_3_STEP_32) AND "Unit1.Em13.ControlNodes".jrUnloadingPnP.sequence.status.seqActive;
   "Unit1.Em13.ControlNodes".jrUnloadingPnP."step".action1[332] := #_w1 AND (NOT "Unit1.Em13.ControlNodes".cm.softcam.jrUnIoadingPnPAxisX.pos03_conveyorQrRead.inPos OR NOT "Unit1.Em13.ControlNodes".cm.softcam.jrUnIoadingPnPAxisZ.pos03_conveyorLoad.inPos);
   "Unit1.Em13.ControlNodes".jrUnloadingPnP."step".transition1[332] := #_w1 AND "Unit1.Em13.ControlNodes".cm.softcam.jrUnIoadingPnPAxisX.pos03_conveyorQrRead.inPos AND "Unit1.Em13.ControlNodes".cm.softcam.jrUnIoadingPnPAxisZ.pos02_conveyorQrRead.inPos;
   #statTonTime[332].TON(IN := #_w1 AND "Unit1.Em13.ControlNodes".jrUnloadingPnP."step".transition1[332],
                         PT := T#100ms);
   IF #statTonTime[332].Q THEN
       "Unit1.Em13.ControlNodes".jrUnloadingPnP.sequence.status.nextStep := #JOB_3_STEP_33;
   END_IF;
END_REGION

REGION Network 31: JR Unloading P&P [QR Read Ready] => Conveyor A
   "Unit1.Em13.ControlNodes".jrUnloadingPnP."step".action1[333] := ("Unit1.Em13.ControlNodes".jrUnloadingPnP.sequence.status.currentStep = #JOB_3_STEP_33) AND "Unit1.Em13.ControlNodes".jrUnloadingPnP.sequence.status.seqActive;
   #statTonTime[0].TON(IN := ("Unit1.Em13.ControlNodes".jrUnloadingPnP.sequence.status.currentStep = #JOB_3_STEP_33) AND "Unit1.Em13.ControlNodes".jrUnloadingPnP.sequence.status.seqActive AND NOT "Unit1.Em13.ControlNodes".unitCommunication.ConveyorA.qrReadComplete,
                       PT := T#5000ms);
   "Unit1.Em13.Alarms".ConvayorVisionTimeOut := #statTonTime[0].Q AND NOT #statPulse[0];   // rising edge
   #statPulse[0] := #statTonTime[0].Q;
   #_w1 := ("Unit1.Em13.ControlNodes".jrUnloadingPnP.sequence.status.currentStep = #JOB_3_STEP_33) AND "Unit1.Em13.ControlNodes".jrUnloadingPnP.sequence.status.seqActive AND "Unit1.Em13.ControlNodes".unitCommunication.ConveyorA.qrReadComplete;
   IF #_w1 THEN "Unit1.Em13.ControlNodes".ConVisionComplete := TRUE; END_IF;
   "Unit1.Em13.ControlNodes".jrUnloadingPnP."step".transition1[333] := #_w1;
   #statTonTime[333].TON(IN := ("Unit1.Em13.ControlNodes".jrUnloadingPnP.sequence.status.currentStep = #JOB_3_STEP_33) AND "Unit1.Em13.ControlNodes".jrUnloadingPnP.sequence.status.seqActive AND "Unit1.Em13.ControlNodes".jrUnloadingPnP."step".transition1[333],
                         PT := T#100ms);
   IF #statTonTime[333].Q THEN
       "Unit1.Em13.ControlNodes".jrUnloadingPnP.sequence.status.nextStep := #JOB_3_STEP_34;
   END_IF;
END_REGION

REGION Network 32: JR Unloading P&P [Loading Ready] <= Conveyor A
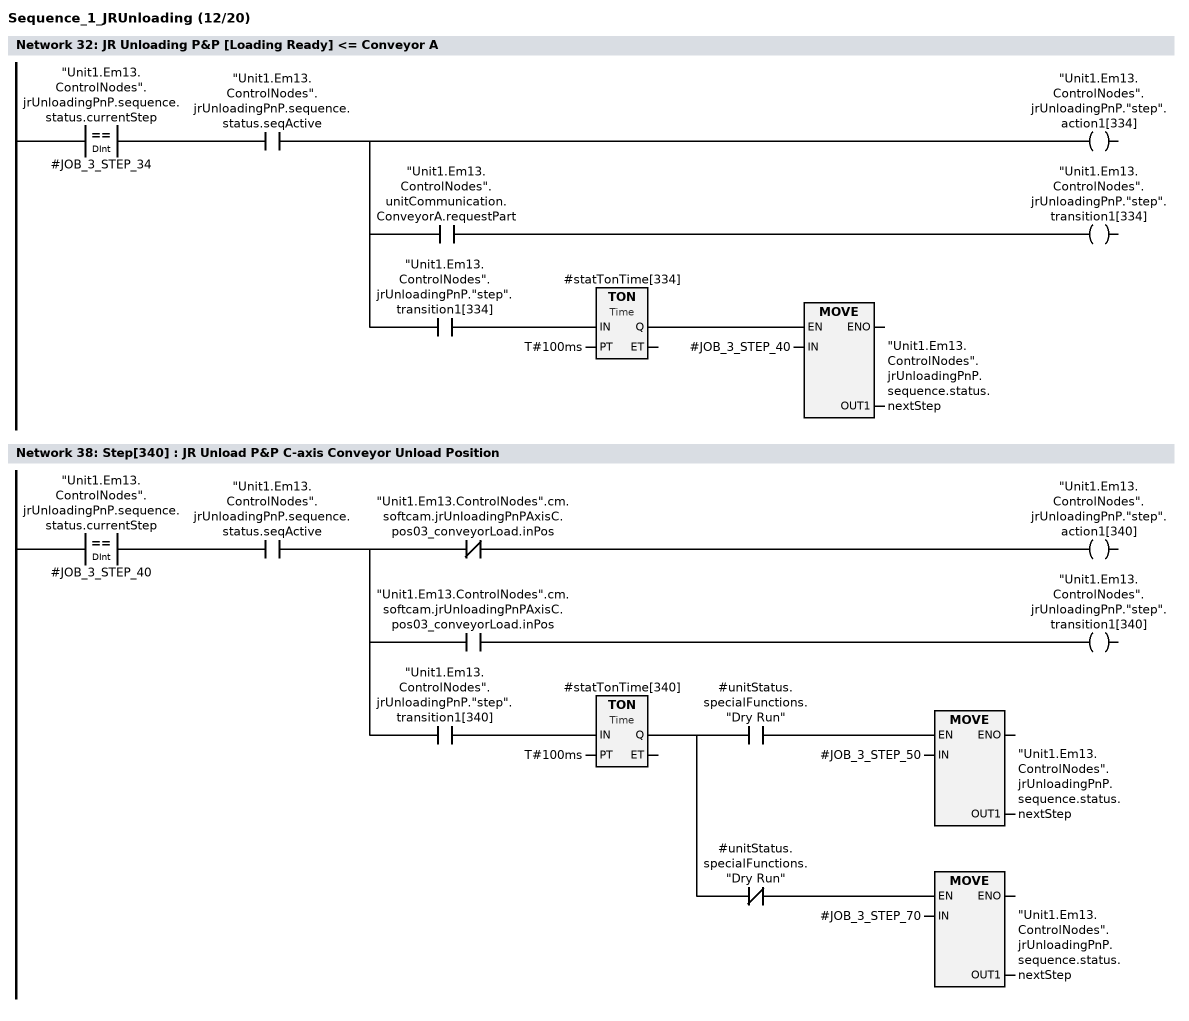
   RUNG wire#powerrail
      { S7_Templates := "SrcType := DInt" } EQ_Contact(in1 := "Unit1.Em13.ControlNodes".jrUnloadingPnP.sequence.status.currentStep, in2 := #JOB_3_STEP_34)
      Contact( "Unit1.Em13.ControlNodes".jrUnloadingPnP.sequence.status.seqActive )
      wire#w1
      Coil( "Unit1.Em13.ControlNodes".jrUnloadingPnP."step".action1[334] )
   END_RUNG
   RUNG wire#w1
      Contact( "Unit1.Em13.ControlNodes".unitCommunication.ConveyorA.requestPart )
      Coil( "Unit1.Em13.ControlNodes".jrUnloadingPnP."step".transition1[334] )
   END_RUNG
   RUNG wire#w1
      Contact( "Unit1.Em13.ControlNodes".jrUnloadingPnP."step".transition1[334] )
      { S7_Templates := "time_type := Time" } #statTonTime[334].TON(pt := T#100ms, et =>)
      Move(in := #JOB_3_STEP_40, out1 => "Unit1.Em13.ControlNodes".jrUnloadingPnP.sequence.status.nextStep)
   END_RUNG
   // the same network as SCL:
   "Unit1.Em13.ControlNodes".jrUnloadingPnP."step".action1[334] := ("Unit1.Em13.ControlNodes".jrUnloadingPnP.sequence.status.currentStep = #JOB_3_STEP_34) AND "Unit1.Em13.ControlNodes".jrUnloadingPnP.sequence.status.seqActive;
   "Unit1.Em13.ControlNodes".jrUnloadingPnP."step".transition1[334] := ("Unit1.Em13.ControlNodes".jrUnloadingPnP.sequence.status.currentStep = #JOB_3_STEP_34) AND "Unit1.Em13.ControlNodes".jrUnloadingPnP.sequence.status.seqActive AND "Unit1.Em13.ControlNodes".unitCommunication.ConveyorA.requestPart;
   #statTonTime[334].TON(IN := ("Unit1.Em13.ControlNodes".jrUnloadingPnP.sequence.status.currentStep = #JOB_3_STEP_34) AND "Unit1.Em13.ControlNodes".jrUnloadingPnP.sequence.status.seqActive AND "Unit1.Em13.ControlNodes".jrUnloadingPnP."step".transition1[334],
                         PT := T#100ms);
   IF #statTonTime[334].Q THEN
       "Unit1.Em13.ControlNodes".jrUnloadingPnP.sequence.status.nextStep := #JOB_3_STEP_40;
   END_IF;
END_REGION

REGION Network 33: JR Unload P&P Z or X-Axis Conveyor Unload Position
END_REGION

REGION Network 34: JR Unloading P&P [Unload Ready] => Conveyor A
END_REGION

REGION Network 35: JR Unloading P&P Clamp Open
END_REGION

REGION Network 36: JR Unload P&P X/Z/C-Axis Wait Position
END_REGION

REGION Network 37: ================================================
END_REGION

REGION Network 38: Step[340] : JR Unload P&P C-axis Conveyor Unload Position
   RUNG wire#powerrail
      { S7_Templates := "SrcType := DInt" } EQ_Contact(in1 := "Unit1.Em13.ControlNodes".jrUnloadingPnP.sequence.status.currentStep, in2 := #JOB_3_STEP_40)
      Contact( "Unit1.Em13.ControlNodes".jrUnloadingPnP.sequence.status.seqActive )
      wire#w1
      I_Contact( "Unit1.Em13.ControlNodes".cm.softcam.jrUnIoadingPnPAxisC.pos03_conveyorLoad.inPos )
      Coil( "Unit1.Em13.ControlNodes".jrUnloadingPnP."step".action1[340] )
   END_RUNG
   RUNG wire#w1
      Contact( "Unit1.Em13.ControlNodes".cm.softcam.jrUnIoadingPnPAxisC.pos03_conveyorLoad.inPos )
      Coil( "Unit1.Em13.ControlNodes".jrUnloadingPnP."step".transition1[340] )
   END_RUNG
   RUNG wire#w1
      Contact( "Unit1.Em13.ControlNodes".jrUnloadingPnP."step".transition1[340] )
      { S7_Templates := "time_type := Time" } #statTonTime[340].TON(pt := T#100ms, et =>)
      wire#w2
      Contact( #unitStatus.specialFunctions."Dry Run" )
      Move(in := #JOB_3_STEP_50, out1 => "Unit1.Em13.ControlNodes".jrUnloadingPnP.sequence.status.nextStep)
   END_RUNG
   RUNG wire#w2
      I_Contact( #unitStatus.specialFunctions."Dry Run" )
      Move(in := #JOB_3_STEP_70, out1 => "Unit1.Em13.ControlNodes".jrUnloadingPnP.sequence.status.nextStep)
   END_RUNG
   // the same network as SCL:
   #_w1 := ("Unit1.Em13.ControlNodes".jrUnloadingPnP.sequence.status.currentStep = #JOB_3_STEP_40) AND "Unit1.Em13.ControlNodes".jrUnloadingPnP.sequence.status.seqActive;
   "Unit1.Em13.ControlNodes".jrUnloadingPnP."step".action1[340] := #_w1 AND NOT "Unit1.Em13.ControlNodes".cm.softcam.jrUnIoadingPnPAxisC.pos03_conveyorLoad.inPos;
   "Unit1.Em13.ControlNodes".jrUnloadingPnP."step".transition1[340] := #_w1 AND "Unit1.Em13.ControlNodes".cm.softcam.jrUnIoadingPnPAxisC.pos03_conveyorLoad.inPos;
   #statTonTime[340].TON(IN := #_w1 AND "Unit1.Em13.ControlNodes".jrUnloadingPnP."step".transition1[340],
                         PT := T#100ms);
   IF #statTonTime[340].Q AND #unitStatus.specialFunctions."Dry Run" THEN
       "Unit1.Em13.ControlNodes".jrUnloadingPnP.sequence.status.nextStep := #JOB_3_STEP_50;
   END_IF;
   IF #statTonTime[340].Q AND NOT #unitStatus.specialFunctions."Dry Run" THEN
       "Unit1.Em13.ControlNodes".jrUnloadingPnP.sequence.status.nextStep := #JOB_3_STEP_70;
   END_IF;
END_REGION

REGION Network 39: Step[350] : JR Unload P&P Z-axis Conveyor Unload Position
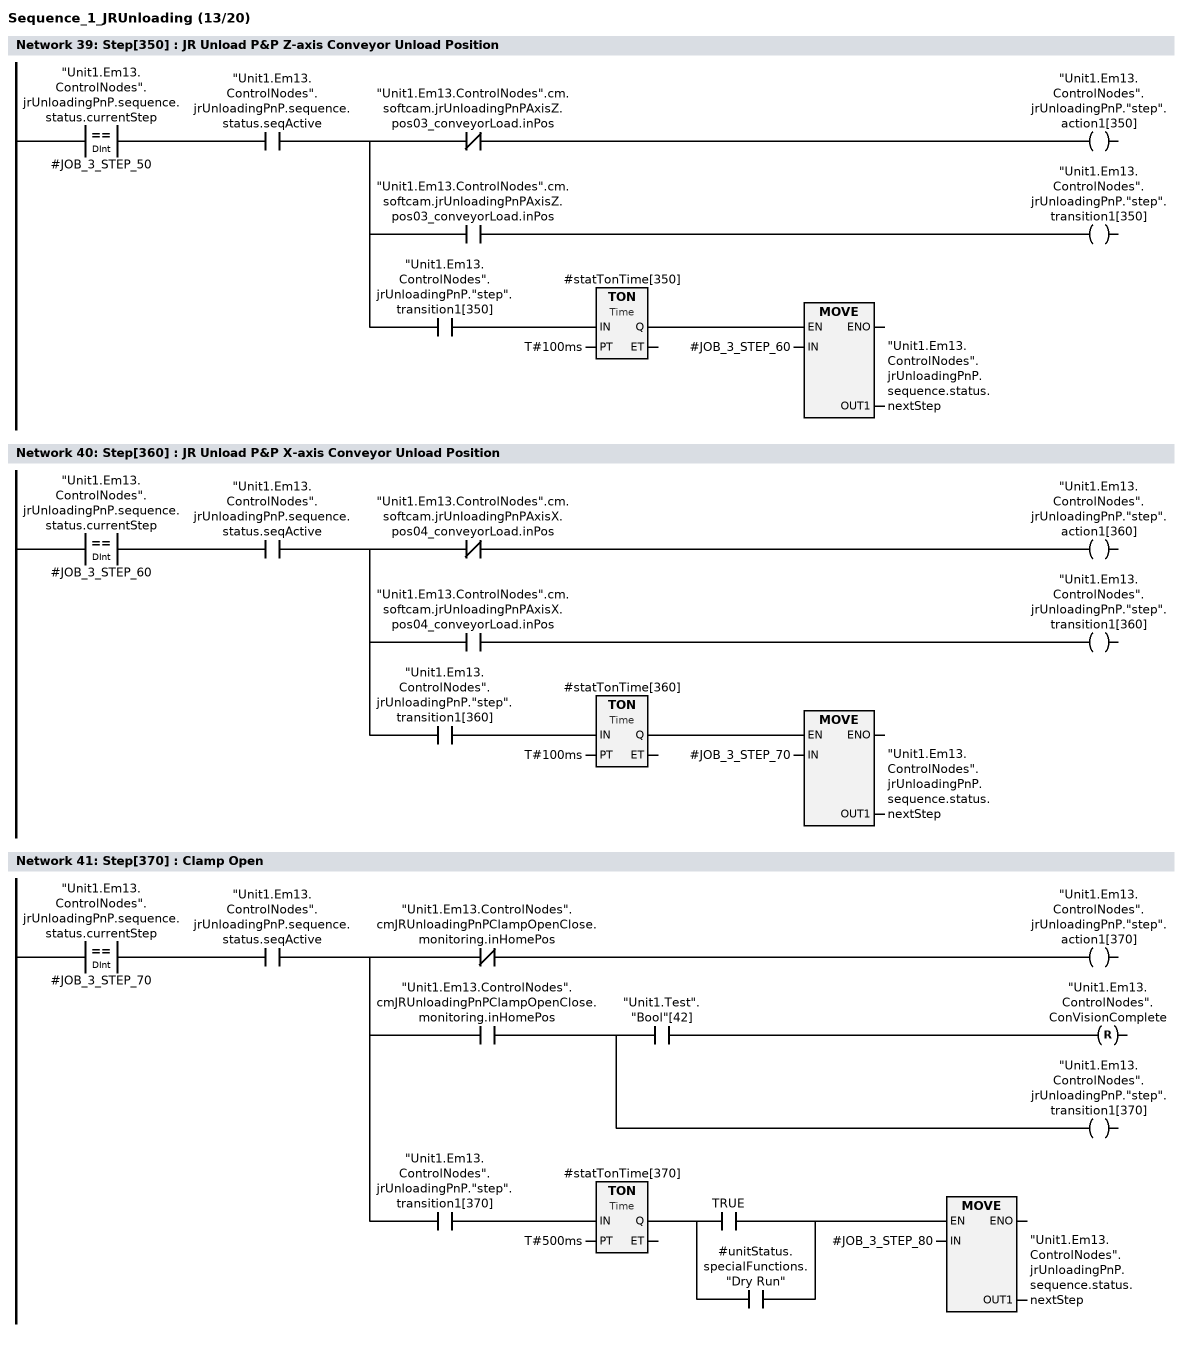
   RUNG wire#powerrail
      { S7_Templates := "SrcType := DInt" } EQ_Contact(in1 := "Unit1.Em13.ControlNodes".jrUnloadingPnP.sequence.status.currentStep, in2 := #JOB_3_STEP_50)
      Contact( "Unit1.Em13.ControlNodes".jrUnloadingPnP.sequence.status.seqActive )
      wire#w1
      I_Contact( "Unit1.Em13.ControlNodes".cm.softcam.jrUnIoadingPnPAxisZ.pos03_conveyorLoad.inPos )
      Coil( "Unit1.Em13.ControlNodes".jrUnloadingPnP."step".action1[350] )
   END_RUNG
   RUNG wire#w1
      Contact( "Unit1.Em13.ControlNodes".cm.softcam.jrUnIoadingPnPAxisZ.pos03_conveyorLoad.inPos )
      Coil( "Unit1.Em13.ControlNodes".jrUnloadingPnP."step".transition1[350] )
   END_RUNG
   RUNG wire#w1
      Contact( "Unit1.Em13.ControlNodes".jrUnloadingPnP."step".transition1[350] )
      { S7_Templates := "time_type := Time" } #statTonTime[350].TON(pt := T#100ms, et =>)
      Move(in := #JOB_3_STEP_60, out1 => "Unit1.Em13.ControlNodes".jrUnloadingPnP.sequence.status.nextStep)
   END_RUNG
   // the same network as SCL:
   #_w1 := ("Unit1.Em13.ControlNodes".jrUnloadingPnP.sequence.status.currentStep = #JOB_3_STEP_50) AND "Unit1.Em13.ControlNodes".jrUnloadingPnP.sequence.status.seqActive;
   "Unit1.Em13.ControlNodes".jrUnloadingPnP."step".action1[350] := #_w1 AND NOT "Unit1.Em13.ControlNodes".cm.softcam.jrUnIoadingPnPAxisZ.pos03_conveyorLoad.inPos;
   "Unit1.Em13.ControlNodes".jrUnloadingPnP."step".transition1[350] := #_w1 AND "Unit1.Em13.ControlNodes".cm.softcam.jrUnIoadingPnPAxisZ.pos03_conveyorLoad.inPos;
   #statTonTime[350].TON(IN := #_w1 AND "Unit1.Em13.ControlNodes".jrUnloadingPnP."step".transition1[350],
                         PT := T#100ms);
   IF #statTonTime[350].Q THEN
       "Unit1.Em13.ControlNodes".jrUnloadingPnP.sequence.status.nextStep := #JOB_3_STEP_60;
   END_IF;
END_REGION

REGION Network 40: Step[360] : JR Unload P&P X-axis Conveyor Unload Position
   RUNG wire#powerrail
      { S7_Templates := "SrcType := DInt" } EQ_Contact(in1 := "Unit1.Em13.ControlNodes".jrUnloadingPnP.sequence.status.currentStep, in2 := #JOB_3_STEP_60)
      Contact( "Unit1.Em13.ControlNodes".jrUnloadingPnP.sequence.status.seqActive )
      wire#w1
      I_Contact( "Unit1.Em13.ControlNodes".cm.softcam.jrUnIoadingPnPAxisX.pos04_conveyorLoad.inPos )
      Coil( "Unit1.Em13.ControlNodes".jrUnloadingPnP."step".action1[360] )
   END_RUNG
   RUNG wire#w1
      Contact( "Unit1.Em13.ControlNodes".cm.softcam.jrUnIoadingPnPAxisX.pos04_conveyorLoad.inPos )
      Coil( "Unit1.Em13.ControlNodes".jrUnloadingPnP."step".transition1[360] )
   END_RUNG
   RUNG wire#w1
      Contact( "Unit1.Em13.ControlNodes".jrUnloadingPnP."step".transition1[360] )
      { S7_Templates := "time_type := Time" } #statTonTime[360].TON(pt := T#100ms, et =>)
      Move(in := #JOB_3_STEP_70, out1 => "Unit1.Em13.ControlNodes".jrUnloadingPnP.sequence.status.nextStep)
   END_RUNG
   // the same network as SCL:
   #_w1 := ("Unit1.Em13.ControlNodes".jrUnloadingPnP.sequence.status.currentStep = #JOB_3_STEP_60) AND "Unit1.Em13.ControlNodes".jrUnloadingPnP.sequence.status.seqActive;
   "Unit1.Em13.ControlNodes".jrUnloadingPnP."step".action1[360] := #_w1 AND NOT "Unit1.Em13.ControlNodes".cm.softcam.jrUnIoadingPnPAxisX.pos04_conveyorLoad.inPos;
   "Unit1.Em13.ControlNodes".jrUnloadingPnP."step".transition1[360] := #_w1 AND "Unit1.Em13.ControlNodes".cm.softcam.jrUnIoadingPnPAxisX.pos04_conveyorLoad.inPos;
   #statTonTime[360].TON(IN := #_w1 AND "Unit1.Em13.ControlNodes".jrUnloadingPnP."step".transition1[360],
                         PT := T#100ms);
   IF #statTonTime[360].Q THEN
       "Unit1.Em13.ControlNodes".jrUnloadingPnP.sequence.status.nextStep := #JOB_3_STEP_70;
   END_IF;
END_REGION

REGION Network 41: Step[370] : Clamp Open
   RUNG wire#powerrail
      { S7_Templates := "SrcType := DInt" } EQ_Contact(in1 := "Unit1.Em13.ControlNodes".jrUnloadingPnP.sequence.status.currentStep, in2 := #JOB_3_STEP_70)
      Contact( "Unit1.Em13.ControlNodes".jrUnloadingPnP.sequence.status.seqActive )
      wire#w1
      I_Contact( "Unit1.Em13.ControlNodes".cmJRUnloadingPnPClampOpenClose.monitoring.inHomePos )
      Coil( "Unit1.Em13.ControlNodes".jrUnloadingPnP."step".action1[370] )
   END_RUNG
   RUNG wire#w1
      Contact( "Unit1.Em13.ControlNodes".cmJRUnloadingPnPClampOpenClose.monitoring.inHomePos )
      wire#w2
      Contact( "Unit1.Test"."Bool"[42] )
      R_Coil( "Unit1.Em13.ControlNodes".ConVisionComplete )
   END_RUNG
   RUNG wire#w2
      Coil( "Unit1.Em13.ControlNodes".jrUnloadingPnP."step".transition1[370] )
   END_RUNG
   RUNG wire#w1
      Contact( "Unit1.Em13.ControlNodes".jrUnloadingPnP."step".transition1[370] )
      { S7_Templates := "time_type := Time" } #statTonTime[370].TON(pt := T#500ms, et =>)
      wire#w3
      Contact( TRUE )
      wire#w4
      Move(in := #JOB_3_STEP_80, out1 => "Unit1.Em13.ControlNodes".jrUnloadingPnP.sequence.status.nextStep)
   END_RUNG
   RUNG wire#w3
      Contact( #unitStatus.specialFunctions."Dry Run" )
   END_RUNG wire#w4
   // the same network as SCL:
   #_w1 := ("Unit1.Em13.ControlNodes".jrUnloadingPnP.sequence.status.currentStep = #JOB_3_STEP_70) AND "Unit1.Em13.ControlNodes".jrUnloadingPnP.sequence.status.seqActive;
   "Unit1.Em13.ControlNodes".jrUnloadingPnP."step".action1[370] := #_w1 AND NOT "Unit1.Em13.ControlNodes".cmJRUnloadingPnPClampOpenClose.monitoring.inHomePos;
   #_w2 := #_w1 AND "Unit1.Em13.ControlNodes".cmJRUnloadingPnPClampOpenClose.monitoring.inHomePos;
   IF #_w2 AND "Unit1.Test"."Bool"[42] THEN "Unit1.Em13.ControlNodes".ConVisionComplete := FALSE; END_IF;
   "Unit1.Em13.ControlNodes".jrUnloadingPnP."step".transition1[370] := #_w2;
   #statTonTime[370].TON(IN := #_w1 AND "Unit1.Em13.ControlNodes".jrUnloadingPnP."step".transition1[370],
                         PT := T#500ms);
   IF #statTonTime[370].Q AND (TRUE OR #unitStatus.specialFunctions."Dry Run") THEN
       "Unit1.Em13.ControlNodes".jrUnloadingPnP.sequence.status.nextStep := #JOB_3_STEP_80;
   END_IF;
END_REGION

REGION Network 42: Step[380] : JR Unload P&P X/Z/C-Axis Wait Position
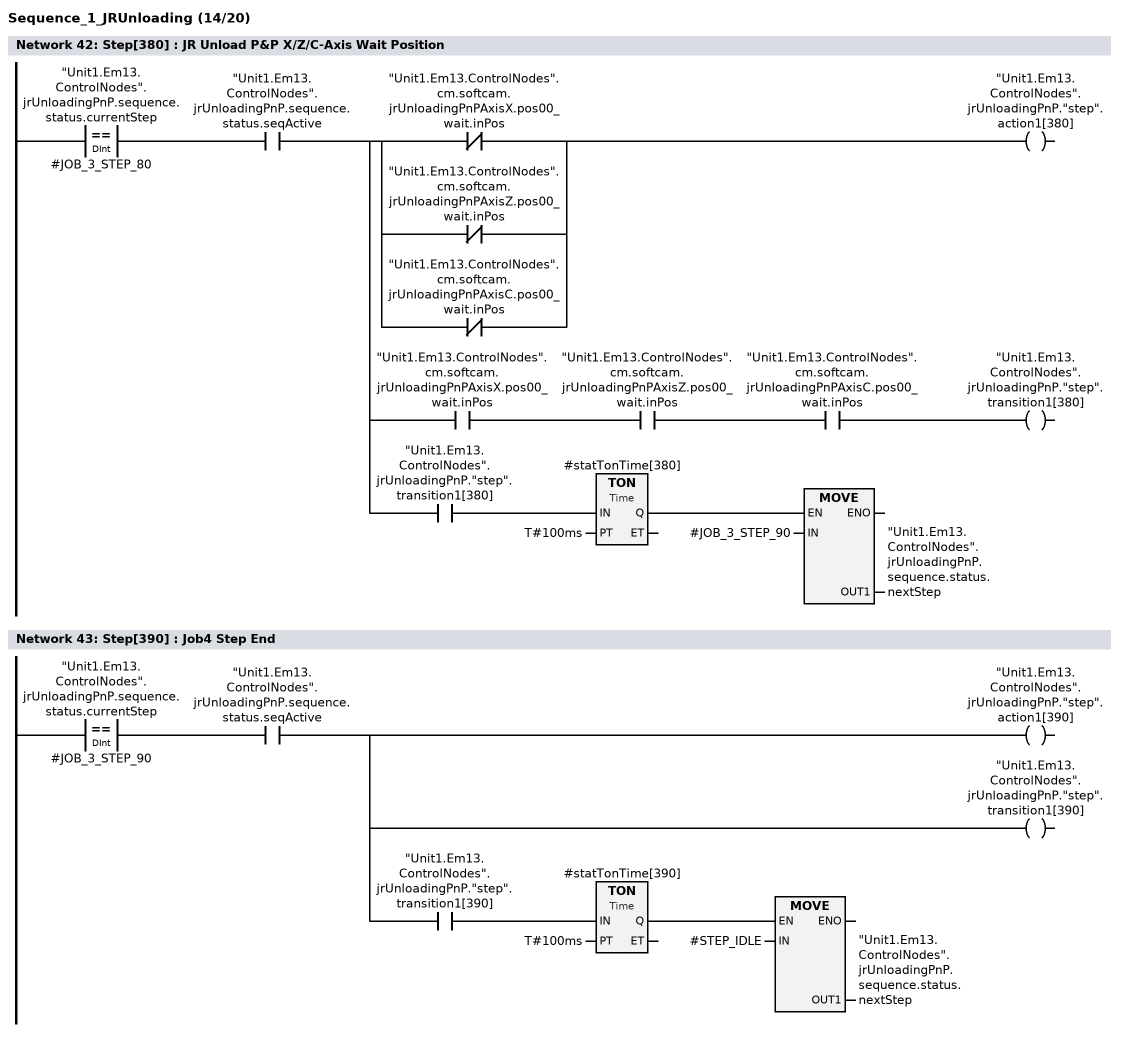
   RUNG wire#powerrail
      { S7_Templates := "SrcType := DInt" } EQ_Contact(in1 := "Unit1.Em13.ControlNodes".jrUnloadingPnP.sequence.status.currentStep, in2 := #JOB_3_STEP_80)
      Contact( "Unit1.Em13.ControlNodes".jrUnloadingPnP.sequence.status.seqActive )
      wire#w1
      I_Contact( "Unit1.Em13.ControlNodes".cm.softcam.jrUnIoadingPnPAxisX.pos00_wait.inPos )
      wire#w2
      Coil( "Unit1.Em13.ControlNodes".jrUnloadingPnP."step".action1[380] )
   END_RUNG
   RUNG wire#w1
      I_Contact( "Unit1.Em13.ControlNodes".cm.softcam.jrUnIoadingPnPAxisZ.pos00_wait.inPos )
   END_RUNG wire#w2
   RUNG wire#w1
      I_Contact( "Unit1.Em13.ControlNodes".cm.softcam.jrUnIoadingPnPAxisC.pos00_wait.inPos )
   END_RUNG wire#w2
   RUNG wire#w1
      Contact( "Unit1.Em13.ControlNodes".cm.softcam.jrUnIoadingPnPAxisX.pos00_wait.inPos )
      Contact( "Unit1.Em13.ControlNodes".cm.softcam.jrUnIoadingPnPAxisZ.pos00_wait.inPos )
      Contact( "Unit1.Em13.ControlNodes".cm.softcam.jrUnIoadingPnPAxisC.pos00_wait.inPos )
      Coil( "Unit1.Em13.ControlNodes".jrUnloadingPnP."step".transition1[380] )
   END_RUNG
   RUNG wire#w1
      Contact( "Unit1.Em13.ControlNodes".jrUnloadingPnP."step".transition1[380] )
      { S7_Templates := "time_type := Time" } #statTonTime[380].TON(pt := T#100ms, et =>)
      Move(in := #JOB_3_STEP_90, out1 => "Unit1.Em13.ControlNodes".jrUnloadingPnP.sequence.status.nextStep)
   END_RUNG
   // the same network as SCL:
   #_w1 := ("Unit1.Em13.ControlNodes".jrUnloadingPnP.sequence.status.currentStep = #JOB_3_STEP_80) AND "Unit1.Em13.ControlNodes".jrUnloadingPnP.sequence.status.seqActive;
   "Unit1.Em13.ControlNodes".jrUnloadingPnP."step".action1[380] := #_w1 AND (NOT "Unit1.Em13.ControlNodes".cm.softcam.jrUnIoadingPnPAxisX.pos00_wait.inPos OR NOT "Unit1.Em13.ControlNodes".cm.softcam.jrUnIoadingPnPAxisZ.pos00_wait.inPos OR NOT "Unit1.Em13.ControlNodes".cm.softcam.jrUnIoadingPnPAxisC.pos00_wait.inPos);
   "Unit1.Em13.ControlNodes".jrUnloadingPnP."step".transition1[380] := #_w1 AND "Unit1.Em13.ControlNodes".cm.softcam.jrUnIoadingPnPAxisX.pos00_wait.inPos AND "Unit1.Em13.ControlNodes".cm.softcam.jrUnIoadingPnPAxisZ.pos00_wait.inPos AND "Unit1.Em13.ControlNodes".cm.softcam.jrUnIoadingPnPAxisC.pos00_wait.inPos;
   #statTonTime[380].TON(IN := #_w1 AND "Unit1.Em13.ControlNodes".jrUnloadingPnP."step".transition1[380],
                         PT := T#100ms);
   IF #statTonTime[380].Q THEN
       "Unit1.Em13.ControlNodes".jrUnloadingPnP.sequence.status.nextStep := #JOB_3_STEP_90;
   END_IF;
END_REGION

REGION Network 43: Step[390] : Job4 Step End
   RUNG wire#powerrail
      { S7_Templates := "SrcType := DInt" } EQ_Contact(in1 := "Unit1.Em13.ControlNodes".jrUnloadingPnP.sequence.status.currentStep, in2 := #JOB_3_STEP_90)
      Contact( "Unit1.Em13.ControlNodes".jrUnloadingPnP.sequence.status.seqActive )
      wire#w1
      Coil( "Unit1.Em13.ControlNodes".jrUnloadingPnP."step".action1[390] )
   END_RUNG
   RUNG wire#w1
      Coil( "Unit1.Em13.ControlNodes".jrUnloadingPnP."step".transition1[390] )
   END_RUNG
   RUNG wire#w1
      Contact( "Unit1.Em13.ControlNodes".jrUnloadingPnP."step".transition1[390] )
      { S7_Templates := "time_type := Time" } #statTonTime[390].TON(pt := T#100ms, et =>)
      Move(in := #STEP_IDLE, out1 => "Unit1.Em13.ControlNodes".jrUnloadingPnP.sequence.status.nextStep)
   END_RUNG
   // the same network as SCL:
   "Unit1.Em13.ControlNodes".jrUnloadingPnP."step".action1[390] := ("Unit1.Em13.ControlNodes".jrUnloadingPnP.sequence.status.currentStep = #JOB_3_STEP_90) AND "Unit1.Em13.ControlNodes".jrUnloadingPnP.sequence.status.seqActive;
   "Unit1.Em13.ControlNodes".jrUnloadingPnP."step".transition1[390] := ("Unit1.Em13.ControlNodes".jrUnloadingPnP.sequence.status.currentStep = #JOB_3_STEP_90) AND "Unit1.Em13.ControlNodes".jrUnloadingPnP.sequence.status.seqActive;
   #statTonTime[390].TON(IN := ("Unit1.Em13.ControlNodes".jrUnloadingPnP.sequence.status.currentStep = #JOB_3_STEP_90) AND "Unit1.Em13.ControlNodes".jrUnloadingPnP.sequence.status.seqActive AND "Unit1.Em13.ControlNodes".jrUnloadingPnP."step".transition1[390],
                         PT := T#100ms);
   IF #statTonTime[390].Q THEN
       "Unit1.Em13.ControlNodes".jrUnloadingPnP.sequence.status.nextStep := #STEP_IDLE;
   END_IF;
END_REGION

REGION Network 44: ************ JOB[4] STACK NG BOX JR PUT=AUTO **************
END_REGION

REGION Network 45: Step[401] : JOB[4] Condition
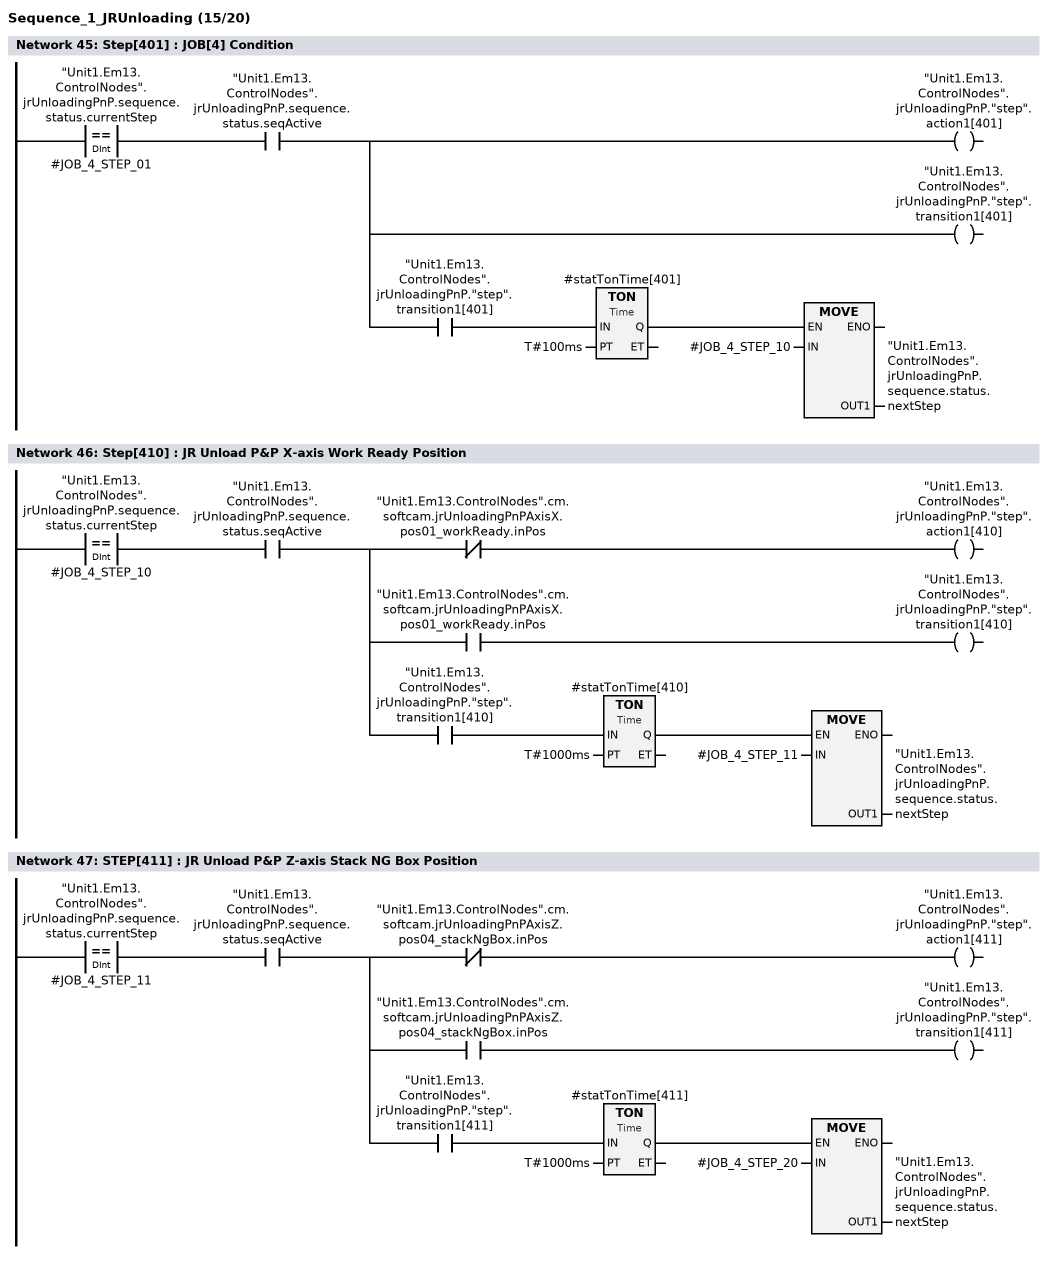
   RUNG wire#powerrail
      { S7_Templates := "SrcType := DInt" } EQ_Contact(in1 := "Unit1.Em13.ControlNodes".jrUnloadingPnP.sequence.status.currentStep, in2 := #JOB_4_STEP_01)
      Contact( "Unit1.Em13.ControlNodes".jrUnloadingPnP.sequence.status.seqActive )
      wire#w1
      Coil( "Unit1.Em13.ControlNodes".jrUnloadingPnP."step".action1[401] )
   END_RUNG
   RUNG wire#w1
      Coil( "Unit1.Em13.ControlNodes".jrUnloadingPnP."step".transition1[401] )
   END_RUNG
   RUNG wire#w1
      Contact( "Unit1.Em13.ControlNodes".jrUnloadingPnP."step".transition1[401] )
      { S7_Templates := "time_type := Time" } #statTonTime[401].TON(pt := T#100ms, et =>)
      Move(in := #JOB_4_STEP_10, out1 => "Unit1.Em13.ControlNodes".jrUnloadingPnP.sequence.status.nextStep)
   END_RUNG
   // the same network as SCL:
   "Unit1.Em13.ControlNodes".jrUnloadingPnP."step".action1[401] := ("Unit1.Em13.ControlNodes".jrUnloadingPnP.sequence.status.currentStep = #JOB_4_STEP_01) AND "Unit1.Em13.ControlNodes".jrUnloadingPnP.sequence.status.seqActive;
   "Unit1.Em13.ControlNodes".jrUnloadingPnP."step".transition1[401] := ("Unit1.Em13.ControlNodes".jrUnloadingPnP.sequence.status.currentStep = #JOB_4_STEP_01) AND "Unit1.Em13.ControlNodes".jrUnloadingPnP.sequence.status.seqActive;
   #statTonTime[401].TON(IN := ("Unit1.Em13.ControlNodes".jrUnloadingPnP.sequence.status.currentStep = #JOB_4_STEP_01) AND "Unit1.Em13.ControlNodes".jrUnloadingPnP.sequence.status.seqActive AND "Unit1.Em13.ControlNodes".jrUnloadingPnP."step".transition1[401],
                         PT := T#100ms);
   IF #statTonTime[401].Q THEN
       "Unit1.Em13.ControlNodes".jrUnloadingPnP.sequence.status.nextStep := #JOB_4_STEP_10;
   END_IF;
END_REGION

REGION Network 46: Step[410] : JR Unload P&P X-axis Work Ready Position
   RUNG wire#powerrail
      { S7_Templates := "SrcType := DInt" } EQ_Contact(in1 := "Unit1.Em13.ControlNodes".jrUnloadingPnP.sequence.status.currentStep, in2 := #JOB_4_STEP_10)
      Contact( "Unit1.Em13.ControlNodes".jrUnloadingPnP.sequence.status.seqActive )
      wire#w1
      I_Contact( "Unit1.Em13.ControlNodes".cm.softcam.jrUnIoadingPnPAxisX.pos01_workReady.inPos )
      Coil( "Unit1.Em13.ControlNodes".jrUnloadingPnP."step".action1[410] )
   END_RUNG
   RUNG wire#w1
      Contact( "Unit1.Em13.ControlNodes".cm.softcam.jrUnIoadingPnPAxisX.pos01_workReady.inPos )
      Coil( "Unit1.Em13.ControlNodes".jrUnloadingPnP."step".transition1[410] )
   END_RUNG
   RUNG wire#w1
      Contact( "Unit1.Em13.ControlNodes".jrUnloadingPnP."step".transition1[410] )
      { S7_Templates := "time_type := Time" } #statTonTime[410].TON(pt := T#1000ms, et =>)
      Move(in := #JOB_4_STEP_11, out1 => "Unit1.Em13.ControlNodes".jrUnloadingPnP.sequence.status.nextStep)
   END_RUNG
   // the same network as SCL:
   #_w1 := ("Unit1.Em13.ControlNodes".jrUnloadingPnP.sequence.status.currentStep = #JOB_4_STEP_10) AND "Unit1.Em13.ControlNodes".jrUnloadingPnP.sequence.status.seqActive;
   "Unit1.Em13.ControlNodes".jrUnloadingPnP."step".action1[410] := #_w1 AND NOT "Unit1.Em13.ControlNodes".cm.softcam.jrUnIoadingPnPAxisX.pos01_workReady.inPos;
   "Unit1.Em13.ControlNodes".jrUnloadingPnP."step".transition1[410] := #_w1 AND "Unit1.Em13.ControlNodes".cm.softcam.jrUnIoadingPnPAxisX.pos01_workReady.inPos;
   #statTonTime[410].TON(IN := #_w1 AND "Unit1.Em13.ControlNodes".jrUnloadingPnP."step".transition1[410],
                         PT := T#1000ms);
   IF #statTonTime[410].Q THEN
       "Unit1.Em13.ControlNodes".jrUnloadingPnP.sequence.status.nextStep := #JOB_4_STEP_11;
   END_IF;
END_REGION

REGION Network 47: STEP[411] : JR Unload P&P Z-axis Stack NG Box Position
   RUNG wire#powerrail
      { S7_Templates := "SrcType := DInt" } EQ_Contact(in1 := "Unit1.Em13.ControlNodes".jrUnloadingPnP.sequence.status.currentStep, in2 := #JOB_4_STEP_11)
      Contact( "Unit1.Em13.ControlNodes".jrUnloadingPnP.sequence.status.seqActive )
      wire#w1
      I_Contact( "Unit1.Em13.ControlNodes".cm.softcam.jrUnIoadingPnPAxisZ.pos04_stackNgBox.inPos )
      Coil( "Unit1.Em13.ControlNodes".jrUnloadingPnP."step".action1[411] )
   END_RUNG
   RUNG wire#w1
      Contact( "Unit1.Em13.ControlNodes".cm.softcam.jrUnIoadingPnPAxisZ.pos04_stackNgBox.inPos )
      Coil( "Unit1.Em13.ControlNodes".jrUnloadingPnP."step".transition1[411] )
   END_RUNG
   RUNG wire#w1
      Contact( "Unit1.Em13.ControlNodes".jrUnloadingPnP."step".transition1[411] )
      { S7_Templates := "time_type := Time" } #statTonTime[411].TON(pt := T#1000ms, et =>)
      Move(in := #JOB_4_STEP_20, out1 => "Unit1.Em13.ControlNodes".jrUnloadingPnP.sequence.status.nextStep)
   END_RUNG
   // the same network as SCL:
   #_w1 := ("Unit1.Em13.ControlNodes".jrUnloadingPnP.sequence.status.currentStep = #JOB_4_STEP_11) AND "Unit1.Em13.ControlNodes".jrUnloadingPnP.sequence.status.seqActive;
   "Unit1.Em13.ControlNodes".jrUnloadingPnP."step".action1[411] := #_w1 AND NOT "Unit1.Em13.ControlNodes".cm.softcam.jrUnIoadingPnPAxisZ.pos04_stackNgBox.inPos;
   "Unit1.Em13.ControlNodes".jrUnloadingPnP."step".transition1[411] := #_w1 AND "Unit1.Em13.ControlNodes".cm.softcam.jrUnIoadingPnPAxisZ.pos04_stackNgBox.inPos;
   #statTonTime[411].TON(IN := #_w1 AND "Unit1.Em13.ControlNodes".jrUnloadingPnP."step".transition1[411],
                         PT := T#1000ms);
   IF #statTonTime[411].Q THEN
       "Unit1.Em13.ControlNodes".jrUnloadingPnP.sequence.status.nextStep := #JOB_4_STEP_20;
   END_IF;
END_REGION

REGION Network 48: STEP[420] : JR Unload P&P C-axis Stack NG Box Position
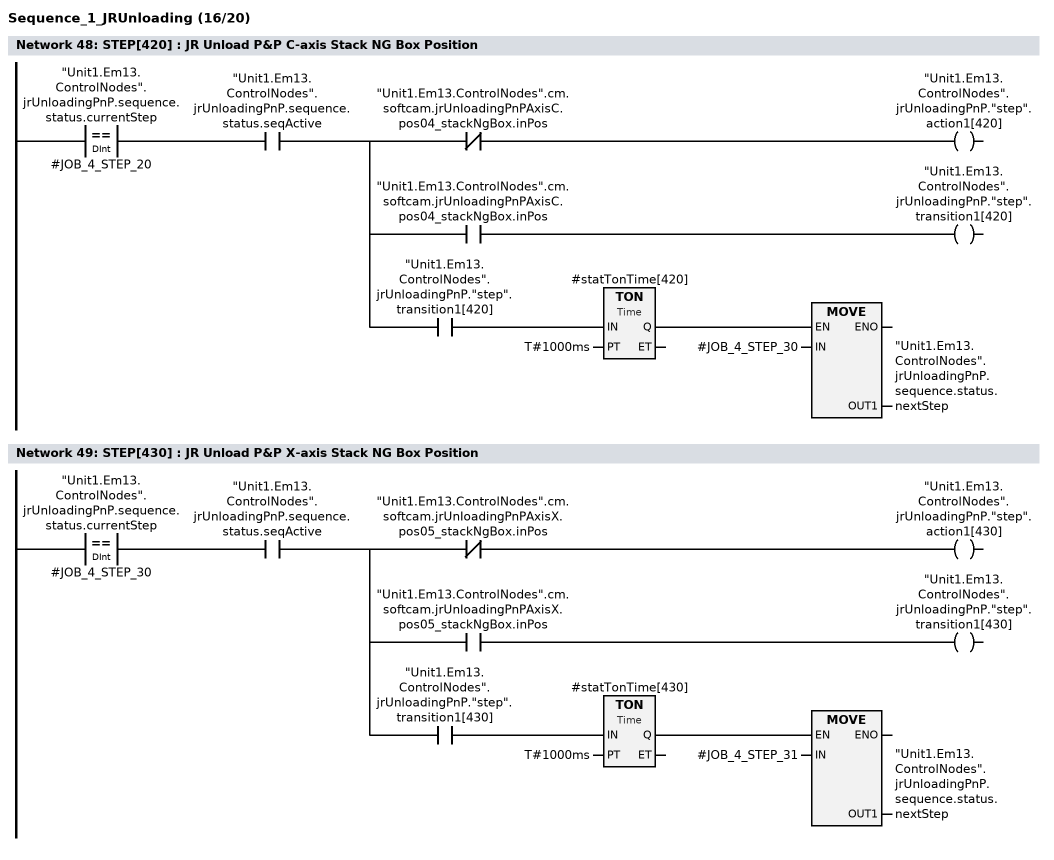
   RUNG wire#powerrail
      { S7_Templates := "SrcType := DInt" } EQ_Contact(in1 := "Unit1.Em13.ControlNodes".jrUnloadingPnP.sequence.status.currentStep, in2 := #JOB_4_STEP_20)
      Contact( "Unit1.Em13.ControlNodes".jrUnloadingPnP.sequence.status.seqActive )
      wire#w1
      I_Contact( "Unit1.Em13.ControlNodes".cm.softcam.jrUnIoadingPnPAxisC.pos04_stackNgBox.inPos )
      Coil( "Unit1.Em13.ControlNodes".jrUnloadingPnP."step".action1[420] )
   END_RUNG
   RUNG wire#w1
      Contact( "Unit1.Em13.ControlNodes".cm.softcam.jrUnIoadingPnPAxisC.pos04_stackNgBox.inPos )
      Coil( "Unit1.Em13.ControlNodes".jrUnloadingPnP."step".transition1[420] )
   END_RUNG
   RUNG wire#w1
      Contact( "Unit1.Em13.ControlNodes".jrUnloadingPnP."step".transition1[420] )
      { S7_Templates := "time_type := Time" } #statTonTime[420].TON(pt := T#1000ms, et =>)
      Move(in := #JOB_4_STEP_30, out1 => "Unit1.Em13.ControlNodes".jrUnloadingPnP.sequence.status.nextStep)
   END_RUNG
   // the same network as SCL:
   #_w1 := ("Unit1.Em13.ControlNodes".jrUnloadingPnP.sequence.status.currentStep = #JOB_4_STEP_20) AND "Unit1.Em13.ControlNodes".jrUnloadingPnP.sequence.status.seqActive;
   "Unit1.Em13.ControlNodes".jrUnloadingPnP."step".action1[420] := #_w1 AND NOT "Unit1.Em13.ControlNodes".cm.softcam.jrUnIoadingPnPAxisC.pos04_stackNgBox.inPos;
   "Unit1.Em13.ControlNodes".jrUnloadingPnP."step".transition1[420] := #_w1 AND "Unit1.Em13.ControlNodes".cm.softcam.jrUnIoadingPnPAxisC.pos04_stackNgBox.inPos;
   #statTonTime[420].TON(IN := #_w1 AND "Unit1.Em13.ControlNodes".jrUnloadingPnP."step".transition1[420],
                         PT := T#1000ms);
   IF #statTonTime[420].Q THEN
       "Unit1.Em13.ControlNodes".jrUnloadingPnP.sequence.status.nextStep := #JOB_4_STEP_30;
   END_IF;
END_REGION

REGION Network 49: STEP[430] : JR Unload P&P X-axis Stack NG Box Position
   RUNG wire#powerrail
      { S7_Templates := "SrcType := DInt" } EQ_Contact(in1 := "Unit1.Em13.ControlNodes".jrUnloadingPnP.sequence.status.currentStep, in2 := #JOB_4_STEP_30)
      Contact( "Unit1.Em13.ControlNodes".jrUnloadingPnP.sequence.status.seqActive )
      wire#w1
      I_Contact( "Unit1.Em13.ControlNodes".cm.softcam.jrUnIoadingPnPAxisX.pos05_stackNgBox.inPos )
      Coil( "Unit1.Em13.ControlNodes".jrUnloadingPnP."step".action1[430] )
   END_RUNG
   RUNG wire#w1
      Contact( "Unit1.Em13.ControlNodes".cm.softcam.jrUnIoadingPnPAxisX.pos05_stackNgBox.inPos )
      Coil( "Unit1.Em13.ControlNodes".jrUnloadingPnP."step".transition1[430] )
   END_RUNG
   RUNG wire#w1
      Contact( "Unit1.Em13.ControlNodes".jrUnloadingPnP."step".transition1[430] )
      { S7_Templates := "time_type := Time" } #statTonTime[430].TON(pt := T#1000ms, et =>)
      Move(in := #JOB_4_STEP_31, out1 => "Unit1.Em13.ControlNodes".jrUnloadingPnP.sequence.status.nextStep)
   END_RUNG
   // the same network as SCL:
   #_w1 := ("Unit1.Em13.ControlNodes".jrUnloadingPnP.sequence.status.currentStep = #JOB_4_STEP_30) AND "Unit1.Em13.ControlNodes".jrUnloadingPnP.sequence.status.seqActive;
   "Unit1.Em13.ControlNodes".jrUnloadingPnP."step".action1[430] := #_w1 AND NOT "Unit1.Em13.ControlNodes".cm.softcam.jrUnIoadingPnPAxisX.pos05_stackNgBox.inPos;
   "Unit1.Em13.ControlNodes".jrUnloadingPnP."step".transition1[430] := #_w1 AND "Unit1.Em13.ControlNodes".cm.softcam.jrUnIoadingPnPAxisX.pos05_stackNgBox.inPos;
   #statTonTime[430].TON(IN := #_w1 AND "Unit1.Em13.ControlNodes".jrUnloadingPnP."step".transition1[430],
                         PT := T#1000ms);
   IF #statTonTime[430].Q THEN
       "Unit1.Em13.ControlNodes".jrUnloadingPnP.sequence.status.nextStep := #JOB_4_STEP_31;
   END_IF;
END_REGION

REGION Network 50: STEP[431] : JR Unloading P&P [Unloading Ready] => Stack NG Box
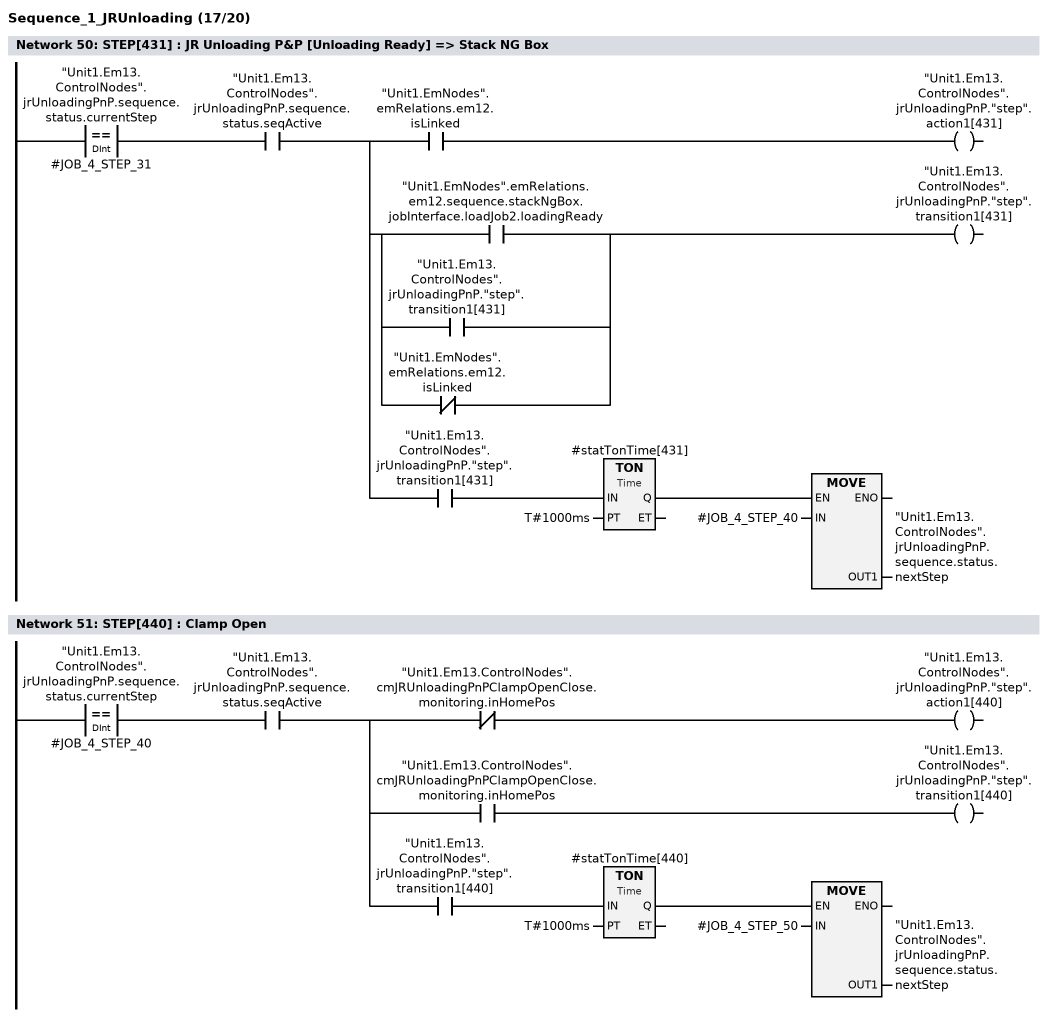
   RUNG wire#powerrail
      { S7_Templates := "SrcType := DInt" } EQ_Contact(in1 := "Unit1.Em13.ControlNodes".jrUnloadingPnP.sequence.status.currentStep, in2 := #JOB_4_STEP_31)
      Contact( "Unit1.Em13.ControlNodes".jrUnloadingPnP.sequence.status.seqActive )
      wire#w1
      Contact( "Unit1.EmNodes".emRelations.em12.isLinked )
      Coil( "Unit1.Em13.ControlNodes".jrUnloadingPnP."step".action1[431] )
   END_RUNG
   RUNG wire#w1
      Contact( "Unit1.EmNodes".emRelations.em12.sequence.stackNgBox.jobInterface.loadJob2.loadingReady )
      wire#w2
      Coil( "Unit1.Em13.ControlNodes".jrUnloadingPnP."step".transition1[431] )
   END_RUNG
   RUNG wire#w1
      Contact( "Unit1.Em13.ControlNodes".jrUnloadingPnP."step".transition1[431] )
   END_RUNG wire#w2
   RUNG wire#w1
      I_Contact( "Unit1.EmNodes".emRelations.em12.isLinked )
   END_RUNG wire#w2
   RUNG wire#w1
      Contact( "Unit1.Em13.ControlNodes".jrUnloadingPnP."step".transition1[431] )
      { S7_Templates := "time_type := Time" } #statTonTime[431].TON(pt := T#1000ms, et =>)
      Move(in := #JOB_4_STEP_40, out1 => "Unit1.Em13.ControlNodes".jrUnloadingPnP.sequence.status.nextStep)
   END_RUNG
   // the same network as SCL:
   #_w1 := ("Unit1.Em13.ControlNodes".jrUnloadingPnP.sequence.status.currentStep = #JOB_4_STEP_31) AND "Unit1.Em13.ControlNodes".jrUnloadingPnP.sequence.status.seqActive;
   "Unit1.Em13.ControlNodes".jrUnloadingPnP."step".action1[431] := #_w1 AND "Unit1.EmNodes".emRelations.em12.isLinked;
   "Unit1.Em13.ControlNodes".jrUnloadingPnP."step".transition1[431] := #_w1 AND ("Unit1.EmNodes".emRelations.em12.sequence.stackNgBox.jobInterface.loadJob2.loadingReady OR "Unit1.Em13.ControlNodes".jrUnloadingPnP."step".transition1[431] OR NOT "Unit1.EmNodes".emRelations.em12.isLinked);
   #statTonTime[431].TON(IN := #_w1 AND "Unit1.Em13.ControlNodes".jrUnloadingPnP."step".transition1[431],
                         PT := T#1000ms);
   IF #statTonTime[431].Q THEN
       "Unit1.Em13.ControlNodes".jrUnloadingPnP.sequence.status.nextStep := #JOB_4_STEP_40;
   END_IF;
END_REGION

REGION Network 51: STEP[440] : Clamp Open
   RUNG wire#powerrail
      { S7_Templates := "SrcType := DInt" } EQ_Contact(in1 := "Unit1.Em13.ControlNodes".jrUnloadingPnP.sequence.status.currentStep, in2 := #JOB_4_STEP_40)
      Contact( "Unit1.Em13.ControlNodes".jrUnloadingPnP.sequence.status.seqActive )
      wire#w1
      I_Contact( "Unit1.Em13.ControlNodes".cmJRUnloadingPnPClampOpenClose.monitoring.inHomePos )
      Coil( "Unit1.Em13.ControlNodes".jrUnloadingPnP."step".action1[440] )
   END_RUNG
   RUNG wire#w1
      Contact( "Unit1.Em13.ControlNodes".cmJRUnloadingPnPClampOpenClose.monitoring.inHomePos )
      Coil( "Unit1.Em13.ControlNodes".jrUnloadingPnP."step".transition1[440] )
   END_RUNG
   RUNG wire#w1
      Contact( "Unit1.Em13.ControlNodes".jrUnloadingPnP."step".transition1[440] )
      { S7_Templates := "time_type := Time" } #statTonTime[440].TON(pt := T#1000ms, et =>)
      Move(in := #JOB_4_STEP_50, out1 => "Unit1.Em13.ControlNodes".jrUnloadingPnP.sequence.status.nextStep)
   END_RUNG
   // the same network as SCL:
   #_w1 := ("Unit1.Em13.ControlNodes".jrUnloadingPnP.sequence.status.currentStep = #JOB_4_STEP_40) AND "Unit1.Em13.ControlNodes".jrUnloadingPnP.sequence.status.seqActive;
   "Unit1.Em13.ControlNodes".jrUnloadingPnP."step".action1[440] := #_w1 AND NOT "Unit1.Em13.ControlNodes".cmJRUnloadingPnPClampOpenClose.monitoring.inHomePos;
   "Unit1.Em13.ControlNodes".jrUnloadingPnP."step".transition1[440] := #_w1 AND "Unit1.Em13.ControlNodes".cmJRUnloadingPnPClampOpenClose.monitoring.inHomePos;
   #statTonTime[440].TON(IN := #_w1 AND "Unit1.Em13.ControlNodes".jrUnloadingPnP."step".transition1[440],
                         PT := T#1000ms);
   IF #statTonTime[440].Q THEN
       "Unit1.Em13.ControlNodes".jrUnloadingPnP.sequence.status.nextStep := #JOB_4_STEP_50;
   END_IF;
END_REGION

REGION Network 52: STEP[450] : JR Unload P&P X-axis Work Ready Position
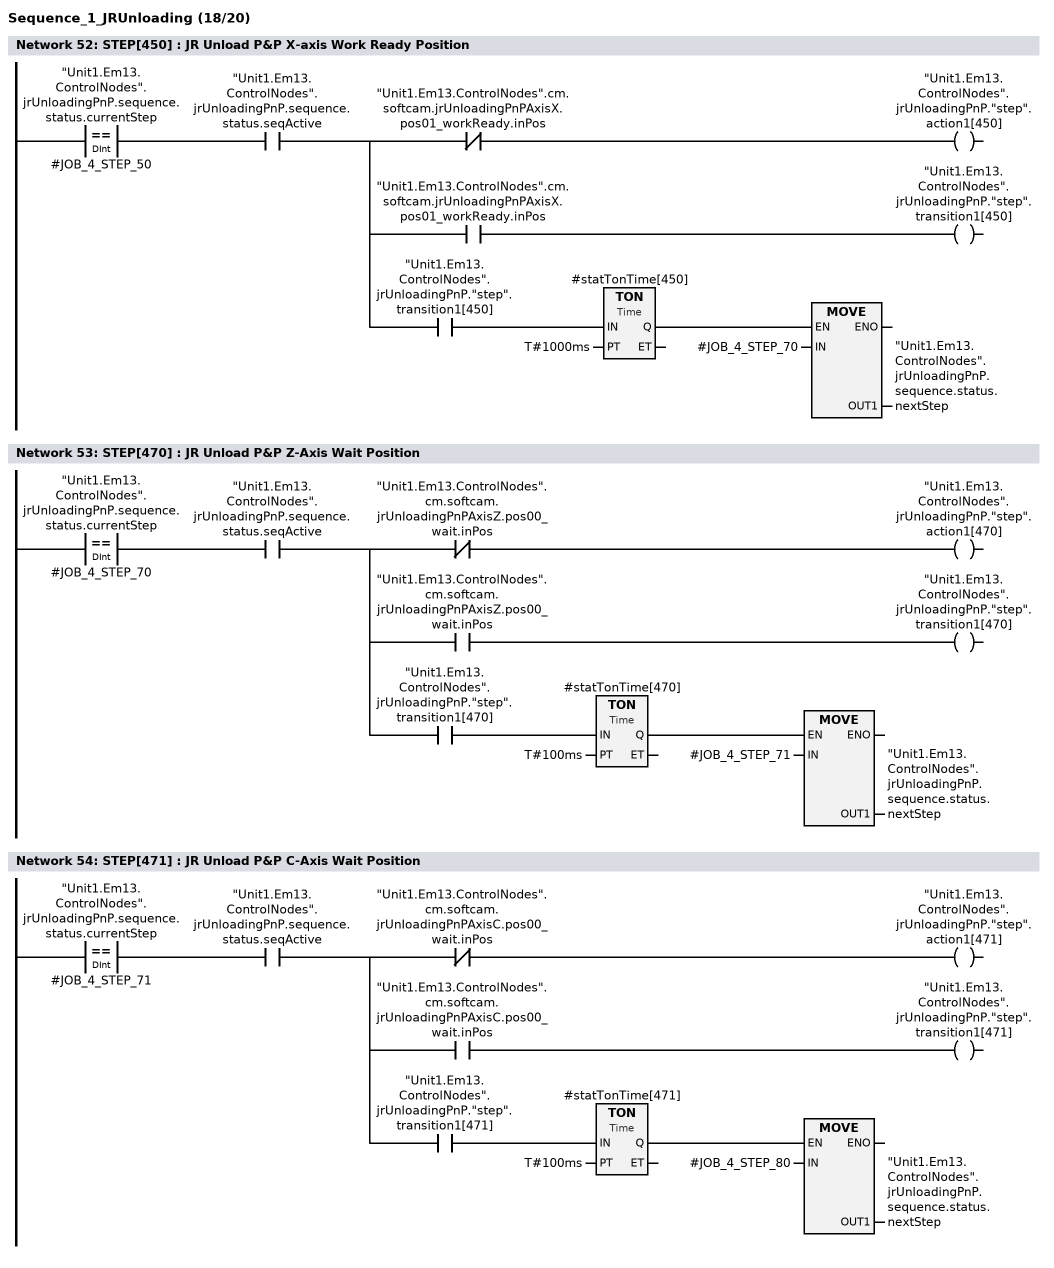
   RUNG wire#powerrail
      { S7_Templates := "SrcType := DInt" } EQ_Contact(in1 := "Unit1.Em13.ControlNodes".jrUnloadingPnP.sequence.status.currentStep, in2 := #JOB_4_STEP_50)
      Contact( "Unit1.Em13.ControlNodes".jrUnloadingPnP.sequence.status.seqActive )
      wire#w1
      I_Contact( "Unit1.Em13.ControlNodes".cm.softcam.jrUnIoadingPnPAxisX.pos01_workReady.inPos )
      Coil( "Unit1.Em13.ControlNodes".jrUnloadingPnP."step".action1[450] )
   END_RUNG
   RUNG wire#w1
      Contact( "Unit1.Em13.ControlNodes".cm.softcam.jrUnIoadingPnPAxisX.pos01_workReady.inPos )
      Coil( "Unit1.Em13.ControlNodes".jrUnloadingPnP."step".transition1[450] )
   END_RUNG
   RUNG wire#w1
      Contact( "Unit1.Em13.ControlNodes".jrUnloadingPnP."step".transition1[450] )
      { S7_Templates := "time_type := Time" } #statTonTime[450].TON(pt := T#1000ms, et =>)
      Move(in := #JOB_4_STEP_70, out1 => "Unit1.Em13.ControlNodes".jrUnloadingPnP.sequence.status.nextStep)
   END_RUNG
   // the same network as SCL:
   #_w1 := ("Unit1.Em13.ControlNodes".jrUnloadingPnP.sequence.status.currentStep = #JOB_4_STEP_50) AND "Unit1.Em13.ControlNodes".jrUnloadingPnP.sequence.status.seqActive;
   "Unit1.Em13.ControlNodes".jrUnloadingPnP."step".action1[450] := #_w1 AND NOT "Unit1.Em13.ControlNodes".cm.softcam.jrUnIoadingPnPAxisX.pos01_workReady.inPos;
   "Unit1.Em13.ControlNodes".jrUnloadingPnP."step".transition1[450] := #_w1 AND "Unit1.Em13.ControlNodes".cm.softcam.jrUnIoadingPnPAxisX.pos01_workReady.inPos;
   #statTonTime[450].TON(IN := #_w1 AND "Unit1.Em13.ControlNodes".jrUnloadingPnP."step".transition1[450],
                         PT := T#1000ms);
   IF #statTonTime[450].Q THEN
       "Unit1.Em13.ControlNodes".jrUnloadingPnP.sequence.status.nextStep := #JOB_4_STEP_70;
   END_IF;
END_REGION

REGION Network 53: STEP[470] : JR Unload P&P Z-Axis Wait Position
   RUNG wire#powerrail
      { S7_Templates := "SrcType := DInt" } EQ_Contact(in1 := "Unit1.Em13.ControlNodes".jrUnloadingPnP.sequence.status.currentStep, in2 := #JOB_4_STEP_70)
      Contact( "Unit1.Em13.ControlNodes".jrUnloadingPnP.sequence.status.seqActive )
      wire#w1
      I_Contact( "Unit1.Em13.ControlNodes".cm.softcam.jrUnIoadingPnPAxisZ.pos00_wait.inPos )
      Coil( "Unit1.Em13.ControlNodes".jrUnloadingPnP."step".action1[470] )
   END_RUNG
   RUNG wire#w1
      Contact( "Unit1.Em13.ControlNodes".cm.softcam.jrUnIoadingPnPAxisZ.pos00_wait.inPos )
      Coil( "Unit1.Em13.ControlNodes".jrUnloadingPnP."step".transition1[470] )
   END_RUNG
   RUNG wire#w1
      Contact( "Unit1.Em13.ControlNodes".jrUnloadingPnP."step".transition1[470] )
      { S7_Templates := "time_type := Time" } #statTonTime[470].TON(pt := T#100ms, et =>)
      Move(in := #JOB_4_STEP_71, out1 => "Unit1.Em13.ControlNodes".jrUnloadingPnP.sequence.status.nextStep)
   END_RUNG
   // the same network as SCL:
   #_w1 := ("Unit1.Em13.ControlNodes".jrUnloadingPnP.sequence.status.currentStep = #JOB_4_STEP_70) AND "Unit1.Em13.ControlNodes".jrUnloadingPnP.sequence.status.seqActive;
   "Unit1.Em13.ControlNodes".jrUnloadingPnP."step".action1[470] := #_w1 AND NOT "Unit1.Em13.ControlNodes".cm.softcam.jrUnIoadingPnPAxisZ.pos00_wait.inPos;
   "Unit1.Em13.ControlNodes".jrUnloadingPnP."step".transition1[470] := #_w1 AND "Unit1.Em13.ControlNodes".cm.softcam.jrUnIoadingPnPAxisZ.pos00_wait.inPos;
   #statTonTime[470].TON(IN := #_w1 AND "Unit1.Em13.ControlNodes".jrUnloadingPnP."step".transition1[470],
                         PT := T#100ms);
   IF #statTonTime[470].Q THEN
       "Unit1.Em13.ControlNodes".jrUnloadingPnP.sequence.status.nextStep := #JOB_4_STEP_71;
   END_IF;
END_REGION

REGION Network 54: STEP[471] : JR Unload P&P C-Axis Wait Position
   RUNG wire#powerrail
      { S7_Templates := "SrcType := DInt" } EQ_Contact(in1 := "Unit1.Em13.ControlNodes".jrUnloadingPnP.sequence.status.currentStep, in2 := #JOB_4_STEP_71)
      Contact( "Unit1.Em13.ControlNodes".jrUnloadingPnP.sequence.status.seqActive )
      wire#w1
      I_Contact( "Unit1.Em13.ControlNodes".cm.softcam.jrUnIoadingPnPAxisC.pos00_wait.inPos )
      Coil( "Unit1.Em13.ControlNodes".jrUnloadingPnP."step".action1[471] )
   END_RUNG
   RUNG wire#w1
      Contact( "Unit1.Em13.ControlNodes".cm.softcam.jrUnIoadingPnPAxisC.pos00_wait.inPos )
      Coil( "Unit1.Em13.ControlNodes".jrUnloadingPnP."step".transition1[471] )
   END_RUNG
   RUNG wire#w1
      Contact( "Unit1.Em13.ControlNodes".jrUnloadingPnP."step".transition1[471] )
      { S7_Templates := "time_type := Time" } #statTonTime[471].TON(pt := T#100ms, et =>)
      Move(in := #JOB_4_STEP_80, out1 => "Unit1.Em13.ControlNodes".jrUnloadingPnP.sequence.status.nextStep)
   END_RUNG
   // the same network as SCL:
   #_w1 := ("Unit1.Em13.ControlNodes".jrUnloadingPnP.sequence.status.currentStep = #JOB_4_STEP_71) AND "Unit1.Em13.ControlNodes".jrUnloadingPnP.sequence.status.seqActive;
   "Unit1.Em13.ControlNodes".jrUnloadingPnP."step".action1[471] := #_w1 AND NOT "Unit1.Em13.ControlNodes".cm.softcam.jrUnIoadingPnPAxisC.pos00_wait.inPos;
   "Unit1.Em13.ControlNodes".jrUnloadingPnP."step".transition1[471] := #_w1 AND "Unit1.Em13.ControlNodes".cm.softcam.jrUnIoadingPnPAxisC.pos00_wait.inPos;
   #statTonTime[471].TON(IN := #_w1 AND "Unit1.Em13.ControlNodes".jrUnloadingPnP."step".transition1[471],
                         PT := T#100ms);
   IF #statTonTime[471].Q THEN
       "Unit1.Em13.ControlNodes".jrUnloadingPnP.sequence.status.nextStep := #JOB_4_STEP_80;
   END_IF;
END_REGION

REGION Network 55: STEP[480] : JR Unload P&P X-Axis Wait Position
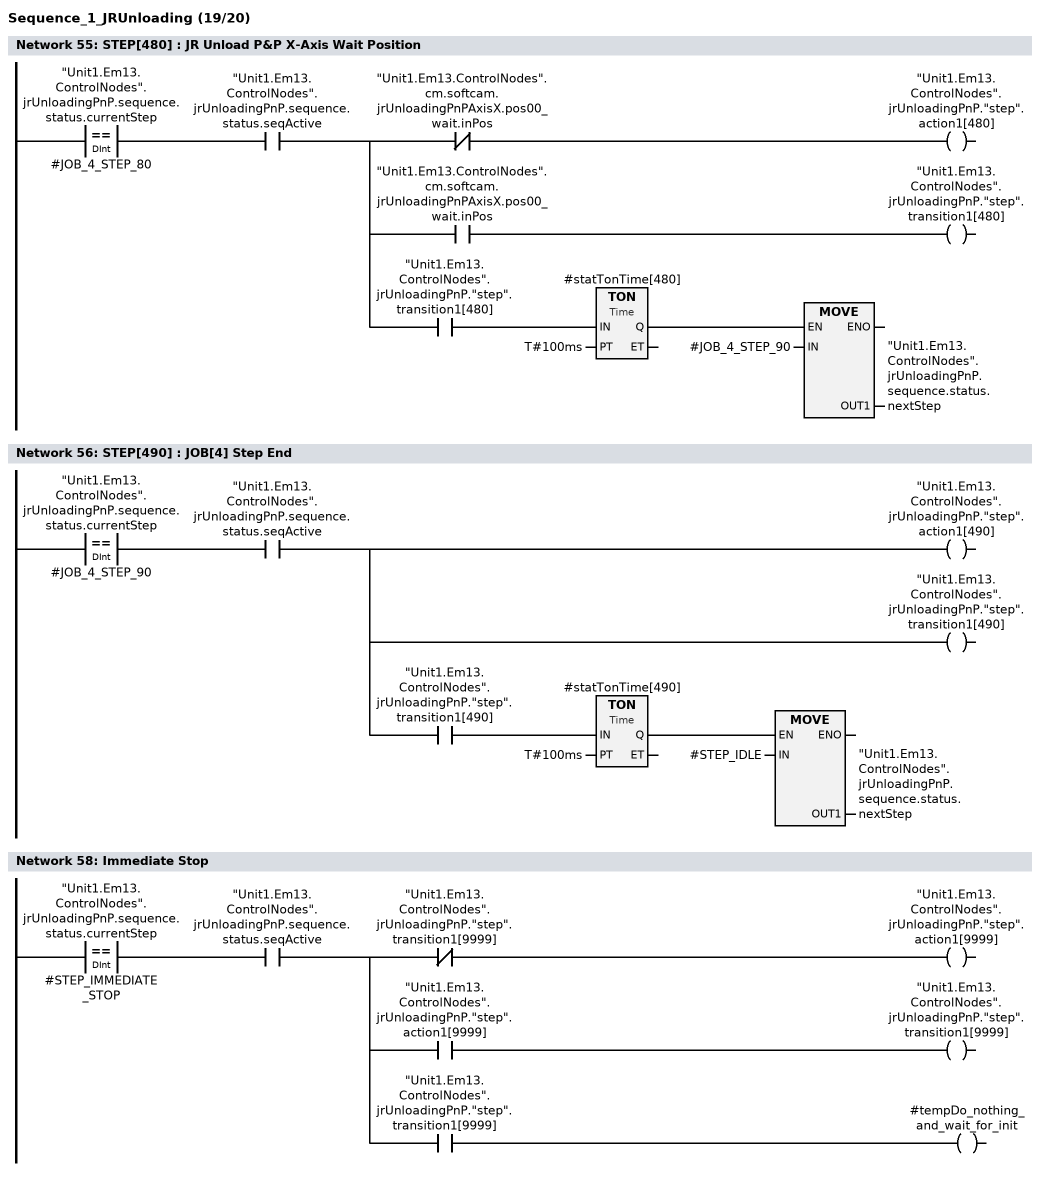
   RUNG wire#powerrail
      { S7_Templates := "SrcType := DInt" } EQ_Contact(in1 := "Unit1.Em13.ControlNodes".jrUnloadingPnP.sequence.status.currentStep, in2 := #JOB_4_STEP_80)
      Contact( "Unit1.Em13.ControlNodes".jrUnloadingPnP.sequence.status.seqActive )
      wire#w1
      I_Contact( "Unit1.Em13.ControlNodes".cm.softcam.jrUnIoadingPnPAxisX.pos00_wait.inPos )
      Coil( "Unit1.Em13.ControlNodes".jrUnloadingPnP."step".action1[480] )
   END_RUNG
   RUNG wire#w1
      Contact( "Unit1.Em13.ControlNodes".cm.softcam.jrUnIoadingPnPAxisX.pos00_wait.inPos )
      Coil( "Unit1.Em13.ControlNodes".jrUnloadingPnP."step".transition1[480] )
   END_RUNG
   RUNG wire#w1
      Contact( "Unit1.Em13.ControlNodes".jrUnloadingPnP."step".transition1[480] )
      { S7_Templates := "time_type := Time" } #statTonTime[480].TON(pt := T#100ms, et =>)
      Move(in := #JOB_4_STEP_90, out1 => "Unit1.Em13.ControlNodes".jrUnloadingPnP.sequence.status.nextStep)
   END_RUNG
   // the same network as SCL:
   #_w1 := ("Unit1.Em13.ControlNodes".jrUnloadingPnP.sequence.status.currentStep = #JOB_4_STEP_80) AND "Unit1.Em13.ControlNodes".jrUnloadingPnP.sequence.status.seqActive;
   "Unit1.Em13.ControlNodes".jrUnloadingPnP."step".action1[480] := #_w1 AND NOT "Unit1.Em13.ControlNodes".cm.softcam.jrUnIoadingPnPAxisX.pos00_wait.inPos;
   "Unit1.Em13.ControlNodes".jrUnloadingPnP."step".transition1[480] := #_w1 AND "Unit1.Em13.ControlNodes".cm.softcam.jrUnIoadingPnPAxisX.pos00_wait.inPos;
   #statTonTime[480].TON(IN := #_w1 AND "Unit1.Em13.ControlNodes".jrUnloadingPnP."step".transition1[480],
                         PT := T#100ms);
   IF #statTonTime[480].Q THEN
       "Unit1.Em13.ControlNodes".jrUnloadingPnP.sequence.status.nextStep := #JOB_4_STEP_90;
   END_IF;
END_REGION

REGION Network 56: STEP[490] : JOB[4] Step End
   RUNG wire#powerrail
      { S7_Templates := "SrcType := DInt" } EQ_Contact(in1 := "Unit1.Em13.ControlNodes".jrUnloadingPnP.sequence.status.currentStep, in2 := #JOB_4_STEP_90)
      Contact( "Unit1.Em13.ControlNodes".jrUnloadingPnP.sequence.status.seqActive )
      wire#w1
      Coil( "Unit1.Em13.ControlNodes".jrUnloadingPnP."step".action1[490] )
   END_RUNG
   RUNG wire#w1
      Coil( "Unit1.Em13.ControlNodes".jrUnloadingPnP."step".transition1[490] )
   END_RUNG
   RUNG wire#w1
      Contact( "Unit1.Em13.ControlNodes".jrUnloadingPnP."step".transition1[490] )
      { S7_Templates := "time_type := Time" } #statTonTime[490].TON(pt := T#100ms, et =>)
      Move(in := #STEP_IDLE, out1 => "Unit1.Em13.ControlNodes".jrUnloadingPnP.sequence.status.nextStep)
   END_RUNG
   // the same network as SCL:
   "Unit1.Em13.ControlNodes".jrUnloadingPnP."step".action1[490] := ("Unit1.Em13.ControlNodes".jrUnloadingPnP.sequence.status.currentStep = #JOB_4_STEP_90) AND "Unit1.Em13.ControlNodes".jrUnloadingPnP.sequence.status.seqActive;
   "Unit1.Em13.ControlNodes".jrUnloadingPnP."step".transition1[490] := ("Unit1.Em13.ControlNodes".jrUnloadingPnP.sequence.status.currentStep = #JOB_4_STEP_90) AND "Unit1.Em13.ControlNodes".jrUnloadingPnP.sequence.status.seqActive;
   #statTonTime[490].TON(IN := ("Unit1.Em13.ControlNodes".jrUnloadingPnP.sequence.status.currentStep = #JOB_4_STEP_90) AND "Unit1.Em13.ControlNodes".jrUnloadingPnP.sequence.status.seqActive AND "Unit1.Em13.ControlNodes".jrUnloadingPnP."step".transition1[490],
                         PT := T#100ms);
   IF #statTonTime[490].Q THEN
       "Unit1.Em13.ControlNodes".jrUnloadingPnP.sequence.status.nextStep := #STEP_IDLE;
   END_IF;
END_REGION

REGION Network 57: *************** IMMEDIATE STOP ****************
END_REGION

